(* IEC 61131-3 sources: ml2plc/benchmarks/st (part 19) *)

    weights_2 : ARRAY[0..287] OF REAL := [-0.086540468, 0.172771111, -0.220383257, -0.552691996, 0.0318835452, 0.612700164, -0.0329583585, -0.0454194695, 0.227657318, -0.476521522, 0.193516552, 0.416927308, 0.360883504, 0.35479334, -0.725205362, 0.0127351284, 0.00659608841, -0.077765286, 0.0985900313, 0.120690353, 0.105450228, 0.508144796, 0.130406424, -1.01746202, 0.904253662, -1.11978483, -0.232323259, 0.181972265, 0.00731435418, -0.0696650892, 1.03260088, -1.09293258, -0.287332207, 0.370921373, 0.321434826, -0.712032735, -0.0679141358, 0.179906562, -0.124551736, 0.192289323, -0.140516713, 0.0810432881, 0.856259704, -1.07160294, -0.223457828, 0.807030499, -0.976367593, -0.307652324, -0.786935031, -0.107092589, 0.150858521, -0.624960959, 0.36329934, 0.532729268, 0.384019405, 0.46479398, -0.802043259, 0.187860116, -0.136551112, 0.0211512949, 0.720803916, -0.827788591, -0.298880219, -0.202536553, 0.173984587, 0.185747623, -0.184981599, 0.0150071271, 0.00353488303, 0.0683722198, 0.187118113, 0.237856477, 1.01755667, -1.10523689, -0.268671334, 0.240274504, 0.30826062, -0.654990911, 0.872478366, -1.05786157, -0.229688749, -0.66336894, 0.0199285392, 0.532636046, -0.0841914713, 0.0642075539, 0.0174617469, -0.0364442356, 0.188555226, -0.242369831, 0.00474316673, -0.759811342, 0.954901636, 0.593428373, 0.096972242, -1.04332292, -0.205035418, 0.18625772, 0.209811807, 0.172150373, 0.0444886386, -0.186326519, 0.902395904, -1.12277734, -0.0967059359, -0.0028087846, 0.141072839, 0.130949974, 0.330060393, 0.323049426, -0.685176551, 0.492645383, 0.322297305, -0.804180861, -0.752909601, -0.107810475, 0.338000387, 0.220442653, 0.451399148, -0.57051903, -0.757164657, -0.126809373, 0.439987898, 0.0298772864, 0.00199659704, 0.166657642, 0.229579955, 0.268833876, -0.694251597, -0.0976240188, 0.0951045454, 0.2128084, -0.488305151, 0.345968217, 0.402587503, 0.0220696926, 0.122957081, 0.138620675, -0.146714658, 0.128199548, 0.0768355131, 0.988235116, -0.820175171, -0.0243866928, -0.564573824, 0.0925929025, 0.436609149, 0.605118215, 0.151139334, -1.10266984, 0.227359504, 0.0128947198, 0.0949031711, 0.120222516, 0.206790701, -0.00842625648, 0.120845072, 0.212780789, 0.12719503, -0.755692124, -0.150177613, 0.340954095, -0.853432715, -0.333076835, 0.391219765, 0.48939836, -0.116058439, -1.27640653, 0.0483904779, 0.217980474, -0.00876715779, -0.644433141, 0.0299610049, 0.399048507, 0.929591358, -0.906723499, -0.0457304083, 0.0974808037, -0.178352863, -0.0875617117, -0.169119462, -0.014128576, 0.133027628, 0.469002575, 0.474750727, -0.581674278, 0.372726113, 0.190089732, -0.973690569, -0.53365171, 0.140256211, 0.40247342, -0.113590144, -1.07570827, 0.916958451, -0.124050736, 0.0386698842, 0.104596823, 0.0975920856, -0.122577384, -0.230316952, 0.0917100608, -0.204680085, -0.157175794, 0.0664396286, 0.443755388, -0.550633371, 0.524068952, 0.155129775, -1.07333207, -0.0423594192, 0.0332752727, 0.193382502, -0.147190854, 0.123858854, -0.18527922, -0.251415074, -1.22913897, 0.845771313, -0.110015817, 0.065641731, 0.0683446452, 0.979607761, -0.910373867, -0.153985277, -0.0826165602, 0.125199199, 0.105670959, 0.127799779, -0.173133329, -0.0312328637, 0.147351772, 0.183071434, -0.226357937, -0.664937735, 0.321295112, 0.338666469, 1.03204453, -0.964660764, -0.207029104, 0.53012073, 0.460012823, -0.891147494, -0.551259696, 0.262762219, 0.241604507, 0.96495378, -0.912866771, -0.143412411, -0.645358205, 0.383842945, 0.425131768, -0.0753789395, -0.00826120377, 0.0299984515, -0.784333527, -0.1359182, 0.4243536, 0.178426176, -0.175408095, -0.077928111, -0.240787193, -0.203756183, 0.0390834771, -0.0964978486, -0.143233955, -0.104287267, 0.22191146, -0.0092907697, 0.138567775, -0.176785797, -0.841094136, 0.893011391, -0.736852944, 0.00464549148, 0.51239562, -0.529248655, 0.0516002066, 0.706514895, -0.518120229, 0.0655920431, 0.586107075, -0.604757965, 0.123719975, 0.379719675, 0.365877658, 0.503408611, -0.481252313];
    bias_2 : ARRAY[0..2] OF REAL := [0.0345217623, 0.145207137, -0.191580176];

END_VAR

VAR
    (* Merged variables from all regions *)
    buffer_0 : ARRAY[0..95] OF REAL;
    buffer_1 : ARRAY[0..127] OF REAL;

    (* Temporary computation variables *)
    i : DINT;
    j : DINT;
    t : DINT;
    sum : REAL;
    (* Computation helpers *)
    max_val : REAL;
    exp_val : REAL;
    exp_sum : REAL;
    (* Spatial loop variables *)
    oc : DINT;
    oh : DINT;
    ow : DINT;
    ic : DINT;
    kh : DINT;
    kw : DINT;
    ih : DINT;
    iw : DINT;
END_VAR

(* Forward pass execution *)

(* Region: r0 [ACYCLIC] *)
(* Acyclic Region r0 *)
(* Layer 0: Fused Linear + RELU *)
FOR j := 0 TO 127 DO
    sum := 0.0;
    FOR i := 0 TO 0 DO
        sum := sum + input_data * weights_0[i * 128 + j];
    END_FOR;
buffer_1[j] := MAX(sum + bias_0[j], 0.0);
END_FOR;

(* Layer 1: Fused Linear + RELU *)
FOR j := 0 TO 95 DO
    sum := 0.0;
    FOR i := 0 TO 127 DO
        sum := sum + buffer_1[i] * weights_1[i * 96 + j];
    END_FOR;
buffer_0[j] := MAX(sum + bias_1[j], 0.0);
END_FOR;

(* Layer 2: Fused Linear + SOFTMAX *)
FOR j := 0 TO 2 DO
    sum := 0.0;
    FOR i := 0 TO 95 DO
        sum := sum + buffer_0[i] * weights_2[i * 3 + j];
    END_FOR;
output_data[j] := sum + bias_2[j];
END_FOR;

(* Softmax: find max *)
max_val := output_data[0];
FOR i := 1 TO 2 DO
    IF output_data[i] > max_val THEN
        max_val := output_data[i];
    END_IF;
END_FOR;

(* Softmax: compute exponentials and sum *)
exp_sum := 0.0;
FOR i := 0 TO 2 DO
    output_data[i] := EXP(output_data[i] - max_val);
    exp_sum := exp_sum + output_data[i];
END_FOR;

(* Softmax: normalize *)
FOR i := 0 TO 2 DO
    output_data[i] := output_data[i] / exp_sum;
END_FOR;

END_FUNCTION_BLOCK

(* ---- MLP9_straton.st ---- *)
FUNCTION_BLOCK MLP9_FB

    (* Model Inputs/Outputs *)
VAR_INPUT
    input_data : REAL;
END_VAR

VAR_OUTPUT
    output_data : ARRAY[0..2] OF REAL;
END_VAR

VAR
    CONSTANT weights_0 : ARRAY[0..127] OF REAL := [-0.113805361, -0.131169349, -0.192945287, -0.0925860032, -0.117703564, 0.450317353, 0.395232439, -0.209253326, 0.52670908, -0.171847999, -0.00362640619, 0.448799431, 0.363001645, -0.0271579623, -0.0230307281, 0.528843641, 0.369391292, -0.0890475214, 0.398711413, -0.20652917, 0.420479208, -0.214330047, 0.343801081, -0.0572591722, 0.444781989, -0.109508358, 0.5149073, -0.195882052, 0.412400335, -0.190297425, 0.35653007, -0.00126373046, 0.476183206, -0.066968143, 0.488184482, -0.0159611255, -0.243453369, -0.186278701, 0.203586325, -0.212845653, -0.0807042271, -0.0202539116, 0.412385583, -0.144617856, -0.00571534038, -0.186419487, -0.193811327, -0.001996696, -0.204087764, 0.549255133, -0.182997674, 0.38119334, -0.182645351, -0.00299030519, 0.343619019, 0.518327653, 0.384723365, -0.20934774, 0.277335167, -0.172167048, 0.429218441, 0.469536155, 0.357460141, 0.234816477, -0.0928637683, 0.354974061, 0.0667782798, -0.128826559, 0.518400848, -0.0675187409, -0.198612809, -0.104182921, 0.397103459, 0.022735877, 0.368016571, 0.432546705, 0.49498266, -0.116236903, -0.0355618298, 0.522722244, -0.0902619362, -0.11224959, 0.353289217, -0.0632346869, 0.010258981, 0.431895882, 0.373197109, -0.130651206, -0.0309539437, 0.506278932, 0.413056433, 0.509223938, -0.0960097685, 0.367133349, 0.381490082, 0.457251966, 0.363914102, 0.42035231, 0.423214704, -0.188088998, -0.0470287502, -0.190154284, -0.162458539, -0.0485363007, -0.0830073208, -0.00753187714, 0.465610594, -0.205922633, 0.482488304, 0.448213607, 0.434718043, 0.34753862, 0.337949961, -0.031719774, -0.170038462, 0.495187283, -0.193692401, -0.172916174, -0.160878286, -0.200849622, 0.00499609578, -0.0520170256, -0.0275448263, 0.382134169, 0.507775307, 0.157361835, -0.0204105377, -0.147839844];
    CONSTANT bias_0 : ARRAY[0..127] OF REAL := [0, 0, 0, 0, 0, -0.100798227, -0.0795678124, 0, -0.108572058, 0, 0, -0.098264277, -0.0816824809, 0, 0, -0.0868740082, -0.0826022923, 0, -0.0856195465, 0, -0.0920739621, 0, -0.0772925317, 0, -0.0993444994, 0, -0.096356459, 0, -0.0921639502, 0, -0.080231972, -0.0145110283, -0.104885586, 0, -0.104719087, 0, 0.304739058, 0, 0.357667863, 0, 0, 0, -0.09254013, 0, 0, 0, 0, 0, 0, -0.119700968, 0, -0.0841121674, 0, -0.00373320258, -0.0695361495, -0.109383397, -0.0865293592, 0, 0.387899101, 0, -0.0930410847, -0.102059513, -0.0704434365, 0.379512459, 0, -0.0799476653, 0.354511678, 0, -0.0894547775, 0, 0, 0, -0.0889909193, 0.346559584, -0.0794480294, -0.0957549438, -0.101200089, 0, 0, -0.108003356, 0, 0, -0.07939253, 0, 0.350568563, -0.0959382132, -0.0757256672, 0, 0, -0.100857422, -0.0881503075, -0.105426408, 0, -0.0800946504, 0.326970756, -0.0932597071, -0.081825532, -0.0898775011, -0.0926302895, 0, 0, 0, 0, 0, 0, -0.00774373114, -0.0858005881, 0, -0.103054315, -0.0990050733, -0.0953028128, -0.0783599094, -0.0757565275, 0, 0, -0.100662939, 0, 0, 0, 0, -0.0165398363, 0.298638582, 0, -0.0855023414, -0.0985088944, 0.363575578, 0, 0];
    CONSTANT weights_1 : ARRAY[0..12287] OF REAL := [0.0951577127, 0.157444745, -0.116936132, -0.0790329278, -0.0228748918, 0.0134683251, 0.110163182, 0.0660780072, -0.0495770946, -0.0592429936, 0.134160757, -0.160569534, -0.0958634838, 0.142136246, 0.0809055567, -0.0727666095, -0.161114678, -0.133757368, 0.0792375952, 0.0649654567, 0.0525315702, -0.0809695944, -0.0614370704, -0.135633662, -0.00297276676, -0.0548477396, 0.128665984, -0.160567224, 0.00753733516, 0.0283032507, 0.12481007, 0.0217095912, -0.0424018651, 0.105811566, -0.0234863013, -0.0909486711, 0.050266549, -0.0875409767, -0.0314820856, 0.0861708969, -0.104749173, 0.0864515305, -0.0256673396, -0.078911148, 0.105528295, -0.106350139, 0.00202976167, 0.11709699, -0.0761083886, -0.15657708, 0.137355566, 0.0239440948, 0.131604254, -0.0955468714, -0.14261815, -0.0404164344, -0.05397138, -0.0310050994, -0.0330105126, 0.0184245408, -0.111915424, 0.0973271728, 0.103177726, 0.149213344, -0.0549873933, 0.0881988704, -0.0177367181, 0.124477774, -0.0285055786, -0.109965578, 0.0402032584, 0.0121235251, -0.0266363323, 0.125837356, -0.0728950202, -0.0705690533, 0.0583580136, 0.0598951429, 0.0236688703, 0.0522443801, 0.00132079422, 0.125945359, -0.00138136744, 0.0651458055, -0.120777965, -0.104297861, 0.0417176485, -0.161106139, -0.0645132065, 0.0710417032, 0.0645282269, -0.0479533747, 0.13674435, 0.106236696, -0.0604583621, 0.0287175775, -0.00439415872, -0.00736361742, -0.134950846, -0.135192379, 0.10444808, 0.0236009806, -0.103126153, 0.0975316465, 0.139209658, 0.0520739704, 0.125309825, -0.0581694618, -0.162468061, -0.0841054246, 0.0483714789, -0.0566895753, -0.0466354638, -0.104527183, -0.007353127, -0.0725882053, 0.0929109752, 0.113443941, 0.0509717613, 0.0587531328, -0.117151141, 0.0126229078, 0.0203929991, 0.047550723, 0.0517018735, -0.101339415, -0.138496399, 0.00150629878, 0.0771658868, -0.00845770538, 0.0908749104, 0.0518915504, 0.0117899328, -0.145934269, 0.0225093067, -0.0222804546, -0.00221456587, 0.0128537863, -0.0276821703, -0.120568201, -0.0423685834, 0.116727293, -0.0766037181, -0.0683219507, 0.138370246, 0.146753311, 0.0569230765, -0.0658973753, 0.0545879006, 0.105433077, -0.0373315513, 0.161194414, 0.0101915747, -0.0552281886, -0.103356332, 0.0682205409, 0.0157359093, -0.0698226318, -0.0442622453, -0.0125101805, -0.033475399, 0.0732399672, -0.149365753, -0.123059414, -0.124025911, 0.0979141891, -0.0852181315, -0.123718902, -0.137371242, 0.0357241184, 0.132824361, -0.160526261, 0.00875844061, 0.14891094, 0.020388782, 0.127746224, -0.0733599514, 0.12927103, 0.156546056, 0.144431114, -0.058117643, -0.0785800591, -0.0507855564, -0.160170823, -0.0641571879, -0.027300939, 0.108366787, -0.0391465947, 0.0696284622, 0.0237422287, -0.11445865, -0.11570774, 0.0200967491, -0.131474406, 0.120322555, 0.106915504, 0.106001765, 0.15025726, 0.148201168, 0.0288652182, 0.0153841078, 0.147035837, -0.0442098752, 0.0455059856, 0.08771047, -0.0411697626, 0.0291817933, 0.118134856, 0.101055682, -0.000335618854, -0.0269186497, 0.015304774, 0.0589915514, -0.02176328, -0.14560017, -0.0776190683, 0.0365733057, -0.0838752836, 0.153584182, 0.134814322, 0.148770154, -0.0831061155, 0.0914156139, 0.077782169, 0.0720475763, -0.0280352235, 0.0480267406, 0.0686243623, 0.0797413886, 0.0645133257, -0.0962903649, 0.0324638784, -0.0570613667, -0.0719860792, 0.111080825, 0.119137555, -0.055265218, 0.0108719021, -0.0382692516, 0.146787912, -0.100032538, -0.0835579708, 0.00157497823, -0.162271053, 0.119353175, -0.0655590296, 0.0131833553, 0.069874689, -0.0753858536, -0.0472645536, -0.0861709341, 0.0184095502, 0.142682731, 0.0667904317, 0.000965476036, -0.115095079, -0.0968379378, -0.121067345, -0.0672623515, -0.112838328, -0.0351838768, -0.137819111, -0.112566784, -0.155080765, 0.138557822, -0.162448362, -0.12402942, 0.0698025823, 0.118413299, 0.139092475, -0.0617644563, -0.125346243, 0.0916123688, 0.076207146, -0.0628192499, -0.128253579, 0.120955229, 0.148212641, -0.0932002217, 0.117295235, 0.161221325, -0.106977157, 0.0483250469, -0.150214329, 0.0903045833, 0.0870901346, 0.149560899, -0.0276673287, -0.151596636, 0.0847090334, 0.127780765, -0.15172115, -0.118571639, 0.0389828235, 0.0767906606, -0.0856763497, 0.0160828382, -0.121637389, 0.0912489295, -0.14491263, 0.131868184, 0.0672539175, 0.0127351731, -0.00589309633, -0.0622787848, -0.141520515, -0.0427362323, -0.0998942479, 0.149263471, -0.152347118, 0.0028988719, -0.00683000684, 0.146410555, -0.0533801764, 0.0977630019, -0.00881588459, -0.160895512, -0.0131007433, 0.0372889936, 0.126067817, 0.11309135, 0.0728558898, -0.0335129797, -0.0818832964, -0.0330946892, -0.0781284794, -0.155981824, 0.0711639673, -0.0405116826, 0.0357084721, 0.142399669, 0.138510466, -0.114842109, 0.0368577391, -0.0718035027, -0.0764543861, -0.107536398, -0.139627516, 0.00174733996, 0.094630897, 0.0877837241, -0.0499476343, 0.0859448165, -0.0901338086, -0.121612534, 0.0269791335, 0.0815927088, 0.0611288548, -0.0593353137, -0.153852284, -0.0354756266, -0.0991432667, 0.141438067, -0.00173516572, -0.0234908611, 0.0649795383, -0.114180557, -0.142907768, 0.0548550785, 0.0757389814, 0.0898238719, 0.0306845456, -0.0634233654, 0.149431825, -0.0129109174, -0.0298580527, 0.0128320903, -0.119393483, -0.0556279495, -0.048238501, -0.110748321, 0.160280555, -0.107997969, -0.129245013, -0.0782359764, 0.0218218118, 0.0503502041, 0.101736844, 0.0445458442, -0.0318994522, -0.048770234, 0.0895831585, -0.138157532, 0.0388857722, 0.111648083, 0.145862103, 0.0815838128, 0.054871738, -0.0941967666, -0.126886413, -0.0578072369, 0.0876997113, -0.108099304, -0.0487953201, -0.131870151, 0.0197252482, -0.0851159021, 0.0999375284, 0.157903999, -0.0588724166, 0.152515322, -0.0926127732, 0.109808058, 0.161163688, 0.153266072, 0.108911484, 0.0491682738, -0.157219395, 0.0929915309, 0.0676452518, -0.0539523736, 0.0412925184, 0.0595459938, -0.115160167, -0.0217127502, 0.0798177123, -0.00466352701, 0.0912430882, 0.0433716774, -0.145626664, 0.148768365, 0.0322260559, 0.131735057, -0.131727949, 0.0504067838, 0.00729522109, -0.039368853, 0.121461481, 0.132999808, -0.0395063236, 0.00795516372, 0.145861775, 0.105656266, -0.156878084, 0.00268745422, 0.117816895, -0.124721214, -0.0546680093, 0.0303108841, 0.0794312507, -0.0877228901, -0.0310570002, -0.135552973, -0.121911898, -0.120446339, 0.0388385206, 0.108996451, 0.0305833668, -0.0586595982, -0.140537083, 0.160965115, -0.125315413, -0.0336649269, 0.144092739, 0.0993903279, 0.116826385, 0.0198810548, 0.130669534, -0.007835567, 0.0403493196, 0.149000049, 0.0241642743, 0.16068995, -0.0206242353, 0.0651469827, -0.0246725529, 0.067141965, -0.0331727564, -0.144538388, -0.0538310185, -0.0991705433, -0.0017388314, 0.16014412, -0.106752947, 0.101663619, -0.142054304, -0.107962027, 0.019818306, -0.0550122112, -0.0132327527, -0.0847105384, 0.509194136, 0.0538960695, 0.604936779, -0.265589058, -0.140676975, -0.00574114919, -0.43431446, -0.453494668, 0.0540918261, -0.406886041, -0.21926257, 0.163309574, -0.143326595, -0.642100513, -0.723519862, 0.570846677, 0.244765401, -0.379419535, 0.00814934261, -0.540151834, 0.154496402, -0.0546880662, 0.161006272, -0.4712421, -0.312546521, -0.449770659, 0.659415066, -0.13482137, 0.0830492079, 0.52391237, -0.565974474, 0.158174455, -0.0621462315, -0.70691061, -0.154083952, -0.360878319, -0.407535791, 0.656996191, -0.369862318, 0.627200603, 0.069169119, -0.546665549, 0.0077586174, 0.4769786, 0.140734434, -0.0507009253, -0.760944128, 0.602752507, -0.571398199, 0.0918866098, 0.00788346305, 0.0322130509, 0.288204491, 0.329203099, -0.392646372, 0.0749019235, 0.320154548, -0.691001058, 0.112304956, -0.125678852, -0.333393902, -0.394726753, 0.752456069, 0.394099623, -0.124766201, 0.0376506299, -0.0682738349, -0.246535376, -0.51199317, -0.137057155, 0.122536659, 0.519263268, 0.0833194107, -0.686214447, 0.123675488, 0.141091406, 0.155417144, 0.331035525, -0.519244015, -0.223143131, 0.621623278, -0.614489675, 0.437765509, 0.0805219561, 0.413208932, -0.0631952509, -0.0913754106, 0.0515855551, -0.160588577, 0.397252113, 0.431347072, 0.408398241, 0.408925176, 0.597231805, -0.336975992, 0.0440444462, 0.270032376, -0.121744737, 0.549877822, -0.422593564, -0.0661128834, -0.17437312, -0.417972744, -0.310103178, -0.0716258809, -0.33077088, -0.205869734, -0.153525308, -0.139355108, -0.438011259, -0.584835529, 0.465125173, 0.344738692, -0.14478299, 0.156904221, -0.624013662, -0.153481901, 0.0398430228, -0.0846624002, -0.516546309, -0.242195129, -0.376353711, 0.532166958, -0.144245222, 0.0689140931, 0.36220032, -0.267864943, 0.057710737, 0.0646699518, -0.586554945, -0.0401847661, -0.248956472, -0.272385627, 0.415772557, -0.0767131969, 0.310505778, -0.0379597098, -0.274617344, 0.126220137, 0.480036318, -0.0241271257, 0.0331539959, -0.324106157, 0.501049876, -0.291424572, -0.0870115086, 0.0509127118, 0.0394147225, 0.584093153, 0.503804743, -0.218451321, 0.00519318879, 0.607654095, -0.3049227, 0.145615906, 0.05105225, -0.202767462, -0.423024982, 0.729864001, 0.276849747, 0.0496818721, 0.0660526454, 0.0130212307, -0.0571260527, -0.439201325, 0.0459277742, -0.0404780358, 0.408804804, 0.0655715987, -0.476458848, -0.0844522044, 0.124375969, 0.114283532, 0.39356488, -0.548989713, -0.34556523, 0.631348431, -0.40491116, 0.518371046, 0.135800749, 0.560781419, -0.00710113347, 0.0723592117, 0.0476910472, -0.124959633, 0.328189194, 0.532768965, 0.587405443, 0.499420702, 0.671146929, -0.352552384, 0.0768999159, -0.0319315642, -0.100787431, -0.0804701298, -0.146786034, 0.141987205, 0.0561998785, 0.0398712754, 0.0927682817, 0.109196901, -0.0432840809, 0.0716784894, 0.0145284683, -0.095403865, 0.0917330086, -0.15252769, -0.110293895, -0.0509034023, 0.0978683233, 0.0202671587, 0.00549578667, -0.135518357, -0.146398097, 0.124808073, -0.13327761, -0.13578631, -0.0443552658, -0.123986423, 0.163084328, -0.0966529474, -0.134083807, 0.0854204893, -0.0765637606, -0.0741811767, -0.00683036447, -0.118621819, -0.039869912, -0.162193045, -0.104409263, -0.056582585, -0.001865834, 0.154557496, 0.0310758501, 0.0742693543, -0.0389179736, 0.112253129, -0.0996025354, 0.038610369, -0.0614454597, 0.0836289823, 0.107963115, 0.140558034, 0.0794830322, 0.163360059, -0.163278833, -0.0120799392, -0.0656130388, 0.00880923867, -0.0657925308, -0.0760729611, -0.075019531, 0.114507735, 0.0841428488, 0.0406958908, 0.11450699, -0.151554912, -0.122948989, 0.0699587762, -0.110302597, 0.00226099789, 0.0974447727, 0.0653391182, 0.108267993, -0.0920944661, 0.15465036, 0.112603068, 0.0013948977, 0.14819929, -0.144036621, -0.016038239, -0.139199302, -0.0771588236, -0.0928127542, -0.0338050127, -0.0522177219, -0.157671407, -0.00344249606, -0.0332395732, -0.113233492, -0.158796951, -0.13916111, 0.0589568615, 0.0945762098, 0.14930898, 0.0418180823, -0.0978229716, 0.0602630973, 0.322021961, -0.0053896904, 0.467693686, -0.249736562, 0.126417518, -0.138710305, -0.363732606, -0.456968129, -0.0944563299, -0.472876072, -0.21804218, -0.143095255, 0.0928375497, -0.57138437, -0.472568661, 0.646057606, 0.351664901, -0.415040404, -0.111070551, -0.65686512, -0.10573642, -0.0150539875, -0.144721866, -0.56100738, -0.30737561, -0.586903989, 0.616061807, -0.043527022, -0.0646082535, 0.434298456, -0.282648176, -0.0882620364, -0.12533547, -0.59989053, 0.125016868, -0.46765244, -0.364355326, 0.523267984, -0.340620995, 0.308997214, -0.018915683, -0.40029791, 0.0643675029, 0.254231155, -0.00991281867, 0.117880344, -0.428295225, 0.443931401, -0.469592839, -0.0985035226, 0.0645282492, 0.0728940368, 0.45560959, 0.487523675, -0.384809881, 0.0336826444, 0.39610061, -0.386167377, -0.0381661206, -0.136605546, -0.445077538, -0.44675684, 0.475525707, 0.245289952, -0.161932707, -0.115931481, 0.0207827687, -0.0385752581, -0.230016008, -0.143260673, -0.0719312429, 0.350897193, -0.112227477, -0.549400151, 0.0996975377, -0.158407763, -0.00293686986, 0.503760517, -0.545467556, -0.259034455, 0.453600407, -0.456205547, 0.487957925, -0.122733943, 0.287507385, 0.0341648608, -0.0692357272, 0.137745768, -0.02918984, 0.201632515, 0.316503704, 0.563527167, 0.428642005, 0.695099711, -0.341352791, 0.14451462, 0.00366416574, -0.0520999208, 0.0875412226, -0.116182968, -0.157112911, 0.114217222, -0.0688723326, -0.121052325, 0.0575330406, 0.0796439499, 0.0595702976, 0.0227632523, -0.0794479102, 0.126714766, -0.0488853008, 0.0934711695, 0.122365475, -0.0437675789, 0.0868758857, -0.0134203285, 0.0346060544, -0.0367608815, 0.0463865548, -0.0707047656, 0.150832742, -0.128055975, -0.0556442216, 0.00231200457, -0.111579061, -0.0886108428, -0.129191309, -0.161951363, 0.0831619501, -0.0794863105, 0.103473008, 0.159343034, -0.0559051931, 0.062377587, -0.121212967, 0.0833023041, -0.162734151, 0.0321030617, -0.10398519, -0.138421714, 0.045194909, 0.142874509, -0.0367347449, -0.155020788, -0.152351826, 0.0173095316, -0.0145311207, 0.0364078283, 0.0694433898, 0.031635046, 0.0519284606, 0.1198695, -0.0134465098, -0.142700329, 0.0394844264, -0.158252656, -0.0392903835, -0.0576177537, -0.0491104871, 0.0735302418, 0.0511014611, 0.109477192, 0.0833617002, 0.101866454, 0.0914892256, 0.00224284828, 0.126525789, 0.137383074, 0.0791972429, -0.0692049414, -0.125604168, 0.128060102, -0.0253694654, 0.0628164113, 0.03625682, 0.159057289, 0.0904439092, -0.0538290292, -0.162247017, 0.00659917295, -0.0887682065, -0.0221569985, -0.0965008438, 0.104463339, -0.0614345372, 0.0150002241, 0.0888507366, 0.115881771, -0.111798167, 0.0199936181, -0.154604435, 0.0775321275, -0.02869986, 0.0626578331, -0.0132484436, -0.0378343761, 0.0255666375, -0.137642473, 0.0340280831, 0.0923664272, -0.132832348, -0.161153629, -0.0162264407, -0.138787255, -0.0474235192, -0.10354051, -0.0473156273, 0.0843745917, -0.151293129, 0.124063998, 0.113260567, -0.137583464, 0.0871079266, 0.0880226791, 0.123843074, 0.1298002, 0.0235676616, -0.118507646, -0.130145669, -0.0655051842, 0.0768328458, -0.0903019831, 0.120177537, -0.109550744, -0.12586607, 0.119989842, -0.06112881, 0.150598377, -0.0707290024, 0.0344911516, 0.103849113, -0.135946766, -0.0548578054, 0.0875094533, 0.113336772, 0.096303165, -0.068084158, 0.114509881, 0.1175614, -0.0225681514, 0.146655113, -0.00232343376, -0.0178669691, 0.054963395, -0.140081167, -0.0873917267, -0.101093426, -0.0865101367, -0.0871431231, -0.109610252, -0.147202581, -0.0557942912, -0.0006223768, -0.134950295, 0.162944168, -0.0371381789, 0.129121751, 0.157590866, 0.122555614, -0.00439842045, 0.156742811, -0.105628684, 0.0453346372, -0.0737311915, -0.0812637657, 0.127866268, 0.059443593, -0.0491509959, -0.0971391797, -0.143130645, 0.0233585835, -0.0147621185, -0.159102827, 0.149393588, 0.0969157219, -0.102926373, 0.154051632, 0.112800837, 0.0364580452, -0.0520509854, 0.0394695997, 0.0302900523, 0.1545147, 0.0542997718, 0.0890843868, 0.0546405762, 0.0287235081, -0.173261896, 0.490024894, 0.0681065172, 0.361833811, -0.328347623, -0.0356032252, -0.133056432, -0.494118333, -0.601521552, -0.121832028, -0.589727759, -0.277259827, 0.111315638, 0.0659579858, -0.741538644, -0.492740691, 0.550138712, 0.320899546, -0.288761914, -0.00195023709, -0.537688792, 0.099278003, 0.00579982996, -0.0347415805, -0.72761929, -0.377573043, -0.555244505, 0.456523657, 0.0320400745, 0.036451485, 0.486669511, -0.378461182, -0.152018994, -0.136228755, -0.720117569, 0.0192903578, -0.531963825, -0.469921142, 0.589513958, -0.366701841, 0.412990361, -0.158252299, -0.364246905, -0.160873383, 0.37125057, -0.00136806071, 0.0729077011, -0.559927881, 0.583796501, -0.387921512, 0.00662960112, 0.00455707638, -0.0358150043, 0.490136683, 0.529693484, -0.326329947, 0.022318691, 0.567211449, -0.707156956, -0.149156183, -0.132085413, -0.527429581, -0.507927239, 0.653061748, 0.349608958, 0.152013838, 0.0440299511, -0.0555629432, -0.101837404, -0.348313838, 0.0049868077, -0.0747583583, 0.262050003, -0.159494683, -0.424277574, -0.149270624, -0.160396859, 0.0718324929, 0.430129915, -0.734822154, -0.220166579, 0.418183774, -0.722909093, 0.251368821, 0.00369682908, 0.448462456, 0.131171644, -0.0492361449, -0.00822554529, -0.146481872, 0.301343501, 0.379717827, 0.573642671, 0.471275508, 0.538758397, -0.350973874, 0.12145821, 0.671127796, 0.116494, 0.640164316, -0.551232457, 0.0458213836, 0.122570068, -0.612397373, -0.660989344, -0.088481836, -0.605110645, -0.603729784, 0.0518653244, 0.139900357, -0.674467802, -0.719813704, 0.707245648, 0.596261024, -0.500923991, -0.00499203429, -0.699686885, 0.0658935606, 0.0570179373, 0.1512371, -0.636342168, -0.418134749, -0.620170534, 0.763878882, -0.002538234, -0.0417705178, 0.420946479, -0.688793957, 0.064556092, 0.157188416, -0.759609997, 0.0812719166, -0.453400403, -0.567348719, 0.724059165, -0.203651771, 0.611069858, 0.0227045268, -0.291180491, -0.157189071, 0.754448414, 0.085985437, -0.119775772, -0.712979138, 0.698715329, -0.58169204, 0.148470551, 0.0952268913, 0.0562097244, 0.633901775, 0.590043008, -0.511904299, -0.128872991, 0.575819671, -0.675768137, -0.0152154565, -0.00212833285, -0.472860008, -0.69616574, 0.622911692, 0.343438059, -0.0224477351, -0.0405841023, 0.0385661274, -0.257873476, -0.396772712, -0.152293921, -0.156207159, 0.595220387, -0.0240174532, -0.615511596, -0.13495256, -0.106912807, 0.0843406469, 0.526772499, -0.736953795, -0.275285572, 0.692019939, -0.582976937, 0.498922467, 0.0128312707, 0.633550167, -0.0273342133, 0.109861545, 0.103651047, -0.0617552027, 0.510849655, 0.394558609, 0.545751154, 0.393026024, 0.793120563, -0.497044265, 0.092567116, 0.138860226, -0.0985106304, 0.00336945057, -0.130671352, -0.111542739, 0.143976063, 0.0285258293, 0.113393039, -0.0218960196, 0.0309942961, -0.0104740858, 0.0956641138, 0.0878303051, 0.102058023, 0.00174370408, -0.117548563, -0.155215263, 0.134208828, 0.0980995595, -0.134259984, 0.0419485718, -0.0534096435, 0.0429573655, 0.0513623953, -0.14403373, 0.06175825, -0.122290827, 0.0777258277, -0.151134908, 0.0914635062, 0.140266359, -0.00751279294, 0.00970570743, -0.0983380377, 0.0919840634, -0.0801352561, 0.0911718011, 0.108400077, -0.161801755, 0.135701865, -0.131035775, -0.0860919133, 0.0889713168, -0.0941296518, -0.0192143917, 0.100918174, -0.0230973512, 0.117296249, 0.133148789, 0.156041861, -0.0570620298, -0.0986587107, -0.148947418, -0.135748416, -0.0595284253, -0.134941593, 0.117915601, 0.0543765277, -0.124985032, 0.066407606, 0.0267682225, 0.0470175147, -0.162895411, -0.149206594, 0.153207392, -0.00830924511, 0.00621114671, 0.146200955, 0.132364035, -0.154241115, 0.0508376509, 0.0611464828, 0.121670395, 0.104352921, 0.0689978153, 0.0547138155, 0.0552895218, -0.154357553, -0.0046634376, 0.118674546, -0.0442880765, -0.0731509998, 0.00893263519, -0.0351747423, 0.014497757, 0.0777242631, -0.111611374, -0.0725884363, -0.112329312, -0.0154200494, 0.146003842, -0.00320079923, -0.163586318, -0.0718479902, 0.0270866752, -0.0277421027, 0.154627293, 0.0143596977, 0.131777287, -0.116288751, -0.142893523, -0.157827795, -0.0544529706, -0.0255519301, -0.0792789161, -0.0977822319, 0.143588871, -0.124468245, 0.0958327651, -0.0322359949, 0.00266860425, -0.1135519, -0.140336871, -0.14343977, -0.113305256, -0.0109504908, 0.0786850303, 0.0330305398, -0.00475849211, 0.0163063854, -0.0716166347, -0.0528806821, 0.0159133375, -0.0289545059, -0.15040499, 0.153120875, -0.0435663164, -0.0760979354, 0.160244167, -0.0592714772, 0.132729143, -0.00471362472, -0.0540071949, -0.0376077443, 0.0736211985, 0.0239118934, 0.0179463774, 0.0792258084, -0.1428767, 0.158036083, 0.15304625, -0.0280214399, -0.0129368603, 0.0730203241, 0.00552131236, -0.102222949, -0.00217039883, 0.149807036, 0.0687736124, -0.0731835365, 0.0183587819, -0.0314919204, -0.119318336, -0.0418934301, -0.118667156, -0.141958326, -0.00374318659, -0.0770075023, -0.129735336, -0.119574621, 0.0406397432, -0.152146041, -0.0276105553, -0.0321829766, 0.0301983207, 0.0734649152, -0.0383871794, -0.158686012, 0.0197154433, 0.136941463, -0.0486620665, 0.0317238569, 0.135865867, -0.0451636165, 0.0228485912, 0.127936155, -0.0893768072, 0.0435742736, -0.0214909464, 0.0240473002, 0.103848428, -0.122813389, -0.0357450694, -0.0580369905, -0.0383514315, -0.0267788023, -0.0101375729, -0.0783320889, 0.0894583762, -0.11558798, 0.00936958194, -0.171604529, 0.37826997, -0.139284834, 0.530997694, -0.212191448, -0.00569155812, -0.13463667, -0.152116403, -0.322950393, 0.0285518467, -0.350297242, -0.0644152015, -0.0703600869, 0.0551211797, -0.260502994, -0.240122318, 0.572239399, 0.46966812, -0.211586058, -0.0670061857, -0.311251044, 0.0108838379, -0.0651359409, -0.150437683, -0.45188126, -0.119499251, -0.282272905, 0.483443588, -0.105406582, 0.00445411028, 0.432145655, -0.332937509, 0.0562750995, 0.046805948, -0.397827655, 0.00858733058, -0.166388154, -0.121550895, 0.298872322, -0.187453955, 0.401923031, -0.0599540249, -0.302921563, 0.0653752834, 0.423189819, -0.0816778094, -0.0318836868, -0.39043653, 0.558439434, -0.0932632908, -0.0381754935, 0.0619168989, -0.0710496083, 0.174890399, 0.151282564, -0.119489975, 0.0900167823, 0.294368684, -0.483624071, 0.00194258988, -0.0865473673, -0.32862553, -0.157639489, 0.403094679, 0.387990355, -0.0647413582, -0.0843798593, 0.115365654, 0.0828580633, -0.151365161, -0.0210992191, 0.113412887, 0.254138768, 0.151015371, -0.398343295, 0.108841717, -0.00285227597, -0.123278439, 0.263769329, -0.393478274, -0.168504938, 0.443632662, -0.519051313, 0.384981513, -0.123920478, 0.161044911, 0.0879419446, -0.115611427, 0.0700436532, 0.0192385763, 0.17883873, 0.29301405, 0.17283237, 0.403273553, 0.477420956, -0.0488811806, 0.0120467003, 0.375956684, 0.12920621, 0.699442625, -0.524834216, -0.121545583, -0.137277544, -0.379925132, -0.548032999, -0.137724444, -0.607119679, -0.298528701, -0.047074832, 0.124948837, -0.770748496, -0.59968704, 0.591483057, 0.494383752, -0.383634984, -0.0311492104, -0.839230597, 0.0822430253, 0.108918607, 0.0935982764, -0.704104125, -0.356704116, -0.755547345, 0.739801884, 0.0709495842, -0.0763972551, 0.586229026, -0.47056818, -0.159900367, 0.113844991, -0.622358143, 0.029721722, -0.346799523, -0.55520165, 0.644957125, -0.180072859, 0.576455891, 0.0997797251, -0.623195469, 0.0432468951, 0.458427429, -0.0401322469, 0.16339761, -0.614164293, 0.528877735, -0.538296103, 0.136346489, -0.075547725, -0.0998050198, 0.596348763, 0.419898242, -0.4143987, -0.159823969, 0.517159164, -0.650046349, 0.15730226, -0.0963807777, -0.466536582, -0.491415739, 0.719611645, 0.343206763, 0.0584654361, -0.142278448, 0.0578351021, -0.0912387967, -0.318331808, 0.0348259062, 0.0380429775, 0.49942252, 0.0159810036, -0.578052282, -0.0696077943, 0.158027083, -0.026454702, 0.356168002, -0.762355506, -0.36194548, 0.6623348, -0.802657306, 0.372459531, -0.0177604109, 0.304009169, 0.155115753, -0.0184258223, -0.163283899, -0.114621252, 0.46932736, 0.372504145, 0.596721768, 0.556582689, 0.814534783, -0.486625105, -0.0306815803, 0.025685221, -0.0854586959, -0.162569836, -0.135548756, -0.059675537, -0.0324641466, 0.0446429998, -0.0321180075, -0.122927211, -0.13147369, 0.0658006519, -0.110076934, -0.111618593, 0.00718669593, -0.00896142423, -0.0493594408, -0.00285220146, 0.0551111698, 0.0986686349, 0.055111438, 0.0596161038, 0.0573125035, 0.107870221, -0.151748225, -0.00931198895, 0.114553243, 0.045098573, 0.139641732, -0.118258893, 0.0492309481, -0.147999257, 0.0854483098, 0.0512779206, 0.0119998306, 0.122926444, -0.128550708, 0.0254909694, -0.129055202, 0.0566999912, -0.105781332, -0.152117521, -0.0161006302, 0.0674194843, 0.0572939217, 0.0674108565, 0.13852039, 0.115954906, 0.0876097679, -0.0544308051, -0.110972494, -0.120723307, 0.0269239992, -0.135097399, 0.123992145, -0.0166501552, -0.141229227, -0.159426779, 0.0976717174, 0.117086768, 0.0111603737, -0.0502780974, -0.060312897, 0.0254771262, 0.0836675465, -0.0817346647, -0.0361399204, -0.0936484933, -0.0401128158, 0.119081914, -0.00509734452, 0.00264297426, 0.128084451, -0.1033554, 0.10066396, 0.039713636, -0.0618551373, -0.159436136, -0.0763160959, 0.0509372652, 0.0389629155, 0.106907725, 0.0491593778, -0.0575763136, -0.0938487053, -0.0658800527, 0.132949799, 0.104060411, -0.108209498, 0.0415501744, -0.026478231, 0.0722434968, -0.0932231322, 0.0147849023, -0.043643266, -0.0856521204, -0.0291557759, 0.306721389, 0.109158009, 0.49179405, -0.420839518, 0.0140549093, -0.0313300639, -0.606817007, -0.659625411, 0.150411934, -0.623003006, -0.246826604, -0.0737855881, -0.0419784896, -0.615695417, -0.481226534, 0.597063065, 0.44444707, -0.134298146, 0.0320285782, -0.660773993, 0.113458276, 0.0531203002, -0.098570019, -0.45033744, -0.484261781, -0.689734042, 0.562280774, 0.0319197029, -0.0688617602, 0.32306987, -0.5978176, 0.128473967, 0.0780164897, -0.474267006, -0.0436522737, -0.478814751, -0.266604304, 0.694460571, -0.232730657, 0.662883461, 0.0570311993, -0.367856115, -0.000895634294, 0.52646184, 0.134058058, 0.120685995, -0.514581442, 0.661175847, -0.300899088, 0.0549793541, 0.14357692, 0.132087469, 0.47485584, 0.40371874, -0.450551987, -0.0643547475, 0.617871702, -0.51760745, 0.00401297212, 0.0904693902, -0.450388253, -0.561228812, 0.767486393, 0.521278679, 0.0991616845, -0.0885995254, 0.105113, -0.235097632, -0.318120718, 0.0142247677, 0.0335372984, 0.287734181, -0.111655399, -0.55720073, 0.0110705784, -0.146056443, -0.123433426, 0.447484374, -0.661124706, -0.218874723, 0.405974746, -0.544911742, 0.547021866, -0.0104877502, 0.408579797, -0.0582740754, -0.0506011918, -0.132799953, -0.0332781523, 0.229849413, 0.365624577, 0.456757605, 0.329040736, 0.700344622, -0.445164233, 0.0976964235, 0.0648446828, -0.068145223, 0.0261178315, -0.0758716539, -0.11843881, 0.0534669161, -0.0287542939, -0.0270300508, 0.116880029, -0.15281184, -0.143178761, -0.0476447642, 0.129514754, -0.04601188, 0.160012543, 0.118659914, 0.149800211, -0.13829422, 0.0939094126, 0.155368924, 0.0961622298, -0.106080502, -0.122065529, 0.119311541, -0.0381726027, -0.106803127, 0.107218027, -0.0559676215, -0.111247316, 0.121596783, -0.107714251, 0.160762399, 0.156685174, 0.0132414103, -0.0558521226, -0.141591221, 0.128323823, 0.028944701, 0.0827338994, 0.157560378, 0.115682334, 0.0123288482, -0.145623147, -0.0590403602, 0.140045971, -0.0549273789, -0.160698339, 0.0633182824, 0.0278355181, -0.119194791, -0.132618979, 0.0221527368, -0.088305898, 0.0622185767, 0.0339545757, -0.0343891829, -0.106521636, 0.00423894823, 0.148137361, -0.112975411, -0.0411045551, 0.0453726053, -0.101802856, -0.057251513, 0.0613131076, 0.109502971, -0.142033398, 0.113049865, -0.0965993702, -0.0804046541, -0.0301233977, 0.0585615784, 0.0964251161, 0.024016276, 0.0813086033, -0.139627039, 0.0790618807, -0.124294251, -0.0733692795, -0.0137121975, 0.160125464, 0.162649721, -0.0006339252, -0.0301739722, 0.114816785, -0.017870754, 0.157246739, -0.0358114392, 0.111886859, -0.0933679715, 0.00454731286, 0.00260421634, -0.0804726258, 0.0668208748, 0.0768273473, 0.125154927, 0.274506718, -0.108850718, 0.700801909, -0.369239748, 0.0876085758, -0.161883846, -0.514561892, -0.542895496, -0.107240081, -0.42260617, -0.502647698, 0.0705162585, 0.144359604, -0.694857001, -0.416060179, 0.587688744, 0.355567843, -0.281352311, -0.0684666783, -0.757600725, -0.147242934, 0.0389017314, -0.0919541046, -0.378516853, -0.251506805, -0.627697766, 0.526410222, 0.0694428086, -0.161055908, 0.480900168, -0.357618064, 0.140872747, -0.0966657028, -0.500380397, -0.0831384659, -0.474707037, -0.278030217, 0.499889076, -0.232787937, 0.37974149, -0.115171164, -0.424904823, -0.108000465, 0.337988645, -0.0508833006, -0.139382228, -0.631711364, 0.565640092, -0.327750266, 0.000222578645, 0.00204922329, -0.0240393933, 0.509130716, 0.324508965, -0.287034571, 0.162361532, 0.528735876, -0.58035022, -0.160843223, -0.144021139, -0.458830506, -0.527102709, 0.732310951, 0.509064853, -0.146347567, 0.0154169202, -0.0792815685, -0.0401333235, -0.453812152, 0.130225003, 0.110475332, 0.320518881, -0.0578591041, -0.685087562, -0.117642418, -0.0518023893, 0.0193753839, 0.43134895, -0.422985643, -0.215356767, 0.58423388, -0.718991458, 0.310932666, -0.12200442, 0.516650975, 0.0559484214, 0.0660565645, 0.00705075264, 0.0235438496, 0.346917182, 0.519647956, 0.423651427, 0.500849247, 0.526616335, -0.317088783, -0.0553651899, -0.125636369, 0.0505954176, 0.0875653625, 0.121670246, -0.13142243, -0.108666703, -0.0196895301, -0.0435220301, 0.0524786562, 0.132473052, -0.159008086, -0.147173628, -0.0993846059, 0.0238770843, 0.0251523107, -0.030727312, -0.132775143, -0.00789819658, -0.132826537, 0.160109013, -0.0251740515, -0.00414946675, -0.0882047564, -0.0729843006, 0.108053684, -0.109337732, -0.0265030414, -0.13644895, -0.0482193008, -0.0911523923, 0.1174016, 0.0776960999, 0.0588599294, 0.157708555, 0.0380899161, 0.0525003821, 0.0228294283, -0.0777316019, -0.0135964602, -0.0270562768, 0.132765859, 0.160099089, 0.103721738, -0.0351472348, -0.103914872, 0.092781961, -0.0441754609, -0.0600776374, 0.0380554199, 0.00477176905, 0.12860328, 0.144565284, -0.115085281, 0.112356871, 0.068504408, -0.107143931, -0.134599656, 0.157213449, -0.089699626, -0.0571548566, 0.0579648465, -0.0209368616, -0.0799036324, 0.108259439, 0.149805754, 0.0211984515, 0.0990114808, -0.0506354049, 0.0673717558, 0.0768712014, -0.0233896524, 0.014501974, -0.0134821385, -0.136239886, -0.0283126235, -0.145492673, 0.10757947, 0.0263343155, 0.0350339562, -0.0399172083, -0.0977675617, 0.152113855, 0.14911887, -0.0786012113, 0.126734585, 0.0955718458, 0.114830911, -0.145009786, 0.0676991791, -0.0959686413, 0.100555807, -0.0834331065, -0.0733062178, -0.107300639, 0.071643129, -0.075324364, 0.495172858, 0.0116833299, 0.664310575, -0.40660584, -0.131899521, 0.15361169, -0.670097411, -0.794834971, 0.0228863657, -0.753837466, -0.50319159, -0.144800603, -0.171272889, -0.806975782, -0.538401663, 0.815371573, 0.498376608, -0.410287172, -0.071450077, -0.5993011, -0.105997548, 0.0634727329, 0.144404054, -0.78970027, -0.537903726, -0.810344875, 0.547044933, -0.0731045231, 0.155906379, 0.559961498, -0.554831266, 0.0948560238, -0.0790507644, -0.6320889, -0.0859265476, -0.430345327, -0.382865727, 0.487086982, -0.425913572, 0.513455987, -0.110053286, -0.290440619, 0.106850773, 0.652535856, 0.0109406114, -0.137107894, -0.57162261, 0.633475184, -0.49240616, 0.0250977576, 0.0285135061, 0.0169690773, 0.653509021, 0.483197391, -0.51222676, -0.151969165, 0.565636218, -0.569306076, 0.0835313201, 0.0990638435, -0.519652009, -0.446549684, 0.55386138, 0.448214024, -0.0644896403, -0.0720341578, 0.108946741, -0.198243439, -0.515864074, 0.0362923592, -0.128786445, 0.39521724, 0.149344534, -0.701411724, -0.0392639488, 0.0790284425, 0.0872871578, 0.648983777, -0.71551162, -0.547274411, 0.47679767, -0.539834619, 0.457414448, 0.114965558, 0.607790053, 0.000513345003, -0.15862602, -0.133385301, -0.0484945923, 0.45784691, 0.538715899, 0.591025174, 0.4980115, 0.612751007, -0.330444664, 0.0633429885, 0.0478636324, -0.0816067979, 0.0906186998, -0.069659844, 0.0245619714, 0.0629294813, 0.11503616, -0.127734646, 0.0248081982, -0.0854954123, -0.0427704975, 0.153739035, -0.0753483102, 0.056936428, 0.0730580091, 0.0647097081, -0.0245947093, 0.0785699487, -0.154720873, -0.0970023721, -0.136104912, 0.0217498988, -0.00194321573, 0.0605532974, 0.0544321686, 0.0432703048, 0.0677633733, -0.158481121, 0.116616905, -0.0726224259, 0.0625041276, 0.0777515769, -0.00548809767, -0.018487826, -0.160460278, -0.054911457, 0.0180923194, -0.0210434645, 0.0419075936, -0.019303903, 0.046921134, 0.0313011557, -0.0415977761, 0.157840312, -0.0598788708, -0.0556366891, -0.110885054, 0.0175383836, 0.0952107012, -0.107919112, 0.0358991623, 0.0492685288, 0.046242103, -0.0062815398, 0.0813554227, -0.0320968479, -0.153601304, 0.161983699, 0.0796003342, -0.0262238085, 0.132196397, 0.133015186, 0.115734339, 0.0785996914, 0.0534717143, 0.0838688016, -0.0398067385, 0.0439830571, 0.0130348057, -0.0977161303, 0.118602931, 0.126940459, -0.106975943, -0.00951477885, -0.091458708, -0.0801269487, -0.0263103247, 0.0140517205, 0.113654554, -0.162440941, 0.016832158, 0.111492127, -0.0812570155, 0.0569194853, -0.0851391926, 0.0359783322, -0.0325656086, -0.10187836, 0.0287739187, -0.00210155547, -0.0120766908, 0.0916896164, -0.0260320753, 0.151476949, -0.0111931562, 0.0437888317, 0.28489542, -0.0559758916, 0.465931833, -0.463729143, 0.087120235, -0.148486435, -0.341843337, -0.490698814, 0.0225778669, -0.665469229, -0.308908492, 0.0079113543, -0.00376867643, -0.744289994, -0.636592388, 0.592644274, 0.402315497, -0.294979662, 0.147730082, -0.561049223, -0.0700448528, -0.120201796, 0.074372679, -0.566724122, -0.412927359, -0.700030982, 0.576705277, -0.047411114, -0.101848476, 0.33052963, -0.52353251, -0.0605568513, -0.0987362787, -0.598086953, -0.105469838, -0.602784157, -0.402369857, 0.456329018, -0.302669674, 0.628839195, -0.136393115, -0.525435746, -0.0802344456, 0.406169444, -0.0156131536, -0.0607768074, -0.745603919, 0.600795031, -0.621863723, -0.0576748848, -0.0739627108, -0.0343489386, 0.383514315, 0.600832939, -0.394926518, 0.0716857016, 0.317405909, -0.554795325, -0.0383089036, -0.03188622, -0.451491356, -0.567595482, 0.805678248, 0.447996467, 0.0610621572, 0.0141366571, -0.0649617091, -0.158469215, -0.453444391, -0.00282855332, -0.0891613811, 0.522305965, -0.139301226, -0.749600589, 0.106357515, 0.0332240313, 0.0198154896, 0.436969399, -0.588302195, -0.542488337, 0.580874205, -0.670159638, 0.427499175, -0.0779737607, 0.494628429, -0.0684950426, -0.0484847948, 0.0581934303, -0.0957432985, 0.341008037, 0.41196987, 0.636635542, 0.331543803, 0.637782216, -0.291789949, -0.0219285339, 0.141708553, 0.147915572, -0.0455616266, -0.116015449, 0.128730416, 0.136381954, 0.118148535, -0.0461406857, -0.0859908909, 0.0922756791, -0.046486482, -0.162138343, 0.0578264743, 0.138941288, 0.0983988643, -0.0634187236, 0.131013304, -0.144170031, -0.00460401177, -0.110742629, 0.102249146, 0.14183858, 0.0570673794, 0.0760297626, 0.144005418, -0.1019134, -0.135117501, 0.0988574922, -0.146373555, 0.0484071076, 0.129275411, -0.0648685247, 0.109079093, 0.092903465, 0.0875290334, 0.0821627527, 0.0400577933, 0.131807089, 0.0926982164, 0.0748465061, -0.102631956, 0.128583759, -0.0478909463, 0.0721225739, -0.0192542672, 0.117644817, -0.0638892725, -0.0383490473, -0.133238122, 0.0774132013, 0.15754208, -0.058579959, -0.0284232348, -0.10272003, -0.14537479, 0.0937844515, 0.0943775177, -0.0467606783, 0.0165154636, -0.0395936072, 0.0463791788, 0.0782236457, 0.10819304, -0.132041946, 0.125683188, -0.00266599655, 0.110281646, 0.131759375, 0.0128004104, -0.136597112, 0.0254746974, 0.0245522559, 0.0709870011, -0.0161857009, 0.135923654, 0.080018118, -0.119462088, 0.0183110982, -0.0249598622, -0.069484368, -0.0728697404, 0.101434618, 0.0643271506, -0.135969162, -0.0447710305, -0.161402419, 0.0465058833, -0.0512671843, 0.0459613502, 0.0268547684, 0.127304405, 0.163579553, 0.0595384985, -0.000113010406, -0.130348891, 0.0503328666, 0.375250161, -0.0564936176, 0.302692056, -0.19715254, -0.0569530427, -0.117529064, -0.136596143, -0.338833302, -0.0733796135, -0.278026968, -0.267448455, 0.104435734, 0.124707699, -0.260120779, -0.527209818, 0.494568408, 0.264729232, -0.111618727, -0.0575552285, -0.488135993, -0.0393007249, -0.146112576, -0.0535632819, -0.349757135, -0.199360996, -0.213421702, 0.305386066, -0.109520003, 0.0877522528, 0.381479502, -0.301432967, -0.0645133629, 0.0213819295, -0.420290262, 0.0836887211, -0.409564167, -0.147765741, 0.26368016, -0.182855934, 0.338299483, -0.125336722, -0.318842828, -0.0468919426, 0.510945916, 0.149190426, 0.0379741043, -0.477670908, 0.365644127, -0.393774331, -0.0996051878, 0.016202949, -0.166504771, 0.344896346, 0.42374298, -0.291637212, -0.144153535, 0.487658083, -0.429527164, -0.0753854215, 0.058832936, -0.352586538, -0.246949509, 0.640125155, 0.315155268, 0.000840380788, 0.0650290996, 0.00279921293, -0.085950166, -0.109702334, -0.115320005, -0.022042729, 0.33425051, -0.105680153, -0.35921216, -0.0682788864, -0.101727784, -0.0590116456, 0.353024542, -0.563083589, -0.0884778053, 0.391844839, -0.539848745, 0.27150932, -0.0919802934, 0.345882803, -0.111236081, 0.0926810429, 0.00275398791, 0.0237689316, 0.141124532, 0.367899001, 0.223004937, 0.342999607, 0.427729994, -0.0563706271, 0.112616539, -0.0385980457, 0.0185367614, -0.0448516086, 0.0826865286, -0.14224188, -0.159731403, -0.0195692331, 0.149634689, 0.00944805145, 0.152616501, -0.160841808, -0.122676469, 0.12757349, 0.0606708676, 0.142268062, -0.163467616, -0.0667494684, 0.0316374302, -0.043245919, -0.132333189, -0.0296333432, -0.0417868271, 0.100532204, -0.0620630011, -0.00514909625, -0.0989871025, -0.095368512, -0.0835502446, -0.0224133134, 0.108457625, 0.132040471, 0.0521520078, 0.0348580927, -0.0590357184, -0.100558415, -0.136832878, -0.101383775, 0.142769724, 0.112205118, -0.0187974125, 0.0119803548, -0.0175860971, -0.00242608786, 0.134173393, -0.0402145013, -0.118409082, 0.133866042, -0.114783771, -0.00724539161, 0.137954712, -0.0289792866, 0.0443437248, 0.0471954048, 0.0967945457, -0.0400497541, 0.0578964055, 0.115920126, -0.0748741776, 0.146988064, 0.150347441, 0.00589601696, 0.132452369, -0.014718771, -0.134253979, 0.044315502, 0.00439803302, -0.0167531669, -0.120916769, 0.132174432, 0.105356872, -0.135500997, 0.106760442, -0.0723429993, -0.12721166, 0.153713912, 0.0988725722, 0.129809558, 0.0186032057, 0.0897754729, -0.0828637555, 0.0463591963, 0.0163919181, 0.0163021386, -0.10156405, 0.0196555555, 0.0925357342, -0.0393088385, -0.0122584552, -0.00292657316, 0.0751423985, 0.0273545086, 0.0428062379, 0.0338970274, -0.00992292166, -0.053788878, 0.11162287, 0.286859989, -0.0357380062, 0.609294713, -0.411515683, 0.15647909, 0.142120957, -0.47610867, -0.54255271, -0.0284564048, -0.567184687, -0.486063093, -0.0387216583, 0.0554273166, -0.461258203, -0.592238665, 0.772567928, 0.521580756, -0.220841631, 0.0394986458, -0.55406636, 0.00442413986, 0.0589080006, 0.0139624774, -0.466613799, -0.254308671, -0.620412827, 0.563562691, -0.00233466923, 0.0419659913, 0.548646152, -0.584581614, 0.158229619, -0.056298323, -0.434417427, -0.151067242, -0.537316918, -0.555012465, 0.504357517, -0.223498568, 0.373282194, -0.0968519896, -0.469088614, -0.102262825, 0.643966615, -0.0385146886, 0.163557559, -0.682493329, 0.70912677, -0.51372081, 0.154046535, -0.0680202246, -0.174102694, 0.336427838, 0.577760816, -0.314038903, -0.0196849704, 0.583641708, -0.649650037, 0.163640857, -0.0640283749, -0.478707552, -0.61454165, 0.611967444, 0.48430568, -0.146429822, 0.000623777509, 0.0175122023, -0.198100418, -0.501747906, 0.0776187927, -0.011092335, 0.45746699, 0.0517713949, -0.486038685, -0.0853327066, 0.0845993012, 0.142949671, 0.516857445, -0.58640039, -0.304828078, 0.482333809, -0.521633863, 0.482619047, 0.135394335, 0.419143081, 0.0475963801, -0.0312981904, -0.0242736191, -0.0331758112, 0.212874725, 0.244892642, 0.497143477, 0.275314152, 0.640861928, -0.229501531, 0.095325321, 0.143483281, 0.076053679, -0.0885042325, -0.0661684126, 0.0922647417, -0.0770055503, 0.0274118632, 0.128228724, 0.153101385, -0.083956331, -0.15904367, 0.119567543, 0.125558734, 0.0556707531, 0.00787755847, 0.127062649, 0.0554860681, -0.111388646, 0.0222603977, -0.0902488381, -0.114971891, 0.0774939656, 0.00238199532, -0.0153052807, -0.00812704861, 0.0620803684, 0.00618925691, 0.137832642, 0.0504140854, 0.0324838609, -0.084137544, -0.0370414406, -0.112767704, 0.158515662, 0.155168414, 0.102624387, 0.0161525309, -0.0468471125, 0.140682071, -0.0403754637, 0.0272016227, -0.149111301, -0.0241065323, 0.0569703728, 0.098033756, 0.131118894, -0.108851224, 0.0753597468, 0.151129752, 0.0428200066, 0.0737956911, 0.00973987579, -0.0393396616, 0.0456132144, 0.125754625, -0.0443908572, 0.0740742534, -0.132125407, -0.139346763, 0.0322488844, -0.077892676, -0.113379627, -0.160263687, 0.086107403, 0.123270541, -0.10032215, -0.0493220985, -0.00889088213, 0.124768049, 0.142044038, 0.0846117586, 0.134811938, -0.155033514, -0.0329990089, -0.0894454494, 0.067272529, -0.0690529197, -0.106234834, 0.161034405, 0.149611831, 0.095339179, 0.160713285, -0.0152688026, -0.115550876, 0.159216642, -0.106235459, 0.144958436, -0.0491170436, 0.0154130906, 0.0386286676, 0.0117719024, 0.0838084817, 0.064068377, -0.161019206, 0.160186738, -0.172268942, 0.533779323, 0.0207956135, 0.667862177, -0.327755451, -0.0113181472, 0.032315135, -0.424538404, -0.684215784, -0.142610312, -0.473788679, -0.397987634, -0.109086797, -0.117940031, -0.586033762, -0.589366198, 0.809207976, 0.526101708, -0.452961713, 0.0863121748, -0.846322536, -0.0562290624, -0.133094609, 0.0637094975, -0.749593079, -0.532095969, -0.577949524, 0.608543158, -0.0566149279, 0.0425800085, 0.427210391, -0.47769469, -0.00117467344, -0.14372474, -0.667633295, -0.10076905, -0.482318223, -0.573654592, 0.623889565, -0.353755951, 0.634499669, 0.0118949413, -0.497158498, -0.0608907863, 0.640300989, -0.162745893, 0.03825517, -0.659903705, 0.567361116, -0.5714854, -0.111586049, -0.0321406946, -0.0118061677, 0.503429532, 0.327712625, -0.443685025, 0.0724555701, 0.723296642, -0.56720376, -0.131573901, 0.111232847, -0.468566656, -0.687999964, 0.607026279, 0.414428055, 0.113355339, 0.124037802, 0.0684210658, -0.20253171, -0.643614113, -0.104998745, -0.0992261469, 0.337527364, -0.10812588, -0.755333364, 0.0732733011, -0.00914275646, 0.024262771, 0.643807828, -0.503936231, -0.48651278, 0.717816532, -0.544827521, 0.512758076, -0.0277692527, 0.582044303, 0.0586120337, -0.0218767021, -0.0681503341, -0.0587955117, 0.454771549, 0.514890373, 0.375687778, 0.543844044, 0.768497825, -0.343580186, 0.143430442, 0.119612262, -0.0208224952, 0.0229425132, -0.0589544587, -0.0669005513, -0.00874778628, -0.0578448772, -0.1257613, 0.0660459697, -0.105283193, -0.0548858978, 0.0649599582, -0.107908644, -0.107327923, 0.0753218979, 0.0329284705, 0.0823225901, -0.103100866, -0.0954225808, -0.134608477, -0.0424488857, 0.15616706, -0.125207216, 0.0365718529, -0.114411235, 0.0753771439, 0.102282077, 0.030843094, 0.029556036, -0.0293676201, -0.13666901, -0.0664778054, -0.106843904, 0.0202000439, -0.139663532, 0.137247473, 0.0616394803, 0.0687653795, 0.136460513, -0.00583777623, -0.0348427594, -0.150973514, -0.117349327, 0.110115826, -0.0271724761, 0.0359578431, -0.116807058, -0.0719165578, -0.00469906628, 0.136935502, 0.0530858263, -0.148500398, -0.070095107, -0.0806360915, 0.142110422, 0.00256738067, -0.120746508, 0.143997222, -0.0649938211, 0.0369416624, 0.0838904232, -0.0202637706, -0.0361969844, -0.142330468, -0.154804647, 0.0754343867, 0.157088041, 0.0986117348, 0.00526530202, -0.120730713, 0.035393998, 0.143105209, -0.129418492, -0.0947114825, -0.109653153, -0.0258620232, -0.0408343822, 0.0078516379, 0.0411707312, 0.0689083934, -0.0703557432, -0.140870243, -0.109314702, 0.118847132, -0.0758976266, -0.125829116, 0.127197295, 0.137463987, -0.114384554, 0.139589235, 0.150440067, 0.180206478, -0.127316907, -0.145665854, -0.06194482, 0.0596955344, 0.429596394, -0.040304482, 0.461228102, -0.224525094, -0.0463400781, -0.0963862389, -0.498867273, -0.396922916, 0.12892586, -0.373993456, -0.352641553, -0.00451430678, 0.102671325, -0.490256935, -0.45638153, 0.629544735, 0.53008157, -0.277163655, 0.145139813, -0.74016118, -0.0342291296, 0.0925118923, 0.0170095414, -0.636625171, -0.18469578, -0.649915874, 0.642586768, -0.0191352069, 0.078931503, 0.525222063, -0.435780257, -0.0115135908, -0.0928486884, -0.780524194, 0.112244129, -0.5725528, -0.464159459, 0.439511329, -0.189455599, 0.540933132, -0.0249120295, -0.296746433, -0.110864177, 0.342180222, -0.102790624, 0.0731332451, -0.79270643, 0.461214572, -0.42133826, 0.162384808, 0.114454783, 0.116161741, 0.290338576, 0.308036834, -0.314717025, 0.105206728, 0.409908891, -0.592649281, -0.0964998677, 0.0581368059, -0.496952087, -0.42098394, 0.449741066, 0.484095663, 0.0679054856, -0.0864579678, -0.14294897, -0.176799446, -0.368165582, 0.117009133, -0.064208068, 0.410696387, -0.156865478, -0.507613182, -0.118181139, 0.000782132149, 0.00910587609, 0.36084646, -0.736773312, -0.439464629, 0.656639457, -0.822452188, 0.282432616, -0.0936930925, 0.482744098, -0.0161796957, -0.155828819, -0.12223433, 0.13154608, 0.391385108, 0.182680577, 0.561095774, 0.39329499, 0.540092587, -0.488901258, -0.1403597, -0.0587246493, -0.0753704756, -0.0801390037, -0.131909817, 0.0475846678, 0.0111608058, -0.12557514, 0.130687833, 0.147357345, 0.0895265639, -0.0310648829, -0.143525109, 0.143476456, 0.00316150486, -0.0652911961, 0.146549463, -0.00135888159, -0.000782638788, 0.0992844701, -0.0547906086, -0.0262224078, -0.160285696, 0.0748166591, 0.0398910195, -0.112211466, 0.0729758292, -0.041509904, 0.0760549009, -0.0819133371, -0.107092738, 0.0195774734, 0.000116586685, 0.0790748745, -0.0693661347, 0.0518049598, -0.0713005289, 0.108286411, 0.154044688, 0.0751872361, -0.0181486607, -0.0103325248, -0.073743172, -0.110061362, 0.0582866371, 0.162033409, -0.133738756, 0.0494103581, -0.0254963636, 0.133866727, -0.142346919, 0.119989604, -0.0809465274, -0.0745492503, 0.0713825077, -0.131087944, 0.128722876, 0.118853122, 0.0659968853, -0.14994061, 0.157307178, 0.0591157824, -0.0941369087, 0.139789015, -0.074152492, -0.048956044, -0.153951243, -0.0587975383, 0.127273291, -0.150281802, -0.0789495036, -0.0668480322, -0.0778852254, -0.0108916909, -0.111826375, 0.101335615, 0.000341191888, -0.0744965374, 0.100597054, -0.0969975367, -0.0443735272, -0.133351743, -0.0812312216, -0.132171765, -0.0269654691, -0.0769562274, 0.122293204, 0.0759865344, 0.029773891, -0.0684559047, 0.126707733, -0.0144809783, -0.0417289585, -0.039344579, 0.0700835586, 0.0316174477, -0.130985767, 0.443270981, -0.0539823025, 0.361890972, -0.363300443, -0.163329676, 0.1204454, -0.469485015, -0.479613245, 0.0138033479, -0.498726815, -0.411633074, -0.00491516292, 0.0560840555, -0.461526364, -0.562141538, 0.579076707, 0.288368225, -0.453016341, -0.0500700548, -0.650161982, 0.0749059767, -0.00136087835, -0.132494196, -0.380091727, -0.200003967, -0.526683807, 0.477090091, -0.0922354832, -0.0950897709, 0.555062234, -0.233314842, 0.0753492862, 0.0217465013, -0.616467893, -0.0504830703, -0.248475283, -0.43391335, 0.49960053, -0.0825850815, 0.591431379, 0.0702786297, -0.439005375, -0.0224506259, 0.541580975, -0.126283556, -0.0278686434, -0.588835895, 0.3644467, -0.392906636, -0.010158807, -0.0639783144, -0.153947413, 0.234401166, 0.525299191, -0.382777631, 0.0551414788, 0.340716243, -0.709058344, 0.132799923, 0.0478774905, -0.275504261, -0.555791557, 0.675438404, 0.290268511, 0.157366931, 0.0900330842, -0.0531345457, -0.316160589, -0.418503553, -0.134245202, 0.106508106, 0.308096081, 0.156949833, -0.379094869, 0.134452462, 0.161377728, -0.0571513847, 0.493007928, -0.576906443, -0.247688457, 0.629550755, -0.748694897, 0.229307622, -0.0219348073, 0.502853155, -0.138585091, -0.158090845, -0.0644304082, 0.113238245, 0.404934347, 0.267524868, 0.34378013, 0.453479499, 0.677596152, -0.155852243, 0.0682766885, 0.0651495159, 0.0671535581, 0.0310572684, -0.0764942616, 0.00573396683, -0.129765928, 0.0821889341, 0.0600581318, 0.0225273371, 0.134855956, -0.134547293, 0.117048204, -0.0339456052, -0.137868702, -0.119512543, -0.0883095264, -0.0782756209, 0.157427222, -0.00296777487, -0.111893997, 0.0621184111, -0.137421608, -0.00874532759, -0.15745239, -0.0671554729, -0.037850067, 0.139058918, 0.0984688997, -0.0954215005, -0.0571428388, 0.045945853, -0.110590212, 0.0175374895, -0.14030464, 0.02324754, -0.0421241224, -0.159510091, 0.145609766, 0.104720712, 0.0327236354, -0.0848023295, 0.15117386, 0.112850457, 0.0635820627, 0.121060938, 0.0202223957, 0.0440441519, -0.116166338, -0.0624290854, -0.161891535, 0.136476934, -0.0927184373, -0.0442456231, 0.157305986, 0.0721562952, 0.00208224356, 0.0666362643, 0.119968712, 0.15061757, 0.00976192951, -0.107399397, -0.00308823586, -0.0651116595, -0.0724300146, 0.0870065689, -0.137364924, -0.0823942274, -0.133502096, 0.155025661, 0.0615383685, 0.0644683391, 0.0479668826, 0.0233534425, 0.0347766131, -0.103369758, -0.11687164, 0.071431011, -0.0658613592, -0.121844277, -0.137742862, 0.13508901, -0.158615977, 0.100335091, -0.127653748, 0.121180356, -0.00451360643, -4.7981739e-06, -0.1393511, 0.0787953287, -0.0618465915, -0.0763548464, -0.0871187001, -0.0918320492, 0.142125458, 0.0136672407, -0.109021977, -0.198058099, -0.131038189, -0.195490673, 0.297558874, -0.0523217916, 0.121066831, 0.497835547, 0.337065011, -0.140253395, 0.326755643, 0.261396229, -0.12922436, -0.158674836, 0.276964813, 0.310892016, -0.288321227, -0.234429002, 0.49902004, -0.0019971421, 0.364040345, -0.00859841704, 0.0765295625, 0.108894452, 0.135448024, 0.568538368, 0.324725598, -0.304421276, 0.0320975184, 0.0213848408, -0.462374985, 0.291738778, -0.00347207487, -0.0637619868, 0.124400146, 0.109356925, 0.582001626, 0.544644654, -0.413018614, 0.492009342, -0.416079402, 0.0841503069, 0.564010024, -0.0810130611, -0.149000078, -0.0450075716, -0.0930458978, 0.197242275, -0.30742532, 0.321026444, -0.089274697, 0.0494512878, 0.097775355, -0.419094712, -0.111523539, 0.349818021, -0.0834798887, -0.292802364, 0.331537873, -0.0858734399, 0.11993666, 0.457367063, 0.412163585, -0.363937169, -0.365025401, -0.116449513, -0.022363171, -0.134212032, 0.238970891, 0.253569782, 0.0807862729, 0.0746707693, -0.403924108, -0.0802614763, 0.164183721, 0.0455143265, 0.1136823, 0.0464541763, 0.00322439731, 0.224464953, 0.457054436, -0.0127919922, 0.216530234, -0.0556155667, -0.101662852, -0.225912377, -0.161279619, -0.101869285, -0.143954292, -0.146414414, -0.510854721, -0.286709309, -0.279252827, -0.157098114, -0.152029797, 0.548834085, -0.155345172, 0.0439191014, -0.042681329, 0.0134783834, 0.0543549806, -0.00572164357, -0.0833741426, 0.0383355469, 0.0183691233, 0.0405271649, 0.147274524, -0.129355818, -0.147480011, -0.13689363, -0.111604936, -0.147378415, 0.0365482271, 0.110202789, -0.117573455, -0.0779136717, 0.0926531553, 0.0223676264, -0.0367053598, 0.0823863894, 0.103221804, 0.127338469, -0.162603036, 0.132409751, 0.00949241221, -0.138571501, -0.0106359422, -0.0275547206, 0.121317029, -0.0802596584, -0.0320254415, 0.114836752, -0.00500901043, 0.134781927, 0.000212699175, 0.0430897921, -0.121422589, 0.141032398, 0.00327046216, 0.108806223, -0.0605520532, -0.0578859076, 0.111974448, 0.0040999949, 0.0295784026, 0.152474821, 0.00350083411, -0.0258826166, -0.039329052, 0.00933359563, 0.0837092102, 0.133108884, -0.105187252, 0.121390551, -0.0943282619, -0.104005396, -0.132854119, 0.0770351589, 0.10846293, -0.0587827861, -0.0215115994, -0.137577578, -0.161529943, -0.112005517, 0.052903235, -0.0329349786, 0.148083866, -0.0371851921, 0.154467374, -0.0183540583, -0.0982050225, -0.00175713003, 0.0203277171, -0.027044028, 0.0521603674, -0.111326873, -0.114216179, -0.128956139, -0.0165171027, -0.0231119394, -0.103463367, 0.119867474, -0.121384464, 0.151464075, 0.0497992039, -0.00840507448, -0.0974707305, 0.158106059, -0.0540469959, 0.0990505219, 0.0175169557, 0.124720305, -0.0267386883, 0.0359646939, 0.0721528083, 0.0266801156, 0.345639259, -0.000464260578, -0.0303840321, 0.300714403, -0.0816367418, -0.12997742, -0.0109285135, 0.373247713, -0.11001116, -0.172555879, 0.179113746, 0.0333056599, 0.225725591, 0.192783251, 0.306283414, -0.10961698, 0.120423622, 0.00992624462, -0.152191728, -0.106580168, 0.0748748034, 0.088953577, -0.0101088481, 0.029878905, -0.159133807, -0.161174282, -0.0770875141, 0.323459804, -0.0147467405, 0.0259445906, -0.0284927543, 0.135673895, 0.359665662, 0.331357986, -0.0823882148, 0.347884804, -0.0235628802, 0.022381695, 0.410131484, -0.0982122794, 0.129379362, -0.0953466222, 0.109578341, 0.0372427665, 0.0755271763, 0.247905314, -0.1556786, -0.107570864, 0.10056641, -0.121430479, 0.0378915854, 0.332279056, -0.00254507363, 0.239575192, -0.0823266804, -0.151332229, 0.0450440198, 0.273305923, 0.326799393, 0.0589323379, -0.136635676, -0.139624432, -0.130868137, 0.0832932591, 0.179266497, 0.115092449, -0.140426815, -0.139837027, -0.182230502, 0.118175067, 0.0586825646, -0.0614913218, -0.126737207, -0.0639282092, 0.160274655, 0.0860009566, 0.236531273, 0.233578801, 0.167818636, 0.27385354, 0.0395541191, 0.178455696, -0.0326292068, -0.0539216362, 0.0986862183, -0.00362370908, -0.0719124451, 0.208243817, 0.114058159, 0.138222709, 0.168737933, 0.138840169, 0.102649122, 0.059117198, -0.157170817, -0.0358595103, -0.11643219, 0.0333441794, 0.161783367, -0.000422552228, 0.125288963, -0.072627306, -0.0231248885, 0.0250298232, 0.105993927, -0.149125472, 0.0557491034, -0.0802814662, -0.0596189573, -0.0894960165, 0.0757104605, 0.133332223, 0.0583767742, -0.0314468145, -0.0230498165, 0.059897244, 0.116782397, 0.118875325, 0.105525047, 0.152943105, 0.0806157142, -0.018586427, 0.0807473361, -0.140097439, 0.0605539978, -0.160223261, 0.00815546513, -0.0224062949, 0.0183072388, -0.140713453, 0.12905854, -0.119064115, -0.110908225, 0.153741747, -0.125838295, 0.0165252537, 0.0573668182, -0.137209073, 0.0130067468, 0.0156047642, 0.0777211487, 0.135009408, -0.0239736289, -0.143850535, 0.0834618956, 0.162123919, -0.0995615274, 0.0951184332, -0.0829925239, -0.0470131785, -0.155363664, -0.110882476, 0.0433360934, 0.150553942, 0.0585212708, -0.0261256397, -0.121727377, 0.0107326359, 0.0840308219, 0.0395815969, 0.0550657511, 0.132816076, 0.0255072117, 0.147922367, -0.000366672873, 0.102769434, -0.127750054, -0.154732198, -0.0529250875, 0.0141885132, 0.0808088332, -0.146736488, -0.0621336251, 0.132529557, -0.0418293998, 0.102083176, 0.0669139028, 0.075059399, 0.122381359, 0.0218984038, 0.108590662, 0.0654821247, 0.0483045578, 0.126004249, 0.148006916, 0.119236141, 0.156065315, 0.0639064759, -0.128038526, -0.119234249, -0.159682393, 0.0830700547, 0.15530315, -0.0311823338, 0.0374294668, -0.148635417, 0.0441427231, 0.0593574345, -0.0673493296, -0.160656735, -0.138513595, 0.0767943263, -0.0385484099, -0.0373497456, -0.15639326, -0.137173593, -0.0586581975, 0.139909446, 0.150342077, -0.0341482013, 0.0519726425, -0.0881596431, -0.0631534234, 0.0577089489, 0.162802517, -0.0488040596, -0.142477766, 0.100804627, -0.118299976, 0.0784850419, 0.155373812, 0.0361293852, -0.0566727221, 0.124344587, -0.132140547, 0.0554906428, 0.00426918268, 0.0962924659, 0.0754590929, 0.0675136447, -0.00398799777, -0.0646605492, 0.124678493, 0.000232174993, 0.157871544, -0.132603765, 0.160627306, 0.070615992, -0.0797000229, -0.147520751, -0.117849961, -0.0335112214, 0.146458656, 0.123430878, 0.102703094, 0.131458551, -0.006874457, 0.100774109, 0.0912412703, 0.017995581, -0.0206750035, 0.0975280106, -0.0100311339, -0.10461884, 0.0157497972, 0.110805631, -0.0451100767, -0.147696033, 0.150593311, 0.145387322, -0.00109639764, 0.103600562, 0.0723435879, 0.0549032241, 0.0939267874, 0.111613899, 0.0295619369, 0.0971619189, -0.0261805803, 0.124614835, -0.134735286, 0.042969346, 0.0557344705, -0.110359684, -0.0114464462, -0.05037947, -0.0943442211, 0.0287796557, -0.0259566009, 0.135300666, 0.063625887, -0.133952856, 0.157382846, -0.0383099169, 0.0372920632, -0.014648959, 0.10090968, 0.032406956, 0.0138688982, -0.109510168, 0.101833522, 0.0126260966, -0.0110776126, -0.104517624, -0.15947552, 0.061394304, -0.16039452, 0.0409538597, 0.0259913653, 0.121440232, -0.107146859, 0.0763221085, 0.096506238, 0.152134687, 0.095012337, -0.0685589984, 0.0935745835, 0.0708169192, -0.12570563, 0.141299695, 0.0227600485, -0.0713248029, -0.095150426, -0.148627341, -0.151661798, 0.060960561, -0.106167793, -0.0271804333, -0.0603089556, 0.112869173, -0.0444020927, 0.0647668839, -0.0181653649, 0.150014848, -0.112447977, 0.0347279608, -0.0887000039, 0.082597062, 0.130681038, -0.137554437, 0.0423372537, 0.0598919392, 0.092202127, -0.112948522, 0.0451487899, -0.0680088475, -0.0662727952, -0.071218431, -0.107761428, 0.078756243, 0.140598953, 0.151240736, -0.119028255, -0.0216255337, 0.0923928618, 0.144822955, -0.0766503438, -0.125935018, -0.0555256009, -0.111566931, -0.147606373, 0.0588800609, -0.0264238715, 0.104606718, -0.1535777, -0.0681323856, -0.0185834318, 0.0536869615, -0.0908887759, -0.0857664868, 0.0897387564, 0.0567321926, -0.1583637, 0.0420223624, 0.0341514349, 0.143909603, -0.137840346, -0.127124161, -0.086690411, -0.0560578778, 0.082620278, -0.137349889, 0.0890271366, 0.0576932281, -0.111131459, -0.145361289, 0.0567848235, -0.118651822, 0.136636406, 0.105677903, 0.0965199322, 0.366979212, -0.159805, 0.591868162, -0.309316784, 0.10565716, -0.0828318372, -0.552903056, -0.670090854, -0.0958844349, -0.684641302, -0.451589614, 0.0989465714, -0.129313618, -0.668335915, -0.612732649, 0.674037099, 0.585167885, -0.465203255, 0.0956034213, -0.677537382, 0.064490065, 0.126039743, -0.154063389, -0.718903661, -0.491585314, -0.584867001, 0.643716812, -0.129321724, 0.0853395909, 0.390318185, -0.584425926, 0.0177175701, -0.0815148205, -0.900959671, 0.0843823552, -0.476634741, -0.541543305, 0.663437843, -0.437237084, 0.45236063, 0.147178471, -0.597239614, 0.125269443, 0.478571326, 0.0924565196, -0.145116434, -0.686861575, 0.611978233, -0.548813939, -0.016938597, 0.0771096274, -0.00988470949, 0.60533762, 0.582346499, -0.40086019, 0.0313683003, 0.446622342, -0.704038143, -0.0328734368, -0.160054505, -0.571746111, -0.364253461, 0.539652169, 0.358666629, 0.116393089, -0.0886342525, 0.0805952698, -0.218607232, -0.414840728, 0.123056293, -0.0659081042, 0.374852479, 0.0479542762, -0.602365255, -0.0826311484, 0.0373556316, -0.128500029, 0.361640543, -0.825604975, -0.516779125, 0.535904944, -0.842159688, 0.352114409, 0.0608875155, 0.550810397, -0.0473180115, -0.0276286602, 0.00968845189, -0.154276043, 0.531933248, 0.299749941, 0.593912959, 0.454191059, 0.687884927, -0.414370596, -0.0839598402, 0.101980835, -0.0667863414, 0.0311347246, -0.0319339037, -0.1628066, -0.112477317, -0.00953990221, 0.103580266, -0.14286913, 0.0385582, 0.0169924796, 0.0500077307, 0.0302406102, -0.010894224, -0.0916189253, 0.0832256675, 0.0105787069, 0.0952459574, 0.002256006, -0.085468173, 0.130231231, -0.0190279037, 0.110951453, 0.050534144, -0.0470464304, 0.0555843711, -0.0201450288, 0.0427593291, 0.0803755522, -0.0746829733, 0.0374078006, -0.110040024, -0.0405577272, 0.0139813572, -0.0960411057, 0.0983247757, 0.091606617, -0.0918946415, 0.0949996412, 0.101967782, 0.0402811915, -0.13712962, -0.0568392575, 0.096350342, 0.0725376755, 0.084889695, 0.149472624, -0.162636518, -0.150049984, -0.041048564, -0.134644926, 0.104585707, 0.0282340646, -0.0112650692, -0.0100469291, -0.153979018, -0.0967262238, 0.0210875571, 0.0857957155, 0.100003898, 0.0371995121, 0.0588918477, -0.0797886029, -0.0846435577, -0.01554057, 0.112514317, -0.0554869324, 0.00155636668, -0.0210719556, -0.0221097022, -0.116172552, -0.154021904, -0.135038599, 0.120178759, -0.150358438, 0.124153703, 0.146567613, -0.0099029094, -0.0146910697, -0.122258946, 0.0341661423, 0.111105323, 0.0934411287, 0.121225029, -0.0771883577, -0.00605081022, -0.018688783, -0.110849932, 0.0479205549, 0.123921722, 0.00295157731, -0.108215317, 0.142806888, 0.0804552287, -0.148575485, 0.0787924528, 0.133483738, 0.0653546453, -0.10935697, 0.0227946192, 0.0435341597, 0.0218579024, -0.160159856, -0.106370464, -0.153127015, 0.046511963, 0.113976598, -0.0266286582, 0.00960974395, 0.144647866, -0.104476884, -0.00153023005, 0.0366762131, -0.0702421069, -0.139834166, -0.0828964189, 0.0899285078, -0.0231033117, -0.0747282431, 0.0981351733, -0.0103534013, 0.1611799, 0.0694469064, 0.108739823, -0.096300669, 0.100393444, -0.0914660767, 0.0376040041, 0.0458742976, 0.0739511847, -0.0697474033, -0.0594112873, 0.0881286561, -0.138204992, -0.163079903, -0.0398469269, -0.0939138308, -0.159009144, -0.0619145632, 0.149995327, 0.12875995, 0.0873259902, 0.0899540484, 0.0759403259, 0.00076764822, -0.0550867766, -0.060861446, -0.00131358206, 0.101475477, -0.0765179098, 0.0207495689, 0.0261558741, -0.0872231945, 0.13897568, -0.128655329, -0.14683415, -0.033559218, -0.0630501732, -0.0828337893, 0.0720491409, 0.00131416321, -0.0159976631, -0.0134833008, -0.0651347637, 0.0168139338, -0.0602552593, 0.0989223421, -0.0598443002, 0.127578259, 0.11455664, -0.0213681608, -0.144386873, -0.161703348, 0.0469059199, -0.0196954757, 0.0289658606, 0.105748832, 0.0850627869, -0.114843942, 0.10807842, -0.0862904117, -0.0998614356, 0.0421211571, 0.156542391, -0.0287993252, 0.154750615, -0.0727792084, 0.0656296164, -0.108356133, 0.03519921, 0.0316959918, 0.112392575, -0.0213551223, -0.162938103, -0.111852445, -0.0496560335, 0.155333489, -0.0170349479, 0.0830459893, -0.0475384742, -0.0792633891, 0.0374832302, -0.0528744757, 0.113499612, 0.0507027507, -0.056821309, -0.0187657624, 0.105995327, 0.15777868, -0.00681558251, -0.0946575999, 0.114332348, 0.155010462, -0.00671795011, 0.0608242154, -0.118855312, -0.128274456, 0.094727844, 0.0675797462, 0.0817165226, -0.0987315252, 0.141097188, 0.0814061165, -0.0333934575, 0.00480532646, -0.0735385492, -0.0617220774, -0.0593319237, -0.100604348, 0.106239438, 0.151611537, 0.0657162815, -0.137690306, 0.0905378759, -0.10086637, -0.0682336465, -0.106367268, 0.154383421, -0.0422126949, -0.0513846725, -0.0768632442, -0.0483663678, -0.142264128, -0.000134855509, 0.0894100666, 0.154009223, 0.109260708, 0.000231668353, -0.157152906, -0.0347710401, 0.129166782, -0.0879465565, 0.13964811, -0.0632168353, -0.159505904, 0.00968042016, -0.151761845, -0.0793759227, 0.135874689, 0.027664572, 0.062231794, 0.0226994604, -0.125483125, -0.0678517148, 0.107348591, 0.0575175881, -0.119363636, -0.137304977, 0.146208733, -0.147234306, -0.0536325648, 0.130470455, 0.116213948, -0.0176331997, -0.150563955, 0.089610815, 0.127705336, 0.143950671, 0.100148171, -0.0856718644, -0.138781786, 0.0115007907, -0.11264237, -0.0358800441, -0.0608763918, 0.00248213112, 0.0114322752, 0.11088568, 0.0416771024, 0.156816691, 0.125182092, 0.0733486414, -0.146360993, -0.161242127, 0.096958369, 0.126698017, 0.0938361287, 0.00978194177, -0.0552634969, -0.0848976225, -0.0830861777, 0.101703435, 0.048320204, 0.146235496, 0.0987181067, 0.0794364065, -0.127117574, 0.116301894, -0.121517643, 0.147007793, 0.0739795119, -0.0320990831, -0.080012776, -0.129819274, -0.143925264, -0.102363348, -0.0488330573, -0.13891317, 0.116308689, -0.151482299, -0.0373460352, 0.051464349, -0.0671437681, -0.0888069943, 0.00538754463, -0.0179329515, -0.126359135, 0.0427336991, 0.0329946727, 0.0260518491, 0.0246852785, 0.0288423896, 0.0529480278, -0.162076697, 0.0958556831, 0.0437395275, -0.161343768, 0.0660625547, -0.0781575441, 0.119420528, 0.0342773497, 0.0186617076, -0.134706333, 0.162374645, 0.115848899, 0.0783955753, -0.063016966, 0.0285542756, 0.0594349355, 0.128454596, 0.146908998, 0.0146725327, 0.109279007, 0.139724314, -0.154606119, -0.0651643798, -0.147924349, 0.141870528, 0.0566236377, -0.0723303184, -0.0688956678, -0.0953988284, -0.0892778561, -0.00998438895, 0.140004516, -0.138403133, -0.121336386, -0.14124538, -0.0392290056, -0.156311229, 0.0186066478, 0.123637974, 0.140597612, 0.137472779, 0.0987142324, 0.151931673, 0.106431276, 0.0457198918, -0.0945641845, -0.077840507, -0.143344477, 0.0360056013, -0.103137434, 0.0560354739, -0.116182849, -0.020291701, -0.0535030961, -0.0226698369, 0.125092268, -0.00848829746, 0.0610738248, -0.120339535, -0.0634002686, -0.132697731, 0.0929083228, 0.0497631431, 0.0315331221, 0.108042151, -0.124601111, -0.0852937922, -0.0859740376, -0.0591733456, -0.0360203534, -0.0201662034, 0.0327463448, -0.102120057, -0.0902734622, -0.113973707, -0.113877371, -0.0750775114, 0.15590781, -0.0966590717, 0.0641274899, -0.0477756038, 0.159189463, -0.0847013444, -0.015976429, -0.101970181, -0.0360754579, -0.0833040625, -0.128675431, 0.000967204571, 0.12452361, -0.0137724131, 0.052472949, -0.0247370154, 0.160731673, 0.147895694, -0.023585692, -0.0742103606, 0.066429466, 0.108699203, 0.115016282, 0.00913280249, 0.151615828, -0.0408849865, -0.00784166157, -0.0684461147, 0.0501029789, -0.00485752523, -0.14747265, 0.0987522304, 0.0887751877, 0.0356176198, 0.0902802348, -0.0260884911, 0.0932527483, 0.00385470688, -0.0997035578, 0.0596693307, -0.00495298207, 0.0622439682, -0.103032276, -0.0559337139, -0.141635314, 0.135635287, -0.096205458, 0.0797926933, -0.151022166, 0.134229034, 0.0540894121, -0.0130882263, -0.0465265214, 0.108011246, 0.0334777534, 0.0220413357, 0.0441906005, 0.0341357887, 0.0450375825, -0.102616899, 0.0168300867, 0.129836231, -0.0439711511, -0.1631428, -0.140327618, -0.0133825541, -0.0304959267, 0.102105021, 0.109223515, 0.157596022, 0.0424760133, 0.025866434, -0.14363046, 0.0839447826, -0.00702808797, 0.0856500566, 0.0974706113, 0.0411905199, 0.0739976615, -0.098994635, 0.125551879, -0.075891085, 0.134391576, -0.0831373706, -0.150016814, 0.153182894, 0.113226146, 0.0668544322, -0.0937932953, -0.0832801461, -0.122296721, -0.0476440266, 0.122502446, -0.0872083306, -0.0760335922, -0.147510961, -0.156250164, 0.0952301919, -0.0415546969, -0.0963032395, -0.115351088, -0.0120344311, -0.0912762433, 0.0580475628, 0.115711004, -0.0530346185, -0.0901259258, -0.153519943, 0.0317372084, -0.120866857, -0.0906759575, -0.120001927, 0.00179213285, 0.162703633, -0.00967292488, 0.0571701974, -0.0859936997, 0.0947292447, 0.100652456, -0.0490462631, -0.0410071611, 0.0876711905, 0.0642231256, 0.0434615016, -0.157467723, 0.0564225614, -0.104834937, -0.142395854, -0.0269855261, -0.0092010498, -0.0192741603, 0.145421296, 0.153734088, 0.154290944, 0.00844147801, -0.135789707, -0.1490058, 0.0132638067, 0.0775982291, -0.115593404, 0.0571661294, -0.102534726, -0.00456105173, 0.0802254379, 0.116427779, -0.0761071071, 0.0259064585, -0.0217196196, -0.0111827403, -0.0905446485, 0.131847352, -0.155291006, 0.152496338, 0.0766965002, 0.0584231317, -0.0593572482, 0.0288425535, 0.115809113, 0.0470971167, 0.0316260308, -0.123210423, 0.0893628001, -0.0261571705, 0.153539211, 0.125678301, 0.0511402413, 0.309443474, -0.0410209745, 0.445964456, -0.359625578, -0.0904764831, -0.139445871, -0.407372952, -0.499414623, -0.129436523, -0.369349003, -0.222930014, -0.0379773453, 0.027540436, -0.674120545, -0.492138475, 0.523334861, 0.237869754, -0.446797192, -0.0635370091, -0.450644523, 0.0559678227, 0.00991535187, -0.0237967819, -0.563645601, -0.147682622, -0.393336058, 0.641609669, 0.0583105683, 0.0314334109, 0.454124957, -0.388759017, 0.161477655, 0.0840028822, -0.490048409, 0.0370392203, -0.419826031, -0.356802881, 0.532599568, -0.305735588, 0.369892329, -0.0152055025, -0.497555792, -0.125483945, 0.24376823, -0.154752567, -0.15329808, -0.57041049, 0.477470905, -0.337265581, 0.0756777227, 0.102758005, 0.0290173031, 0.513453543, 0.427936137, -0.471153051, -0.060199149, 0.461946398, -0.723814905, 0.0214590728, -0.0620852411, -0.320358276, -0.243344843, 0.568753362, 0.233652547, -0.0664692223, 0.119743079, 0.0966901779, -0.146970004, -0.409434915, -0.0698849335, -0.0276391152, 0.428497791, -0.133351237, -0.618188918, -0.121357717, -0.0110222846, -0.0604976937, 0.444407314, -0.472613662, -0.306672066, 0.419025421, -0.609449208, 0.441865802, -0.0382930636, 0.367543191, 0.0110176504, -0.0977119505, -0.000515893102, -0.0948615968, 0.43166858, 0.456758261, 0.362691075, 0.199984983, 0.73247081, -0.410469204, -0.0500826463, 0.00678436458, 0.076051265, 0.00419035554, -0.075273782, 0.0135698169, 0.0476934314, 0.0130815506, 0.161955059, -0.0255148113, -0.0254456699, -0.158978, -0.160531878, -0.0877384245, -0.0536556989, -0.0989084765, 0.109233826, -0.111181527, -0.00619885325, 0.0296189785, -0.0289089978, 0.159552723, -0.0156824142, 0.161916196, 0.112175375, -0.0390156806, -0.109862953, 0.0766022652, -0.117787056, 0.139306366, 0.153947622, 0.109614968, 0.122255504, -0.0341136605, 0.121012628, -0.0626597777, -0.114562526, -0.0176611841, 0.146118104, -0.115447983, -0.148465171, 0.0994842947, 0.0570782572, 0.122706175, -0.0831273049, -0.00532698631, 0.135909051, 0.148210049, -0.103683367, 0.152936161, 0.113456458, -0.0364342779, 0.00445565581, 0.0283626467, 0.00979864597, -0.034679845, -0.0868891403, -0.118503317, -0.0332165062, -0.12679565, 0.141245067, 0.027341947, -0.118432924, 0.0276024789, -0.0614001602, -0.108914442, -0.158766434, -0.124834843, 0.160843134, 0.0514851213, -0.0766366869, 0.128185183, 0.0217501223, 0.000925049186, 0.0450871736, -0.0931365043, 0.136534452, -0.126440689, 0.0521594286, 0.0254421979, 0.0871620774, -0.156746745, 0.09702456, -0.0395499095, 0.140528142, -0.139346838, 0.0109403431, -0.151589453, -0.0431390032, -0.0110176504, -0.0573284552, -0.0414792672, -0.149166748, 0.0521813184, 0.102638483, 0.114292502, -0.175287291, 0.507310271, 0.145499885, 0.640718222, -0.431651801, -0.0270268917, 0.0974114388, -0.358768851, -0.681254327, 0.0593203008, -0.675242722, -0.294044942, -0.0413634181, 0.0357905589, -0.618607342, -0.67785114, 0.599707246, 0.644103765, -0.448615789, 0.105018906, -0.763976872, 0.0102487504, -0.0453047529, -0.112931363, -0.440053999, -0.425577015, -0.493176043, 0.684021771, -0.0921099186, 0.144310728, 0.477689624, -0.359718174, -0.0742876604, 0.0744303614, -0.516384363, 0.0872224569, -0.321946532, -0.428286523, 0.564672947, -0.366745055, 0.458216041, -0.13321124, -0.522803187, -0.124522485, 0.705768466, -0.0293953866, -0.0446631387, -0.601200938, 0.601401687, -0.620148838, -0.124550618, 0.134968013, 0.108758181, 0.638626456, 0.559719324, -0.304972917, 0.0753992349, 0.670586109, -0.759760082, 0.152544022, -0.0344163477, -0.368279606, -0.580714703, 0.684982598, 0.511205792, 0.0245447606, -0.0283989757, -0.132486314, -0.106720522, -0.533188045, -0.095429644, -0.157350898, 0.361209184, -0.134494558, -0.514968336, 0.0523039512, -0.104569636, 0.147384107, 0.483279437, -0.748663604, -0.407871455, 0.531846941, -0.509758651, 0.428317964, 0.00657755136, 0.38526994, 0.0274642408, 0.0411971174, -0.13891992, 0.115089417, 0.2890625, 0.464041501, 0.537629664, 0.386016846, 0.69347173, -0.288379073, 0.00259512663, 0.153360009, -0.104501389, -0.124651484, -0.0994781777, 0.0342565924, -0.0875080824, -0.0986559018, -0.0327717513, 0.0833479315, -0.00281594694, -0.117249236, -0.0592920855, 0.0637751371, 0.0372549593, -0.0974785015, -0.0978867263, 0.0905888677, 0.0822022408, -0.0533728451, -0.034975931, -0.0581181571, -0.103711769, 0.0761750787, 0.0914187729, 0.0272061974, 0.108920366, -0.0473434478, 0.00286011398, -0.0819454566, -0.0545869246, -0.0272968411, 0.0600103736, -0.0848217607, 0.100141436, 0.0185231417, -0.0492273942, 0.123306692, -0.0477575734, -0.0228613913, 0.0328577459, 0.149354488, -0.102355972, -0.146478444, 0.0882565975, -0.0578210503, -0.0827491581, -0.0141749382, 0.123653859, -0.0747208297, 0.0870402753, -0.0453518108, 0.044588685, -0.159154654, 0.154590636, -0.0531909689, 0.11537981, -0.0682943985, -0.0845522508, -0.0007263273, 0.13022992, -0.132736936, -0.0592299625, -0.146575481, 0.138293713, 0.027850613, 0.0206435025, -0.0495990217, -0.069524169, -0.139569417, -0.0722318739, 0.120699823, -0.136658415, 0.0416600108, 0.037176609, 0.138313621, 0.0537907183, 0.0865195096, 0.0768840015, -0.157129601, -0.0424082279, -0.0557150468, 0.140841722, -0.0492894351, 0.139309496, 0.0526455045, -0.00730262697, 0.0539788753, -0.111365937, -0.0693356618, 0.0169841349, 0.153485686, 0.0697082281, 0.00517641008, 0.0662829429, 0.0297198892, 0.0974073559, 0.0527710095, 0.0542461276, 0.0121014137, 0.0983252972, 0.03839311, -0.0752131045, -0.0583192445, 0.0256708153, -0.0617399514, -0.162323549, 0.134012789, 0.118890554, 0.00273517519, -0.0800314471, 0.0412297696, -0.0571742766, 0.0784918144, -0.0127361417, -0.0994722992, 0.143718079, -0.0675426722, -0.00598713756, 0.0846547633, -0.0600037687, -0.0354444496, 0.0256366432, -0.030177556, -0.0515845418, 0.104366556, -0.00214775815, -0.0498692654, 0.0720154196, 0.0614446104, -0.0786873251, -0.0922366157, -0.138412878, 0.136779994, 0.179302603, -0.133729726, 0.150865316, 0.102304459, -0.15150322, -0.0432793573, 0.0548448004, -0.0175472796, -0.0759298354, -0.0818395913, 0.159195855, -0.0844869763, 0.127749622, 0.0623118468, 0.138545707, -0.0734245181, 0.00545040704, -0.0781268403, 0.140223682, -0.040840786, 0.115423113, 0.00377982855, -0.108167157, 0.0234216172, -0.134580851, -0.0855451301, -0.0865153819, -0.0740812793, -0.030549109, -0.10352096, -0.0662894845, -0.0756704211, 0.0606323481, 0.092569679, 0.150832579, -0.127181888, -0.0580021441, -0.0868376493, -0.134938821, -0.046344921, -0.128015026, -0.0359454304, -0.00955039263, 0.0946386829, -0.0238915198, 0.0673492104, 0.0279185176, 0.0883836821, 0.0428816229, 0.0417820551, 0.14585498, 0.0654753298, 0.108118899, -0.0838340074, -0.135392383, -0.133392319, -0.0725811422, 0.0193491187, -0.168806329, 0.530087411, 0.0406112671, 0.643129289, -0.475254178, 0.0011806041, -0.151397467, -0.412369937, -0.592032373, -0.161963612, -0.360388964, -0.349347144, 0.0538633503, -0.0628043786, -0.479809225, -0.570897639, 0.760729313, 0.383155823, -0.262503356, 0.150528312, -0.621515214, 0.113631099, -0.00338578387, 0.143046618, -0.384876817, -0.296113551, -0.473288178, 0.477635801, -0.00615948439, -0.0573445559, 0.499427468, -0.543975592, -0.151235029, -0.0411666781, -0.519301534, 0.00746612251, -0.323862463, -0.292993277, 0.51971662, -0.0623354502, 0.654080689, 0.157254994, -0.242604136, -0.116682388, 0.5508039, 0.00576280057, -0.132955253, -0.357764959, 0.523423135, -0.391797274, 0.13513124, -0.0902149379, -0.00448856503, 0.540275395, 0.30841133, -0.457743198, -0.120846331, 0.653473258, -0.317180187, -0.110743642, -0.100062959, -0.208966568, -0.35412696, 0.697604895, 0.267000139, 0.0882976651, 0.0859353989, 0.126033753, -0.109840102, -0.349812597, -0.0934672952, 0.00340263662, 0.412219048, -0.0632713363, -0.56117022, -0.169174731, 0.0643895566, 0.151125431, 0.637183845, -0.473790526, -0.208168596, 0.54246366, -0.589235127, 0.638085127, 0.0230967551, 0.421797842, -0.0346478075, 0.0590770878, -0.0905418843, -0.0940413475, 0.332086086, 0.493487746, 0.366049528, 0.646426201, 0.766292214, -0.133262813, 0.051349625, 0.395899981, 0.00388689339, 0.494815379, -0.281581283, 0.0515768975, 0.125198662, -0.266026378, -0.383036941, 0.0100709349, -0.574913204, -0.321213245, -0.1525442, 0.0779309422, -0.598291039, -0.67618829, 0.447915524, 0.293678463, -0.435835302, -0.0936105773, -0.715294778, -0.148454636, -0.107942559, -0.159281746, -0.342858136, -0.249567077, -0.379220247, 0.624188364, 0.00389993191, 0.113193348, 0.420729011, -0.488305628, -0.125710428, -0.119276464, -0.572307408, -0.115350783, -0.536709726, -0.254787117, 0.48124963, -0.190767244, 0.589077473, 0.015547052, -0.331876308, 0.120542526, 0.505546808, 0.0755365491, 0.151749402, -0.584850311, 0.473985374, -0.46886611, 0.0277551711, 0.140559211, 0.0909491628, 0.282177687, 0.29187876, -0.31223321, -0.0719461218, 0.366725892, -0.514394939, 0.0661440194, 0.00924283266, -0.251746356, -0.543293655, 0.654523671, 0.400812119, 0.156397074, 0.140883684, -0.145640835, -0.0929114446, -0.22473228, 0.156979352, 0.0333597064, 0.526512027, -0.142326146, -0.476264447, 0.0180234667, 0.121793121, 0.130113572, 0.456732929, -0.601095021, -0.368622184, 0.32785511, -0.557375312, 0.326730669, -0.136411101, 0.19332467, 0.107854605, -0.148511142, -0.10753499, 0.127788454, 0.185422555, 0.444670141, 0.448104441, 0.261858225, 0.546359897, -0.211134925, -0.0101957982, 0.398396522, -0.0269882679, 0.486129194, -0.524054885, 0.0727696568, -0.118738256, -0.438090384, -0.469442487, -0.00278258324, -0.468992561, -0.583100319, 0.0269657075, -0.0669030473, -0.814213276, -0.504547656, 0.605623543, 0.530114889, -0.260449857, 0.15419656, -0.736406028, 0.00292864442, -0.135944843, 0.0293183625, -0.768488169, -0.495452046, -0.633008897, 0.735788822, -0.028500542, 0.0832792521, 0.630212367, -0.617331326, 0.148983002, 0.0830580741, -0.607211053, 0.00499406457, -0.523331702, -0.471750289, 0.604487598, -0.141686991, 0.471280068, -0.103268117, -0.477256984, 0.043151021, 0.486764938, -0.0526891649, 0.0831881762, -0.718536496, 0.792366803, -0.676878095, -0.113822311, -0.164372757, 0.0626577586, 0.561889887, 0.580988765, -0.573537648, -0.0261766762, 0.428409547, -0.547622681, -0.0791829675, 0.0884450674, -0.366336882, -0.525043964, 0.741204917, 0.426674157, -0.141808748, -0.146373868, -0.015917629, -0.158308223, -0.589035511, 0.0272668749, 0.133654833, 0.361192167, 0.0850632191, -0.678721011, 0.0615904741, -0.0218304694, 0.101252556, 0.651000559, -0.580663681, -0.38956967, 0.549939513, -0.731697917, 0.391068518, 0.126874208, 0.418774664, 0.00719602406, 0.0579656251, 0.00795219839, 0.159683913, 0.383722872, 0.479412884, 0.473163426, 0.529177964, 0.85292536, -0.40756166, 0.0685930699, -0.136739925, 0.0922677517, 0.129282087, 0.0102041066, 0.158997357, -0.0855297893, 0.0311845988, -0.0428866595, 0.0168897808, -0.106866732, -0.13909325, -0.0805881321, 0.0341135859, -0.150936097, 0.121639252, -0.132139146, 0.0987407267, 0.0620809942, -0.00286878645, -0.103712827, 0.0591438115, 0.0411442816, 0.0279308408, 0.122015625, 0.0595818907, -0.156353369, -0.0935732946, 0.0566514134, 0.0325902253, 0.00210338831, 0.0499197394, 0.0718968064, 0.146708459, -0.155467927, -0.0565499589, 0.0719884634, -0.125986919, 0.159107715, 0.00474877656, -0.145661786, -0.124665841, -0.156221405, 0.108644038, 0.117592335, -0.00519475341, 0.00753878057, -0.0557395443, 0.0367338806, 0.028139323, 0.0497469455, -0.162103146, -0.0264572799, -0.0240476131, 0.0175928473, 0.0990706384, -0.0561073571, 0.0856311619, 0.0213924199, -0.0227620751, 0.0389403701, 0.135115117, -0.0453911424, -0.110545494, 0.129325539, 0.0947327018, 0.159509331, 0.0771846175, -0.0242215246, 0.123737007, 0.0832939595, -0.149173588, 0.114168346, -0.157780588, 0.14469409, -0.0783481598, -0.12071573, -0.113739625, -0.162453011, 0.0244588852, 0.156361014, -0.0704952255, -0.159694925, -0.0917142853, -0.137090802, 0.14289692, 0.041899398, 0.14936924, 0.132419586, -0.0325821042, -0.114108101, -0.0276777893, -0.160233051, -0.118044585, 0.0791963488, -0.144054577, 0.0271427818, -0.0217401367, -0.0110936165, 0.202737838, 0.320353329, 0.0400065631, 0.0512734056, 0.281253934, 0.0797522292, -0.137393907, 0.0451838896, 0.345733911, 0.142001897, -0.135361344, 0.0854217261, 0.0524540097, 0.259759128, 0.216498002, 0.3923558, -0.114049412, 0.0122456271, -0.133329511, -0.0725391656, -0.00678158039, 0.126580909, 0.0954810381, 0.143829852, 0.0336655378, -0.081894882, -0.152411312, -0.146954179, 0.287810862, -0.0366004705, -0.0305089951, 0.0418138094, -0.146023124, 0.249957636, 0.259197444, -0.0751675367, 0.326609641, 0.0486662649, -0.0398752466, 0.296301484, -0.0908877179, 0.279924721, -0.105482832, 0.0375565141, 0.0506152511, 0.177911937, 0.270081609, -0.0623320043, -0.00954065379, 0.00429970492, -0.00950819999, 0.0726488009, 0.303632617, -0.0721708834, 0.0783931985, 0.216672555, -0.129633695, -0.126710668, 0.294468433, 0.15697737, 0.263451576, -0.0925969109, -0.0990182459, -0.107685491, 0.102668047, 0.337305516, 0.211583152, 0.0959029868, 0.0353240073, -0.168356106, 0.0670877621, 0.159387246, -0.0154752787, -0.00822967291, -0.0159040838, 0.25072819, -0.0283130296, 0.206127927, 0.255291402, 0.190409914, 0.158475682, -0.0939276442, 0.0387200229, -0.050979957, 0.134874895, -0.0778312981, -0.145023376, 0.0532395802, 0.00979417749, 0.136485144, 0.144414574, 0.116937362, 0.194281086, 0.108338654, -0.00313591957, -0.124966219, -0.150131568, 0.0970275402, -0.0511199236, 0.040860489, 0.0450057387, 0.112365693, 0.0998730958, -0.153620467, 0.0787642002, -0.0468129292, 0.0937750041, -0.0339456797, 0.0815242231, 0.100352347, 0.109116137, -0.151327819, 0.1362167, -0.0983692557, 0.140543491, 0.0566242933, 0.143955231, -0.143135101, 0.0831642896, 0.130589634, -0.158614844, -0.140757188, 0.0859078914, 0.0386551321, 0.158173949, 0.0597891957, 0.0753865093, -0.0432403758, 0.087349236, 0.0729618967, -0.0272989422, -0.0383048058, -0.00840806961, -0.0684592649, 0.0501502603, -0.0734564513, 0.112330407, -0.120182052, 0.144563466, -0.136457816, -0.0890362784, 0.109228492, -0.063772209, -0.0414140671, -0.0281617641, -0.0734562501, 0.156790078, 0.0490309596, -0.0089442879, -0.0754611194, 0.0683722794, 0.152359962, -0.0114639252, 0.00558507442, 0.0681650937, -0.123505808, 0.112213433, 0.0313823074, -0.0307093263, -0.136884928, -0.0653262362, 0.0441680551, 0.148320258, 0.108153164, 0.0154031068, 0.0839119703, -0.149226144, 0.0102346539, 0.110051364, 0.148182124, -0.00468592346, -0.151746541, -0.133229762, -0.0341391414, 0.0275392383, -0.102420628, 0.0219992697, 0.0557424426, -0.153013036, -0.163454145, 0.147724718, 0.122225344, 0.114112616, -0.0749990046, -0.0339612514, 0.0982846618, 0.160975575, -0.0879514739, -0.027687788, -0.040075317, 0.337122709, 0.107447267, 0.640170038, -0.329167187, -0.0782561153, -0.116001979, -0.390516013, -0.408062309, -0.0230023712, -0.344756961, -0.191970453, -0.0982619897, -0.0374863222, -0.677941144, -0.393138319, 0.463380277, 0.542116821, -0.280091047, -0.0900378451, -0.732562482, -0.0660698116, 0.00760039687, -0.0983186513, -0.36917448, -0.199815884, -0.367835581, 0.590327799, 0.0596091598, 0.0875963122, 0.492991835, -0.227184862, 0.0808094889, 0.148977399, -0.444585264, 0.0352514535, -0.356494039, -0.361255109, 0.520882905, -0.233719334, 0.403641045, -0.0699140579, -0.330485076, -0.111756064, 0.451643586, -0.0491847098, 0.0904435515, -0.713424981, 0.637271583, -0.576943457, -0.131233528, 0.050658714, 0.124697693, 0.367391616, 0.472480297, -0.404045999, 0.0101627856, 0.556181908, -0.637078285, -0.163084477, -0.0383832306, -0.300044745, -0.510922074, 0.562109292, 0.413187742, -0.128509164, -0.0564064085, 0.0175370127, -0.0172287393, -0.175369397, 0.0639542192, 0.1058902, 0.313734561, -0.162553921, -0.502674282, -0.0472101085, -0.0159854144, 0.0263384134, 0.300245047, -0.531729043, -0.442276359, 0.453635544, -0.684684515, 0.386095226, 0.116625696, 0.533678293, 0.10686177, 0.0719436184, -0.0362551063, -0.0360603482, 0.3622531, 0.382044673, 0.57828176, 0.354670405, 0.719807088, -0.388015062, -0.174508139, 0.215570286, -0.0529062375, 0.587997556, -0.274947524, 0.147426516, 0.0804440752, -0.304535478, -0.454660237, 0.0439731479, -0.498901427, -0.238230318, -0.0102666914, 0.132998526, -0.464719653, -0.668762863, 0.652952313, 0.414137334, -0.164560154, 0.0550990552, -0.553726614, -0.112812109, -0.122778744, -0.0852179676, -0.565746963, -0.258202195, -0.467502058, 0.572059691, -0.0768992975, 0.0707095638, 0.54078877, -0.448104501, -0.162558943, 0.0321276784, -0.455607891, -0.128493592, -0.456510514, -0.312486023, 0.648222923, -0.161865026, 0.53218621, -0.00764027238, -0.454849929, -0.0451953411, 0.308694005, 0.0343857855, 0.0705213398, -0.601460397, 0.485473126, -0.321680903, 0.0949182808, 0.00787513889, -0.136335582, 0.421144545, 0.385141343, -0.473435849, -0.104788467, 0.52582401, -0.427538633, 0.100839704, -0.0165983438, -0.278423756, -0.413939446, 0.710184216, 0.383353055, -0.0378847569, 0.0809023529, 0.128169835, -0.151743189, -0.289103478, 0.066611968, 0.0934093818, 0.545054197, -0.15806447, -0.497845143, -0.0229860172, -0.0444824323, -0.141557619, 0.327936679, -0.462643296, -0.475876302, 0.403761983, -0.736859441, 0.555431128, -0.00659908354, 0.33542043, 0.0818387717, -0.160694242, 0.0236755461, -0.1533968, 0.398297995, 0.384744167, 0.331441551, 0.402751356, 0.574325919, -0.432564348, -0.0759227723, 0.21706064, -0.00387589633, 0.595609605, -0.16957134, -0.100181989, -0.00945903361, -0.344490319, -0.529660106, 0.00818738341, -0.479003251, -0.129812747, -0.0479281582, -0.168775782, -0.292848498, -0.274457544, 0.49036634, 0.567371368, -0.250275254, -0.151724041, -0.354970723, -0.122710414, -0.163857132, 0.0673733875, -0.368491411, -0.177162036, -0.485425949, 0.602810919, -0.116760544, -0.0111203426, 0.377181858, -0.207599178, 0.0399638712, -0.0879004747, -0.304508209, 0.0691077411, -0.246673048, -0.260217458, 0.582288802, -0.234835148, 0.436360151, -0.0231363978, -0.264080077, -0.132058918, 0.404458582, -0.130737647, 0.0289660543, -0.304377824, 0.668018639, -0.104033113, -0.017525509, 0.0636320934, 0.0609187111, 0.538498819, 0.226304561, -0.207088634, -0.0801743567, 0.495170355, -0.377418458, 0.00442689657, 0.0791558772, -0.084760122, -0.170767263, 0.662046015, 0.317836255, -0.0690529197, 0.0191694796, -0.0940831006, -0.02795678, -0.401670635, -0.155979499, -0.121273443, 0.362218797, -0.0847134963, -0.193296194, 0.0645343363, 0.147687644, -0.154912859, 0.277315527, -0.501701415, -0.254464865, 0.33047539, -0.468411326, 0.451083332, -0.0666101649, 0.502041042, -0.0057362318, 0.0234047901, 0.0615597069, -0.0230766982, 0.178798541, 0.272201389, 0.193953156, 0.523422956, 0.58787322, -0.0762311071, 0.124301597, 0.146508142, -0.0245867968, 0.0490946323, 0.181274444, -0.0463002399, -0.0781106129, 0.254877925, 0.161187053, -0.0924234465, -0.0232587345, 0.111719772, 0.153336734, -0.100928925, -0.0635686293, 0.133363381, 0.200311378, 0.173549443, 0.110425085, -0.00163604121, 0.0115742395, 0.0842915475, -0.086629197, 0.111786924, 0.112823293, 0.234550133, 0.15787448, 0.195090517, 0.00715474784, 0.130857646, -0.100298427, 0.311769009, -0.143178761, 0.103133738, 0.0129326005, 0.0264683794, 0.301859975, 0.356458753, 0.212239712, 0.332933933, 0.00455258274, 0.0237383973, 0.281135976, -0.104026474, 0.249128297, -0.0867572501, -0.163077056, -0.023107715, -0.0466414206, 0.354050308, -0.132886782, 0.101235151, -0.153015211, 0.14476037, 0.00557650113, 0.242924795, -0.138929993, 0.0375652537, 0.125058398, -0.0741051212, 0.00141421182, 0.351935267, 0.32540375, 0.022557836, -0.101481967, -0.0460637361, 0.0761575252, -0.0773790553, 0.27669093, 0.174276769, 0.0963980481, 0.102250092, -0.250503659, 0.0271127075, -0.0766117796, 0.142860278, -0.0988712534, -0.0182005614, 0.173824608, -0.0354685336, 0.326069683, 0.0977501795, -0.00536953844, 0.189159334, -0.123455241, -0.105712011, -0.103039339, 0.138820991, 0.144249767, -0.0986062661, -0.0333374292, 0.00253537344, -0.0127978548, 0.139320791, 0.134012252, 0.378334731, 0.159006089, 0.158631384, -0.0491215289, -0.119058341, 0.151373267, 0.0978735089, -0.135633588, 0.0106204599, 0.1536493, -0.130392283, -0.036535576, -0.0961244926, 0.0741660744, -0.0625309348, -0.0770806223, 0.0163824856, -0.00639404356, 0.0915825069, 0.100205839, 0.12346223, 0.0245793015, 0.151512235, 0.124110103, 0.101939768, 0.0779728591, -0.153700769, -0.0725752115, 0.0262785256, 0.0832325369, 0.0713638961, 0.118414849, -0.0110956132, 0.0532189459, -0.0898631215, -0.0841295794, 0.132030934, 0.145936608, -0.082064271, 0.0247146189, 0.149070531, 0.0442207605, 0.121726424, 0.119324535, 0.0319827944, 0.0127410144, -0.0877777562, -0.049722366, 0.0433338284, 0.0680450201, 0.0709024072, 0.00350956619, -0.0812475756, 0.0194038749, -0.0353440195, 0.0494886041, -0.135520726, -0.135726601, -0.0388039947, 0.0957541168, 0.119312555, -0.111680865, 0.0307031274, -0.0424036235, -0.084837921, -0.129196346, 0.0787917078, -0.0558628514, 0.109969705, 0.119111836, -0.0690820292, 0.0367564708, -0.00851109624, -0.00579847395, -0.0819538459, 0.129984707, -0.118437953, 0.00957283378, -0.148309514, -0.155115411, 0.0160821825, 0.113973528, 0.0600227416, -0.156380221, 0.0118638724, -0.0939336866, 0.0164368302, -0.159813866, 0.0110994726, -0.154618025, 0.0571646541, 0.0965426266, 0.0777838081, -0.0862945095, 0.0870448351, -0.0645615533, -0.0133520067, 0.105862245, 0.630711079, -0.0482766256, 0.582876384, -0.468586981, -0.0930065662, 0.0433471054, -0.632086515, -0.623380303, 0.150847018, -0.458049506, -0.515512288, -0.130552813, 0.12842685, -0.547448397, -0.548324585, 0.651475549, 0.677594602, -0.321426928, -0.148372516, -0.857636094, 0.12027508, -0.139636055, -0.156285748, -0.660622597, -0.340143412, -0.542996168, 0.771724463, -0.117285527, -0.12961939, 0.515686512, -0.633553743, 0.0262765735, -0.0320099145, -0.612082779, -0.0577144846, -0.530255616, -0.602814734, 0.747009516, -0.281968534, 0.429226577, -0.108002335, -0.369228363, -0.0983397961, 0.563722134, -0.0548454374, 0.069581911, -0.565653741, 0.576729715, -0.682845891, -0.0798710883, -0.171374962, -0.131261602, 0.459016383, 0.492421597, -0.42575106, 0.0185760558, 0.534101665, -0.581607759, -0.108211331, -0.0990887955, -0.312394887, -0.386555672, 0.654724061, 0.492949098, -0.0820863917, 0.0125001818, -0.0965857878, -0.0550288111, -0.525408864, 0.157194942, 0.0500186533, 0.439202189, -0.149013907, -0.774572015, 0.0820892155, -0.119983904, -0.0655998066, 0.462346435, -0.553625941, -0.55579263, 0.60715872, -0.72079587, 0.552710772, 0.0245950222, 0.599570632, -0.161135942, 0.138237879, -0.047213085, -0.146563828, 0.336478353, 0.588278234, 0.591952503, 0.549817085, 0.65846318, -0.350836992, -0.121515155, -0.110477298, 0.0122210383, 0.201217785, 0.395042509, -0.104612797, -0.083784923, 0.0757881626, 0.20623751, -0.130482346, -0.0672471523, 0.37774393, 0.0587109923, -0.100154921, -0.0529181957, 0.114344984, -0.0643938631, 0.0425152443, 0.271492839, 0.00219953689, 0.133931518, -0.00557613373, 0.00475039706, -0.125167385, 0.191803291, 0.354961276, -0.023218561, -0.0377069525, -0.115602538, -0.00906254444, -0.0770430937, 0.313838035, 0.0363580436, -0.021689415, 0.0965251252, 0.135844037, 0.301656395, 0.391370624, -0.0270590279, 0.303341031, -0.056381505, -0.113421284, 0.474829495, -0.118202001, 0.107827209, 0.0186836272, -0.026815787, 0.179403469, 0.00967931189, 0.270995289, -0.026760146, -0.151628032, -0.0115571199, 0.0529516041, 0.0263677593, 0.124068633, -0.160642922, -0.112853952, -0.0200299285, 0.0159182549, -0.0208371449, 0.339251608, 0.305176735, 0.117476285, -0.134620458, 0.0015437305, 0.127077252, -0.0785016268, 0.417288393, 0.238831848, -0.0646649003, -0.13563621, -0.062621884, -0.100907519, 0.221166372, 0.000283576926, 0.108006507, -0.00899751484, 0.171452075, 0.163231164, 0.334624052, 0.269409269, 0.0745114684, 0.0378841646, -0.156279817, 0.00339309173, 0.0224851519, -0.0913040936, 0.0710502118, 0.0245534331, -0.0525172763, -0.038577199, 0.0161448307, -0.107072286, 0.136192858, 0.39509064, 0.133099765, -0.150670916, -0.049446024, 0.130605578, -0.0288623422, -0.143798009, -0.163164347, 0.00693029165, 0.126590222, 0.118523479, 0.080938369, -0.00965197384, -0.0947464108, -0.0619419217, -0.00715470314, -0.00270146132, -0.0735214204, 0.0742535591, -0.151724458, -0.0125956684, -0.104397401, -0.0435350612, -0.119662181, 0.130253017, -0.0800807476, 0.0336041003, -0.162998661, 0.151249141, 0.118235916, 0.152863652, -0.0664393678, -0.0333562046, 0.0307316929, -0.0308411717, -0.102692015, -0.0138695687, 0.0295279026, -0.142072499, -0.00501096249, -0.107449733, 0.0455400497, -0.0195156187, -0.0615311861, 0.115972221, 0.124515563, -0.0950696915, -0.126622051, 0.124619126, 0.0318044722, 0.125589073, 0.0714403093, -0.0599766597, 0.0153121948, -0.0946025029, 0.0842743814, -0.0511309654, -0.0530208051, 0.0968111455, 0.00915293396, -0.0872821137, -0.0341456234, 0.102241755, -0.01665999, 0.119171172, -0.144422844, -0.0895541161, -0.0499199256, -0.052215457, -0.0440448597, -0.0190680623, -0.0335104018, -0.0262646675, -0.0497884303, 0.0697918534, 0.142495424, -0.0332986861, 0.110444307, -0.0094948411, -0.126372278, -0.00455704331, -0.0486105233, 0.12990889, 0.0143363625, 0.0227083117, -0.0708423927, -0.152520552, -0.137440622, 0.0991905332, 0.100105286, 0.000482797623, -0.106433988, 0.0626822561, -0.0254948735, -0.0445605963, 0.143724233, -0.0775816068, 0.0380899385, 0.131213173, 0.0369970351, 0.555347502, -0.201430574, -0.0414778665, 0.141114205, -0.33520025, -0.370464921, -0.0574532077, -0.274042398, -0.131483033, -0.0907322243, 0.0974460095, -0.203305453, -0.42073375, 0.47158137, 0.366813898, -0.113600843, -0.0614014827, -0.353852451, 0.0422197282, 0.129882872, 0.124867126, -0.461125076, -0.305486768, -0.296992272, 0.273998022, -0.021624133, -0.135703504, 0.213814691, -0.22922188, -0.0694982186, -0.0723364055, -0.410044223, 0.133643985, -0.346173316, -0.377693415, 0.273995072, -0.092024982, 0.492017895, 0.155702621, -0.243523747, -0.113333344, 0.411658019, -0.128447473, -0.0385939032, -0.389254302, 0.5887869, -0.366192728, -0.154247478, -0.168141752, 0.125041366, 0.325447083, 0.195079327, -0.224076152, -0.118206054, 0.446439296, -0.486365557, -0.124470234, 0.133741826, -0.171902403, -0.177047312, 0.638065815, 0.274646997, 0.051066041, -0.139466986, -0.107618734, 0.0297544282, -0.220091492, -0.0604409091, -0.151147515, 0.330189705, 0.0256975237, -0.350477636, -0.0640393198, 0.00320906937, 0.0241069943, 0.464509428, -0.417699486, -0.246973693, 0.444603145, -0.266747594, 0.376226664, -0.150105625, 0.152337834, 0.0612906218, -0.0664541274, 0.114929914, 0.0786673874, 0.268577397, 0.15605171, 0.417720705, 0.199413553, 0.470382959, -0.0577348359, -0.0548698977, -0.0935151204, 0.127545625, 0.0078035742, 0.0265699625, -0.0717224181, -0.0504340976, 0.141311139, -0.0696884468, 0.16323486, 0.161642551, -0.122329846, 0.000614061952, -0.11422047, 0.050358355, -0.00613173842, 0.147310913, -0.094123058, 0.0851150006, -0.0109216571, 0.162879407, -0.0766158551, -0.0408613831, -0.138835713, 0.0914271474, 0.0538008511, 0.00182381272, 0.0737814903, -0.145339787, 0.0960951149, 0.00186766684, 0.074337095, 0.0707745701, -0.121303573, 0.0869064927, -0.143426806, -0.0767021254, -0.145929232, 0.0590681434, -0.0940708891, -0.0895382762, 0.0371032953, 0.0883596539, -0.0582239404, -0.113797262, 0.0268214941, -0.131399393, 0.0876528025, -0.0169712156, 0.1179443, 0.123716325, -0.10347344, 0.0290490538, 0.131688386, 0.117466539, -0.0690310672, 0.078287527, -0.0800115243, 0.0246971101, 0.163132936, 0.0679558963, -0.162407547, 0.0510225743, 0.0700337291, 0.0353672355, -0.0471597016, 0.124563307, -0.0549175069, 0.0960765481, 0.0576039851, 0.0939226151, -0.138071612, -0.16272974, 0.14180693, 0.127052635, 0.0691979527, 0.0186066478, -0.0436210185, 0.112668008, 0.151836753, -0.130478293, -0.0800932348, 0.0843013078, -0.0159841925, -0.0699108988, -0.0854893997, 0.101829261, -0.131741494, 0.110427737, -0.0373147428, 0.0468182415, 0.120769411, 0.157920867, 0.131401509, -0.116937503, -0.0149295926, 0.0747306943, 0.0690521449, 0.157443345, 0.0361470133, -0.000928029418, -0.085797511, -0.099450469, 0.0439981967, 0.0752660632, 0.0999066532, -0.0695023164, 0.127101213, 0.138731539, 0.0538168997, -0.126113072, 0.0579102933, 0.0603288114, -0.11367555, -0.0932602361, -0.0947551876, 0.161928266, 0.0670054406, -0.152517274, -0.119443081, -0.0530025437, 0.0707716495, -0.0716721267, -0.0182028264, 0.0914666355, 0.0158282369, -0.107406847, 0.148881912, -0.0748758167, 0.135902673, 0.0107438415, -0.0505460501, -0.035291031, 0.0490114987, -0.116351187, -0.0820245892, 0.125596762, 0.055951938, 0.0660329014, -0.141267851, 0.159412682, 0.10837099, -0.105503708, -0.0242334604, 0.0999364257, 0.0926392674, 0.0424462706, 0.131631523, 0.149942487, 0.103099883, 0.0117439628, 0.00787490606, 0.120170981, -0.0066229254, -0.0698821396, -0.142651588, -0.069035396, 0.101812184, -0.0520091951, 0.128917664, -0.152586937, -0.068852745, -0.150097668, 0.0555632114, -0.104257867, -0.0154575855, -0.113112211, 0.028790772, 0.0293522775, -0.0490736142, 0.0488602519, 0.0887404382, 0.0914811492, 0.017524913, -0.0747600794, -0.122864351, -0.00964725018, -0.0602798834, -0.0753273591, 0.0550567359, -0.0577910841, -0.0398901626, 0.0426249057, -0.00190958381, -0.0837952122, -0.0396775827, 0.0311595798, 0.142115742, 0.0540243685, -0.102474824, 0.111106873, -0.0722910613, -0.14458482, -0.0315432698, 0.00662769377, -0.0315567404, -0.0343233198, -0.138836607, -0.1084117, -0.120071545, 0.0678287297, -0.0514928028, 0.042799294, 0.0842432827, -0.151789159, -0.0310573131, -0.145213485, 0.0543832779, -0.105361283, -0.147677034, 0.121757835, 0.0353050381, -0.109623164, 0.0578208119, 0.0270651281, 0.0954961479, 0.0455076545, 0.122286648, -0.0423400179, 0.123219997, -0.0148939341, -0.0822361931, 0.00892750919, -0.0868784487, 0.151639044, -0.142283082, 0.047772795, -0.12218824, 0.106648445, -0.0525964126, -0.0187165588, 0.0657648593, 0.15673545, 0.119693875, 0.0478522331, 0.0524375588, 0.152596295, 0.0568727404, -0.0369117409, 0.0815172493, -0.0637242943, -0.0175206214, -0.0627865121, 0.0228999853, 0.0277960598, -0.0258706808, -0.148519099, 0.0107162446, -0.0336691737, -0.0282700807, 0.135024667, -0.0349259824, 0.118313044, 0.0499210954, 0.0843484104, 0.134076774, 0.069212392, 0.0448146164, 0.0758006424, 0.0656589568, 0.0590565503, -0.111669049, -0.0728071108, -0.0931207761, 0.0381206721, 0.14083901, 0.156331807, -0.132252619, 0.0311704725, -0.00140348077, -0.122498423, -0.0275599957, -0.00414100289, 0.160844088, -0.0431024805, -0.0646839961, -0.10675396, 0.0082680285, 0.0919086933, -0.145149052, 0.0982291996, 0.117589533, 0.0733727515, 0.0108935535, -0.0992472172, -0.048558116, -0.150409788, -0.0792096928, 0.030762082, 0.49022162, 0.0182307661, 0.480714977, -0.378586292, -0.0368776768, 0.049268052, -0.425883979, -0.725615144, -0.0373228937, -0.675218999, -0.574738979, -0.0518868715, -0.0013038636, -0.583526909, -0.730223477, 0.609810591, 0.441707015, -0.363520652, -0.0241881199, -0.752693892, 0.00165833533, -0.115487777, -0.15008311, -0.567783654, -0.232549682, -0.633635938, 0.500672102, -0.161515221, -0.0721822381, 0.620773315, -0.522351861, -0.00097887218, -0.156921908, -0.580892146, 0.129641712, -0.298512191, -0.566257, 0.536092401, -0.287257999, 0.484759092, 0.0449498594, -0.490486383, 0.110678136, 0.689217448, -0.0428475589, 0.15737474, -0.545062065, 0.76489383, -0.47298798, -0.0273196995, 0.0972206593, -0.00384633429, 0.630496681, 0.32831189, -0.538388073, 0.145757467, 0.399862111, -0.691184819, 0.0017003864, -0.0220513642, -0.447445124, -0.644410372, 0.668422043, 0.392070234, -0.0468451977, 0.0855437219, -0.0803282112, -0.300294876, -0.3404468, -0.0529031977, -0.156171352, 0.604205549, -0.142909676, -0.69650954, 0.116179541, -0.141062409, -0.0140885115, 0.641033947, -0.651350856, -0.476627052, 0.736315191, -0.705283701, 0.370219767, -0.0481508225, 0.295990199, -0.130537242, -0.120599881, -0.155902058, 0.0943113565, 0.534347773, 0.314219654, 0.659861743, 0.298346281, 0.774193525, -0.401816577, -0.0551900975, 0.0420240201, -0.154031619, 0.0370177217, 0.362220645, -0.00129672885, -0.202740803, 0.356362015, 0.0258443691, 0.0255437344, 0.149662539, 0.369858652, -0.0747841522, -0.0535692647, 0.27031967, 0.104696937, 0.146699116, 0.0754570588, 0.379355639, -0.0937281996, 0.249930471, 0.11574167, 0.146808445, 0.131498873, 0.0208481476, 0.372382045, -0.0393468291, -0.0316809863, 0.130481809, -0.149029747, -0.232095107, 0.361285716, -0.114618637, -0.0316845179, 0.205974355, -0.137053832, 0.490240693, 0.297377646, -0.120189525, 0.330296159, 0.115219384, -0.0331172645, 0.387578487, 0.146963894, 0.0641053915, 0.0907479823, -0.0902338177, 0.200826332, -0.111598574, 0.187561527, -0.0348756909, -0.0835927054, -0.0900550336, 0.0753460377, -0.0871660635, 0.194430575, 0.12928158, 0.0506621487, 0.144959927, -0.112752371, 0.0526520722, 0.403419793, 0.198506206, 0.11006856, -0.195946127, -0.0933659822, -0.0305248052, -0.0438925624, 0.316075265, 0.350200236, -0.0871866569, 0.124133334, -0.275475562, -0.0483866632, 0.236736432, -0.120782956, 0.00392837822, -0.0532640964, 0.13787958, 0.243518308, 0.261905015, -0.0372108705, 0.19408752, 0.0487671271, 0.0377072096, -0.173241466, -0.108089164, -0.0878314525, -0.145793796, 0.0463362187, -0.0969878435, -0.0221837349, -0.110339925, -0.0465959013, -0.0996397138, 0.441467464, -0.100139305, 0.500793517, -0.12553893, 0.650648475, -0.448481858, 0.055727765, -0.0804335698, -0.37545985, -0.382088363, 0.142399877, -0.592610776, -0.387133062, 0.146225095, -0.0953281298, -0.679993451, -0.575969636, 0.7376948, 0.568961322, -0.269446194, -0.0607884936, -0.531687319, 0.16166997, -0.0567344129, 0.110301703, -0.541509688, -0.340792179, -0.647219956, 0.608231425, 0.00234161317, -0.0024798885, 0.374973297, -0.498539656, 0.0463496745, -0.0568172559, -0.461672008, 0.0596202761, -0.358760566, -0.512394845, 0.474952221, -0.329839826, 0.477880478, 0.155993015, -0.474174678, -0.0169381648, 0.624229074, -0.131074041, 0.123580843, -0.728925049, 0.722532332, -0.598751128, -0.0936767384, 0.120279208, 0.0826101005, 0.52550292, 0.48629564, -0.296032012, 0.00989131629, 0.573383629, -0.63683629, -0.0097566992, 0.134450316, -0.251293987, -0.574646294, 0.570992053, 0.358471274, -0.0954062417, 0.0190446526, 0.0947686136, -0.133238733, -0.394725561, -0.0839549676, -0.0391273946, 0.4193497, 0.0271346197, -0.680548251, 0.113933273, -0.108122133, 0.0418651849, 0.493965507, -0.621778667, -0.364649504, 0.532188177, -0.408471376, 0.493265361, 0.15193212, 0.421377808, 0.118740946, 0.0574604534, -0.144471034, 0.0241376609, 0.281591117, 0.470254034, 0.427933753, 0.525194347, 0.510937274, -0.209113285, 0.0440744981, 0.537911177, 0.0631909966, 0.700703204, -0.296489149, -0.121498212, -0.0651518553, -0.438825577, -0.428939164, -0.0273933411, -0.542364836, -0.447933465, 0.11440134, -0.0916150808, -0.582198918, -0.472121894, 0.568189561, 0.316690892, -0.31232211, 0.113893203, -0.816570938, 0.141042948, -0.00329105556, -0.133219779, -0.681307614, -0.51381892, -0.520639539, 0.719965994, 0.130457491, -0.00253837183, 0.415222347, -0.554577887, 0.155463308, -0.107652009, -0.576649547, 0.118378758, -0.421216518, -0.505962789, 0.566176474, -0.237000242, 0.645743132, -0.0933980942, -0.510626853, -0.145580977, 0.65582639, 0.154009104, -0.0868722498, -0.549431741, 0.636650503, -0.354063123, -0.105135903, -0.161880419, -0.0204298478, 0.549638927, 0.508406162, -0.436023414, -0.0584783927, 0.446715385, -0.566174209, -0.0571391732, -0.0420459658, -0.416007429, -0.470021367, 0.775681853, 0.412166148, -0.0932256281, 0.11301896, -0.0802996904, -0.353574634, -0.246986672, -0.156189337, -0.140446439, 0.303787619, 0.125294387, -0.617018402, -0.0880270675, 0.0654413402, 0.0156612247, 0.542069077, -0.662613392, -0.46349588, 0.560698509, -0.608466208, 0.469120681, 0.00691606104, 0.328685313, 0.114083976, -0.109526314, 0.0544763058, -0.107762322, 0.234286532, 0.386639029, 0.324281037, 0.246348247, 0.687322855, -0.41911912, -0.116650671, 0.477443218, 0.0278963149, 0.444910675, -0.386232644, 0.103998303, 0.15486148, -0.320408076, -0.393775672, -0.131230876, -0.414794326, -0.359006017, 0.0249598324, -0.127389133, -0.569236636, -0.629272878, 0.539147139, 0.278620213, -0.257499665, 0.0520966873, -0.63428694, -0.125744715, 0.0248388648, -0.104800373, -0.566212237, -0.208551422, -0.363361478, 0.533870697, -0.0685384348, 0.0626019239, 0.439630836, -0.319578081, -0.14858824, -0.0550490022, -0.403415829, 0.108038008, -0.34575063, -0.429843307, 0.447198749, -0.141990691, 0.59693414, 0.110544086, -0.234951258, 0.0155857205, 0.357939929, -0.114321262, -0.152918845, -0.557902098, 0.37512207, -0.369553179, 0.0144886672, -0.160623297, 0.0732184798, 0.441052884, 0.317533225, -0.447550356, 0.0472142547, 0.284377068, -0.414046228, 0.120714337, -0.0163616836, -0.277786702, -0.32725051, 0.601789117, 0.402672023, -0.16362685, 0.141238362, -0.153014898, -0.16286689, -0.216121882, -0.013390556, -0.162145436, 0.47623083, -0.0257440992, -0.439182729, 0.103489846, -0.122017995, -0.0420396402, 0.461774796, -0.625268221, -0.309446841, 0.555086374, -0.609337032, 0.431747079, -0.043488197, 0.234840974, 0.0455984175, -0.0035201048, -0.133364901, -0.056265153, 0.370648772, 0.209268123, 0.390237391, 0.307164699, 0.614932656, -0.189340666, -0.0842343122, -0.0473672897, -0.0557996035, 0.027109459, -0.0249961168, 0.0939038396, 0.103752702, 0.045732066, -0.147157088, -0.0992687121, -0.00786061585, -0.0154058039, 0.00219622254, -0.0564748123, -0.130933926, -0.042567119, -0.0871178806, 0.0647472441, -0.00422275066, 0.0225516111, 0.102591366, 0.00966468453, -0.114079177, -0.120590433, -0.0356951207, 0.0790043622, -0.0486133695, 0.107794017, -0.0546786189, -0.129563645, 0.096283108, -0.13277939, -0.0293904841, -0.0927322134, 0.102269202, 0.0439638942, -0.138153598, -0.11100094, 0.0922213197, -0.0625466928, 0.106727898, 0.0414349884, -0.00586426258, -0.0285898596, 0.137372851, -0.0835694075, -0.0667934418, -0.0879341066, 0.0573251098, -0.0845206007, 0.0711719245, -0.0733544454, 0.0576870143, 0.157588571, 0.0551721156, -0.0499989837, 0.0523094982, -0.101175874, 0.108446538, -0.0881896168, -0.00455497205, 0.148655325, -0.134757295, 0.0246354938, 0.130518228, 0.092833668, 0.062664032, 0.00789417326, -0.152462259, -0.152179718, 0.0317082852, -0.0225716233, 0.0739560723, 0.159877151, -0.0290782303, -0.0287330598, 0.0506217927, 0.0666262805, 0.0566642135, -0.102736846, 0.00603431463, -0.00853055716, 0.07415694, 0.100707084, 0.121025503, -0.07195241, -0.0150468051, 0.121577859, -0.0408267304, -0.120197229, -0.0681589618, 0.115850985, 0.0236096829, 0.0548617393, -0.0622332469, 0.0821170658, -0.110110804, -0.0769889653, 0.0318334252, -0.0336323529, 0.123325884, 0.13359347, -0.133499131, 0.12924853, -0.00541119277, -0.111132674, -0.0541024879, 0.0614909977, -0.0928525105, -0.0908371881, 0.0132574886, -0.0147155672, -0.0558533296, -0.134932235, -0.106114566, 0.0129137635, 0.0888277292, 0.162185282, 0.0526746511, 0.124589205, 0.0483893156, 0.133044064, -0.0779883564, 0.134553224, -0.0794128329, -0.110639259, -0.00511342287, -0.157095894, 0.0743829459, 0.0151098669, -0.12768501, 0.0795354396, 0.157717228, -0.0775416121, 0.12226823, 0.00716878474, 0.0430308729, 0.0567948222, 0.017297551, 0.00478850305, -0.150256559, 0.0542277843, 0.154354751, -0.152704701, 0.129501969, -0.058455877, 0.116351455, -0.159054905, 0.0939283967, -0.0433823317, -0.0626717582, -0.0263082236, -0.0351381749, -0.100268766, -0.0709652305, 0.0514042675, -0.0680380762, -0.056085974, 0.046707347, -0.131497651, -0.116149254, 0.00604832172, 0.145483106, -0.0444852039, -0.111925371, -0.116210908, 0.054586336, 0.106943041, 0.0966070294, -0.0428996906, -0.0645875037, -0.00403787196, 0.115516216, -0.126738533, -0.0812134668, 0.131926775, -0.0382048339, -0.153560132, -0.133586928, 0.0575451404, 0.114768088, -0.0789349154, -0.114086047, 0.151159137, -0.0538072959, 0.0923282206, 0.134355068, -0.0795231089, -0.0624867603, 0.134258896, -0.101627342, -0.0795248598, 0.0107967677, 0.441993952, -0.139066011, 0.509807169, -0.338727742, 0.121571869, 0.0526470989, -0.253651619, -0.293420553, 0.163493395, -0.335473537, -0.320666045, -0.0325923488, 0.0726035386, -0.529781938, -0.504741907, 0.534747183, 0.21533148, -0.306457669, -0.113015719, -0.687392771, -0.0583471283, 0.0610998571, -0.146588206, -0.57851243, -0.201835886, -0.62127316, 0.405878484, 0.0238256156, -0.0037840358, 0.309542894, -0.505534053, 0.074793756, -0.051894553, -0.532541692, -0.114649743, -0.370541394, -0.485619992, 0.394204617, -0.0929058194, 0.527324915, 0.0534673929, -0.30447951, 0.056747213, 0.503786325, -0.143919289, -0.0526537746, -0.686152935, 0.651907206, -0.509824336, -0.0910361111, -0.103456348, 0.0490102917, 0.348727286, 0.343414128, -0.23864533, 0.0663249195, 0.400783867, -0.502852857, -0.155497, -0.0931663513, -0.420302957, -0.367817551, 0.547714174, 0.164440691, -0.0813766941, -0.124500081, 0.100800812, -0.180826217, -0.29651469, -0.144222438, 0.0243655443, 0.4347004, -0.161698669, -0.501220822, -0.146695539, -0.117981143, -0.147671416, 0.244278744, -0.503401697, -0.427816302, 0.311740518, -0.563367724, 0.47603637, 0.0146994144, 0.37532112, -0.075766921, 0.058101818, 0.0307064801, 0.0104036629, 0.215222538, 0.438887119, 0.312867224, 0.434892386, 0.678836644, -0.230070308, -0.0346788764, 0.135539651, 0.0684356987, -0.0969461799, 0.0690549463, 0.019808352, -0.0010163188, -0.158974886, -0.109342575, -0.130033523, 0.0430771559, -0.0633718967, 0.158747047, -0.0806969181, 0.0806020647, -0.0229079723, 0.0113418251, -0.0197244287, 0.0359276384, 0.140138358, 0.16205129, 0.14720434, -0.158206537, -0.126719534, -0.113589481, -0.0429993868, -0.11510475, -0.061171107, 0.160494298, -0.0569947138, -0.064365752, 0.0895652771, -0.160383955, 0.094832927, -0.102129027, 0.1289213, -0.10924194, 0.0664292276, 0.077781707, 0.00805166364, -0.156181887, -0.0123315454, -0.162259966, 0.0842120349, -0.153292581, 0.0169813335, 0.048204869, -0.0271361917, -0.0257713348, -0.120521367, -0.0996543169, 0.070569098, -0.142044365, -0.0572488979, -0.123574056, 0.105383098, 0.0740566254, 0.0334204286, -0.0226937234, 0.0601163059, -0.0554802567, -0.122368634, -0.129194438, 0.00694075227, -0.00992651284, -0.117194608, -0.0737629905, 0.0412670374, -0.120901704, -0.0318135619, 0.142036945, -0.122761771, -0.0417991206, 0.0187350959, 0.151388019, -0.083446525, 0.0418585837, 0.12548551, -0.12980698, 0.129596412, 0.0319731534, -0.113043115, -0.0834885538, -0.0419114605, 0.0409790277, -0.144570425, 0.153580338, 0.14070195, -0.0528837591, 0.126832068, -0.0166703314, 0.157051057, 0.0121169239, 0.0262094587, 0.139373958, 0.105287313, 0.0971889794, 0.0245707184, 0.104733497, -0.0554573163, 0.118129134, -0.00633625686, -0.104179233, 0.132831305, -0.154248729, 0.0872364938, 0.120168746, 0.0602686852, -0.110118181, -0.00822480023, 0.0902855694, 0.0575203598, -0.00816880167, 0.111358821, 0.0666944534, 0.0063624382, -0.116616175, -0.00947968662, -0.143011168, 0.0111370087, 0.0329586565, -0.0655932948, -0.0110010654, -0.052273795, -0.15626055, -0.0279808193, 0.160158396, -0.0524790436, -0.0802717507, 0.120310575, -0.126747116, 0.151772678, 0.120188922, 0.120360225, -0.112718269, 0.0354563892, -0.145706937, -0.0829948261, 0.0753687918, 0.0902329087, -0.0786656737, -0.0319633633, 0.124139667, 0.152555436, 0.000954940915, 0.148836911, -0.127420843, 0.144207329, -0.0666759089, -0.0436390489, -0.00409628451, -0.0378840864, 0.10916838, -0.112517662, -0.155451417, -0.00303453207, -0.104178339, 0.0397262722, -0.145308688, 0.0642977804, -0.0240566581, -0.0208615959, -0.0868684202, 0.0205352604, 0.0880286694, -0.00967116654, 0.100672543, -0.112298802, 0.065178901, 0.0787963867, -0.158477649, -0.102013916, 0.0337083638, -0.153997511, -0.0629012734, -0.0121338218, -0.158902302, -0.1543331, -0.0726605877, 0.111928463, -0.0777457282, -0.113058992, 0.116038084, -0.0927543789, 0.162210882, -0.0585885867, 0.0893027484, 0.123223305, 0.0966741741, 0.143311441, 0.145341635, -0.103996426, -0.164190054, 0.557450056, 0.0884151161, 0.639291942, -0.492361397, 0.0588587224, 0.117629766, -0.697069645, -0.742527306, -0.135094091, -0.642018616, -0.533658803, -0.116707787, -0.0142391846, -0.619176805, -0.611424685, 0.830365181, 0.491555691, -0.38637495, -0.132741034, -0.826098859, -0.0299241245, 0.0403840393, 0.0436050296, -0.602282345, -0.396619678, -0.785297215, 0.772719622, 0.0429444015, 0.0994133949, 0.507937968, -0.576737106, 0.146941662, -0.0635526776, -0.813409805, -0.0771416128, -0.536961317, -0.499054492, 0.644790232, -0.367845625, 0.685696363, 0.0110028088, -0.571688116, -0.0189255625, 0.70587188, -0.0163114965, -0.0300222635, -0.819171786, 0.597843289, -0.730313182, 0.0847572237, -0.126224041, -0.179086804, 0.620737255, 0.658990204, -0.428564608, -0.00946056843, 0.70666337, -0.720004976, 0.159122914, -0.0150391608, -0.399178833, -0.536109865, 0.639187992, 0.33377105, -0.0819991454, -0.00196225941, -0.0973744318, -0.245614499, -0.655343592, 0.0418089926, 0.136663407, 0.450652063, -0.0654002577, -0.811347425, -0.154498622, 0.0102185905, -0.160562858, 0.585477829, -0.578837037, -0.483005613, 0.605349004, -0.719573796, 0.47880441, 0.0901592076, 0.576717079, -0.131314769, -0.123574443, -0.111098178, -0.0128426254, 0.49125734, 0.603938222, 0.694636881, 0.723750353, 0.868569374, -0.484859616, -0.0460911319, -0.0282955319, 0.0105078816, -0.141571507, 0.0507009178, -0.00449171662, 0.160088629, 0.00964927673, -0.01668033, -0.0717027932, 0.0996360481, 0.107839793, -0.0042155236, -0.144733965, 0.145816535, 0.145177275, -0.13588506, 0.0657990873, -0.0969760343, -0.112076342, -0.056308195, 0.0260210633, -0.110306494, -0.137235254, 0.10531497, 0.026987642, -0.0318824798, 0.115143389, -0.0018171072, -0.0149492621, 0.041564256, -0.131003618, 0.143586278, -0.152686045, 0.140414089, -0.0679210946, 0.0356287062, 0.121698976, 0.0570731461, -0.0440827906, 0.148509175, 0.0366041809, 0.140334755, 0.0871664286, -0.0929299295, 0.0331635177, -0.145010069, 0.048058033, -0.150053769, 0.105083108, -0.116331905, 0.0805566013, 0.0667756051, 0.0069886297, -0.0406157449, 0.135706544, 0.156641632, 0.0750845373, -0.108838312, 0.103431165, 0.00327451527, 0.0382039696, 0.0843829811, 0.14751029, 0.0988347232, -0.135932952, 0.011143133, 0.13726452, 0.133011132, -0.155044481, -0.163575575, -0.0662450865, -0.12452057, -0.0628954619, 0.0880795717, -0.0777861103, -0.147109449, -0.0931565985, -0.028097108, 0.127007425, -0.0165983438, 0.0371452719, 0.0371015668, 0.130644977, 0.136970609, -0.0527876541, -0.0943405926, -0.0974269137, -0.132315829, -0.148498803, 0.103043675, 0.0140194893, -0.0725216344, 0.00304752588, 0.0776591748, 0.137675077, 0.0794013739, 0.0382805914, -0.162488669, -0.0958845466, 0.45020178, -0.101660199, 0.0576596111, 0.172514543, 0.167942315, -0.0752003118, 0.14174071, 0.312186599, 0.0337000154, -0.112241484, -0.0183200799, 0.173688367, -0.106258214, 0.139832288, 0.397794992, -0.0765157267, 0.161394566, -0.110299118, 0.0283825845, -0.134118006, 0.151293561, 0.389932126, -0.0337686837, -0.0862103403, -0.140315637, -0.129797518, -0.309679002, 0.294054031, -0.0485343561, 0.0548333377, 0.217076972, 0.140377596, 0.252240419, 0.269010067, 0.0323706903, 0.427743554, -0.155928552, 0.0966330469, 0.498500675, -0.0237093419, 0.0201865807, -0.013591826, -0.0770387575, -0.0273821075, -0.00800037198, 0.30545491, 0.0933884084, 0.0674042925, 0.0630279109, -0.00901216641, -0.240343884, 0.343841553, 0.00339852273, 0.106477417, 0.23892124, 0.0218574703, -0.0225892235, 0.497582793, 0.315465987, 0.151702091, -0.102816641, 0.00822237134, 0.114549458, -0.115673319, 0.25545013, 0.294650525, -0.0473477505, -0.108388156, -0.13317962, 0.102105878, 0.122800909, -0.11320357, 0.0174437165, -0.102633208, 0.103764646, 0.0253255628, 0.382327557, 0.0639541373, 0.21675925, -0.0397479422, 0.160911381, -0.1017536, -0.10928978, -0.160529092, -0.158405811, 0.117346019, -0.302847862, 0.00291978917, -0.0958752409, 0.0248619895, 0.105108425, 0.341887057, -0.00308091217, 0.287705183, -0.0105575472, 0.688412488, -0.26570183, -0.0863649845, -0.110546738, -0.392989814, -0.500748336, -0.0560525283, -0.448686957, -0.473035693, 0.0970930457, 0.0248499755, -0.574537039, -0.59329325, 0.490238756, 0.364462078, -0.346703529, 0.00366949174, -0.729998648, 0.0676431507, -0.163104802, 0.134877235, -0.460834265, -0.215701088, -0.559190631, 0.474410236, -0.158409089, -0.156517759, 0.458755732, -0.487597734, -0.0281765163, 0.129767358, -0.688476324, -0.105123416, -0.378440678, -0.435511798, 0.539446592, -0.290164888, 0.33827883, 0.0429170877, -0.333833486, 0.109210134, 0.416009873, 0.0366159976, -0.0821951479, -0.741815627, 0.458495885, -0.488926262, 0.127418876, -0.103338398, -0.0534072742, 0.528965116, 0.301861882, -0.424823552, 0.0128292888, 0.620722651, -0.615962863, -0.122730121, -0.0244416296, -0.415584892, -0.391243011, 0.689538658, 0.35691601, -0.039811112, 0.146358579, 0.0182403624, -0.288917094, -0.234162822, 0.0675176233, 0.0780176967, 0.515063047, -0.0749909282, -0.466391742, -0.0223069396, -0.104797281, 0.107833564, 0.382557809, -0.769132912, -0.557063818, 0.639055431, -0.553016961, 0.532853186, 0.0337761343, 0.457398891, 0.00832043588, 0.144739807, 0.129954278, 0.0430634618, 0.229402944, 0.399002939, 0.492834717, 0.217971221, 0.626553833, -0.355263889, -0.0705634356, 0.365773976, -0.102968745, 0.581715167, -0.292746723, -0.158097163, 0.000816971064, -0.524812043, -0.540849507, 0.0835072398, -0.554740667, -0.203891128, 0.112377599, 0.0999121964, -0.577461302, -0.624885738, 0.645700157, 0.546612561, -0.16563566, -0.159115002, -0.553806603, -0.0300434828, 0.12264204, 0.142362773, -0.319244921, -0.141219452, -0.563815057, 0.524686813, 0.0863822699, -0.0676425621, 0.487702399, -0.42823261, 0.103487641, -0.0790933371, -0.579273939, -0.0181378126, -0.233051777, -0.369673759, 0.531396389, -0.216927305, 0.389629453, 0.0376024395, -0.263708085, -0.1122142, 0.600750923, -0.00697302818, 0.143476903, -0.354352534, 0.466777235, -0.513120234, 0.148634136, -0.0483818129, -0.0145727647, 0.552580833, 0.302301943, -0.514643669, 0.035983488, 0.565658629, -0.555040777, -0.0657578036, 0.043617785, -0.368212581, -0.2518332, 0.682877779, 0.210403129, -0.0530348495, 0.0242800862, -0.0479837731, -0.155546635, -0.32477513, 0.147618383, 0.0404638797, 0.331791252, -0.0305147041, -0.29054299, 0.00499023171, -0.04934863, -0.11974787, 0.335277975, -0.354659379, -0.179735973, 0.473471969, -0.453504831, 0.4686625, 0.107458383, 0.556927741, -0.152169064, 0.0492892563, -0.0520460755, -0.15253292, 0.244955033, 0.535728574, 0.448274583, 0.449199677, 0.58666712, -0.255327255, -0.00719438493, 0.113307148, -0.0490309298, 0.136712521, 0.102911264, -0.0562655032, -0.135443196, 0.0771055222, 0.00926114619, -0.15982151, -0.119227417, 0.0349941254, 0.023914516, -0.0962749496, -0.0184646845, 0.00231051445, -0.0516015515, 0.0474790484, -0.0376097709, 0.139554203, -0.00712683797, 0.0152093768, 0.0482303798, -0.0546784252, 0.000771477818, -0.115711249, -0.0532100871, 0.0822083354, -0.151371017, 0.0722572356, 0.0575166941, -0.0874566957, 0.0718728453, 0.119369715, 0.145302653, 0.126144797, 0.00938253105, 0.0255864561, -0.072615169, 0.092800498, 0.0756323785, 0.141705006, 0.138131678, 0.153961122, 0.0350870192, -0.139959693, 0.158412635, 0.0583490431, 0.124685198, -0.141283348, -0.0853454173, 0.107138813, -0.0281750262, 0.145110786, 0.120010078, -0.0907068178, 0.144778758, 0.11662972, 0.111001283, 0.0123670399, 0.00130191445, -0.060296312, -0.0778801888, 0.13452217, -0.118228219, -0.121032074, 0.160016149, -0.010779351, -0.0615965873, -0.113177419, -0.00719375908, -0.135659263, 0.151763588, -0.0326568335, -0.122038797, 0.158478349, 0.0329133123, 0.0567354709, -0.0743193477, 0.0364985466, -0.00123086572, -0.0693276227, -0.0117699951, 0.0864805281, 0.0515207797, -0.104820654, -0.139231101, 0.00988297164, 0.0226658136, 0.0392648578, -0.0405441448, 0.118405789, 0.090160042, -0.111576803, -0.00421194732, -0.048291415, 0.0914777219, 0.0717419237, 0.0794127584, 0.0746217966, 0.149923742, 0.0298696458, 0.129404753, 0.127113312, -0.154944152, -0.111794457, 0.0374573171, -0.0439781398, -0.145979106, 0.115781009, 0.138640881, 0.110454142, -0.0922910497, -0.0243179351, 0.12454167, -0.122636236, 0.146100909, 0.102338761, -0.0293168128, -0.0777365565, -0.0299185067, -0.116654679, 0.073814109, -0.0465901643, -0.0353710204, -0.0922853127, 0.110100627, 0.121983886, 0.0366243571, 0.0896642208, 0.146680325, -0.0634426847, 0.0662637353, -0.023409307, 0.0878977776, -0.105877489, -0.0825615823, 0.0578624904, 0.000741735101, 0.106188476, -0.161148012, -0.0537287071, -0.0181663334, -0.160685301, 0.0324846804, 0.058604002, -0.136509702, 0.0350973606, 0.123163432, 0.13711828, -0.121017516, 0.0100488067, -0.158680752, 0.12512064, 0.0452426672, -0.0946112797, 0.0939565301, -0.10807839, 0.112726271, -0.0899684727, 0.0789184868, -0.0634277016, -0.0892491713, 0.089758873, -0.00540518761, 0.148056298, -0.129682034, 0.160088122, -0.0990025997, 0.0283056647, -0.116143093, 0.0582511276, 0.0243424028, 0.14091894, 0.089319855, 0.106828302, -0.158878192, 0.108011752, -0.0146413445, 0.0393931568, -0.0985064879, 0.0611050129, -0.0437651649, 0.0230949968, -0.132615, 0.0725359917, -0.030034855, -0.139944196, 0.0286053121, -0.161292106, 0.115559071, 3.50028276e-05, 0.138058379, 0.44595167, -0.112750418, 0.586436749, -0.18605642, 0.0221053362, -0.121054962, -0.28348121, -0.481277496, -0.138386697, -0.443925351, -0.152053058, -0.143291309, -0.09675356, -0.331217974, -0.322780609, 0.652282, 0.389210433, -0.22817868, 0.108947843, -0.605782509, -0.0636121109, -0.103902429, -0.00235677604, -0.474621475, -0.331117302, -0.50037533, 0.576908469, 0.138083309, 0.0427852869, 0.216796279, -0.204590082, -0.139792457, 0.151014566, -0.396641999, -0.0956864879, -0.273098677, -0.340411037, 0.49002412, -0.035883449, 0.315274835, -0.153516039, -0.431934029, 0.13903892, 0.442591548, 0.147287577, 0.0348900855, -0.33573693, 0.349962384, -0.512681246, -0.0903105661, 0.137177259, -0.183730364, 0.52737993, 0.432697535, -0.188888282, -0.100112647, 0.388102978, -0.36916399, 0.0430034846, -0.109816089, -0.333949298, -0.25057292, 0.430464625, 0.256102145, 0.150464833, -0.137685239, 0.0858787149, -0.0092154704, -0.409404546, -0.135986999, 0.115654387, 0.190700099, 0.0764649734, -0.489438385, 0.013715148, 0.0423517674, -0.0132389218, 0.34220162, -0.504123628, -0.417430013, 0.443611652, -0.381673127, 0.372079343, -0.0413543284, 0.48459959, -0.0061288625, -0.0898546651, -0.139980927, -0.122052342, 0.397376984, 0.287683517, 0.389755011, 0.168228, 0.440504611, -0.391135067, -0.115398087, 0.368806154, 0.144292057, 0.666148245, -0.295957625, -0.128800988, -0.0523887873, -0.327424884, -0.63010931, -0.0571694896, -0.4527722, -0.327675492, -0.0638770536, 0.116620019, -0.623492956, -0.399212122, 0.687634766, 0.4854168, -0.165422186, 0.0381399803, -0.560516655, -0.111920848, -0.0713309273, -0.0218032002, -0.600302339, -0.245551959, -0.584802151, 0.602103591, -0.0248815566, 0.147765622, 0.547490478, -0.363089383, -0.135686725, -0.056656763, -0.709209502, -0.0244266093, -0.33522138, -0.376700163, 0.454973698, -0.164785072, 0.417199075, -0.118631303, -0.4710522, -0.149125859, 0.396622092, 0.0551476926, -0.159949645, -0.672562361, 0.391216636, -0.572889864, -0.134335175, -0.00379136065, 0.0866543278, 0.562384129, 0.562679172, -0.291454941, 0.123171002, 0.543776989, -0.617436826, -0.0384951085, 0.0378085077, -0.315583587, -0.596083164, 0.667865932, 0.369450241, -0.0663186833, 0.0879521668, 0.0813223422, -0.278673381, -0.239515796, 0.0235563815, -0.0272717029, 0.418066204, 0.0371295176, -0.395289093, -0.169852585, 0.0153496116, -0.106603414, 0.563040793, -0.391532809, -0.39579609, 0.614383042, -0.733934581, 0.34122771, -0.127683178, 0.256479502, 0.139217913, 0.0250917338, -0.00917327404, -0.138782993, 0.398879826, 0.503764868, 0.572306454, 0.417858213, 0.709144771, -0.423139185, -0.00984169636, 0.249974772, -0.138091862, 0.364506155, -0.349626631, 0.0302381963, -0.127652079, -0.490085542, -0.506152272, 0.0902526975, -0.544142902, -0.401436567, 0.147049859, -0.100977749, -0.443593055, -0.640596688, 0.513544142, 0.272330821, -0.308311224, -0.0190547593, -0.42115292, 0.088840723, -0.0523722842, 0.0393958986, -0.431444377, -0.221192867, -0.630877137, 0.392028749, 0.0817826539, 0.0805819854, 0.283990055, -0.347432345, -0.11417982, -0.147417858, -0.606067061, 0.0422533602, -0.539653599, -0.40425384, 0.618931174, -0.138789877, 0.509309411, -0.0261738747, -0.469365388, -0.135597095, 0.442085475, 0.0206466317, -0.102746956, -0.70041877, 0.625671446, -0.367646456, -0.0632964373, -0.0993643552, -0.0348705277, 0.377774149, 0.278579116, -0.48243764, 0.126838237, 0.529198825, -0.669488847, 0.0812171698, 0.054817766, -0.187311932, -0.349997312, 0.542369664, 0.303090066, 0.0404316038, -0.00761955976, 0.0447394699, -0.142743871, -0.155341089, 0.097596854, -0.114327192, 0.489023179, 0.0430193879, -0.622503221, 0.042683389, -0.0441782326, -0.0414686576, 0.300205052, -0.373713821, -0.276699483, 0.400933266, -0.616034627, 0.307890356, 0.162023872, 0.400575429, 0.0726469308, -0.0236400664, -0.0107193291, -0.156185508, 0.2785483, 0.457425833, 0.410774738, 0.193416193, 0.432937652, -0.17723386, -0.146579936, -0.00756184757, -0.119481906, 0.102186471, -0.00778718293, 0.00475034118, -0.13913402, -0.0542624295, -0.110377587, 0.140395194, -0.127389356, -0.0256051123, 0.125957698, -0.00957213342, -0.138897985, 0.119996846, -0.00475716591, -0.0739550516, -0.147220612, -0.0860958546, -0.108710796, 0.00204724073, 0.0643659383, -0.016369611, 0.0479123294, -0.0116454363, -0.0187886357, 0.033736527, -0.0737894103, -0.103630066, 0.037814945, 0.0955679715, 0.00987255573, 0.130285144, 0.023203209, -0.0693595409, -0.0193948895, 0.0844631642, 0.0923372805, 0.00386692584, 0.00629664958, 0.0247004628, -0.133215606, -0.0103455931, 0.139389604, 0.117557853, -0.154562965, -0.121263929, 0.128890812, 0.112620324, -0.134338409, 0.00920456648, 0.0256420672, -0.143788069, 0.0683580041, -0.12773031, 0.0784700215, 0.155654162, 0.0480764508, -0.0747131407, -0.0710990727, -0.13354747, 0.131954491, -0.149661109, -0.107521765, -0.139731497, -0.0106424689, 0.0728490204, 0.01741831, -0.158807725, 0.0159702748, -0.0415058434, -0.119286455, 0.0227292627, 0.0414880812, -0.126885593, 0.0374771059, -0.0701874718, -0.0629096627, 0.122658938, -0.0442790613, 0.114217967, -0.0829791799, -0.100799873, 0.12931779, 0.0433369577, -0.0923474357, -0.104685172, 0.120629996, 0.0667749494, 0.0171021372, 0.118342817, -0.0239938796, 0.0588032752, 0.00731675327, -0.056843549, -0.1150617, 0.519775033, 0.147494406, 0.614444494, -0.258088827, -0.0822837204, 0.088101238, -0.353880972, -0.424828082, 0.017291069, -0.401889592, -0.342932194, 0.0998233259, 0.128418967, -0.499779075, -0.417371124, 0.635582507, 0.595416248, -0.266298324, 0.0291384086, -0.597675443, 0.124464393, 0.0385677665, -0.155177101, -0.66621244, -0.398452222, -0.627606809, 0.533958614, 0.153116792, -0.1258737, 0.556227088, -0.589947164, -0.146078765, 0.016105786, -0.423407733, 0.0321676433, -0.243269831, -0.442018747, 0.616438389, -0.31291604, 0.520751715, 0.126311183, -0.262663662, -0.1560155, 0.653536022, -0.00504483283, 0.157828242, -0.466344327, 0.651329696, -0.353001237, -0.097630173, -0.0325627476, 0.0778525472, 0.485905498, 0.427210808, -0.413364828, -0.0744382367, 0.614035904, -0.565784395, -0.161923185, -0.146218568, -0.31388855, -0.458032191, 0.757910967, 0.230990171, -0.0592873618, -0.0806296095, -0.122000054, -0.0845654085, -0.359386235, 0.0791448355, 0.0826618373, 0.468694746, 0.0463402309, -0.494799078, -0.00298376475, -0.0321459472, 0.020420149, 0.397592872, -0.614408612, -0.293756515, 0.49530074, -0.555849254, 0.524762213, -0.089752771, 0.544954598, -0.152584046, 0.0429189093, -0.113132432, -0.140150577, 0.478245139, 0.497568518, 0.327347666, 0.51620239, 0.679007888, -0.395210326, -0.0649744272, 0.148974866, 0.145406544, 0.326290607, 0.310199171, -0.126020357, 0.0601469167, 0.201868996, 0.0761633217, -0.0479025319, 0.0397451632, 0.05259436, -0.147881895, 0.0754169673, 0.111209087, -0.00514646061, 0.0437962823, 0.12779972, 0.0701746419, 0.0762056783, 0.122506157, -0.103380799, 0.0606693588, -0.02817134, 0.0684814155, 0.104962528, 0.0349797159, 0.0805134177, 0.113111347, -0.0596714243, -0.0685503334, -0.0513786189, -0.0752981305, 0.0539475381, 0.117789574, -0.0718425959, 0.221287593, 0.15251343, 0.286976069, 0.294763237, 0.21767965, -0.154597819, 0.355161935, 0.0312419534, 0.340162426, 0.136729896, 0.020221144, 0.0934556276, 0.0655074269, 0.294748843, -0.122991249, -0.117743813, 0.123258702, 0.131560728, 0.0630405247, 0.0318238959, -0.101435632, 0.0697783306, -0.139293939, 0.112363696, 0.0877092034, 0.236433983, 0.313382506, 0.0940187052, -0.0633466691, 0.0664201677, -0.161030874, -0.151650518, 0.256947249, 0.160200164, 0.0945609882, 0.112756416, -0.0365187563, -0.109610677, -0.127906963, -0.0406174064, -0.101556361, 0.0777039379, 0.268369436, 0.191169307, 0.226924211, 0.196128279, -0.0254770555, 0.185996354, -0.141340315, 0.202250749, 0.0238962919, 0.108804502, 0.0545238703, 0.0531742275, -0.0210179687, 0.0817717761, 0.184890166, 0.0318714604, 0.139185533, 0.364861608, 0.106378496, 0.405968398, 0.11867854, 0.621314943, -0.150368065, -0.0711757839, -0.090414755, -0.367947131, -0.555050194, -0.0816438645, -0.595071852, -0.199055448, -0.061466828, -0.101530716, -0.53283298, -0.636598051, 0.539453864, 0.389318317, -0.349864304, -0.0257032141, -0.560641646, 0.0508092493, 0.0861191601, 0.121918261, -0.381255478, -0.18316631, -0.466059476, 0.572981119, -0.155610383, -0.154670388, 0.554691136, -0.469072819, -0.159416512, 0.013751179, -0.594866157, -0.101650283, -0.219495296, -0.358794928, 0.31815964, -0.0620448031, 0.328524083, 0.144110203, -0.366164953, 0.0451763719, 0.556052566, 0.0099939853, -0.0961542651, -0.637229979, 0.659403741, -0.32282716, -0.10913717, -0.130307913, 0.0232311822, 0.518359661, 0.33809033, -0.401391, -0.0845281705, 0.417067647, -0.55512315, -0.0236482769, -0.0824360922, -0.495364964, -0.522868514, 0.51517874, 0.270456582, -0.0449266434, 0.0202498734, 0.0107681155, 0.0149108153, -0.424757004, 0.0333399437, -0.16085735, 0.500839889, -0.00494448934, -0.305134892, -0.0757917464, 0.0154404491, 0.112606734, 0.215725273, -0.502727866, -0.440516531, 0.582694948, -0.509508312, 0.394873142, -0.116406709, 0.29935807, 0.138118565, 0.139017195, -0.012118876, 0.142583609, 0.381821364, 0.385827512, 0.338229328, 0.349675417, 0.525165737, -0.162506357, 0.0806630775, 0.397840798, 0.158269227, 0.565423429, -0.482560396, 0.076637432, -0.0361478329, -0.551676989, -0.518240035, -0.00471878052, -0.750547767, -0.533950269, -0.130543947, 0.117984653, -0.577980936, -0.542497277, 0.709943354, 0.608192801, -0.290380239, 0.0145241646, -0.641399682, 0.0205915272, 0.0721015781, -0.0806564167, -0.769179463, -0.391189367, -0.66115123, 0.61085844, -0.0707913935, 0.0495737791, 0.607234836, -0.670937061, -0.0285124332, 0.0933458805, -0.649779618, 0.00695577264, -0.447989613, -0.478503346, 0.547068417, -0.263118178, 0.570910633, -0.0855446532, -0.299159408, 0.131563038, 0.457598746, 0.0860937089, -0.131892502, -0.728270054, 0.665035605, -0.676929832, -0.103465825, -0.0917274803, 0.0441536009, 0.526314795, 0.551245034, -0.508450031, 0.162079453, 0.723964572, -0.626730025, -0.138353184, -0.0878784657, -0.316647023, -0.614921331, 0.689072728, 0.560254633, 0.0810371786, 0.158037364, 0.108243942, -0.269830137, -0.588239431, 0.0591605008, -0.108321875, 0.518104255, -0.0168613438, -0.536693215, 0.134729356, 0.0346420407, -0.0584235266, 0.417535305, -0.612774253, -0.359917134, 0.665088236, -0.740427077, 0.684177279, -0.158214375, 0.417424828, 0.0969944596, -0.0641079023, 0.0246922672, 0.0800217092, 0.324285537, 0.382858187, 0.64445585, 0.564454079, 0.622563481, -0.264034808, -0.182002351, 0.50633955, 0.148214698, 0.667985201, -0.275125474, -0.112389594, 0.149507165, -0.29702732, -0.530860662, 0.160199463, -0.519571424, -0.395419925, 0.115671486, -0.0081042964, -0.582681179, -0.541328728, 0.66664952, 0.521088779, -0.333488792, 0.150842801, -0.585325658, -0.106383383, -0.0460309237, 0.0532179326, -0.351838708, -0.155277163, -0.474652886, 0.624399066, 0.0299001634, -0.060808327, 0.312970072, -0.500387847, 0.101518661, -0.0265271217, -0.619048536, 0.0174390376, -0.432781994, -0.449227065, 0.63662535, -0.188352078, 0.570470452, -0.151203692, -0.349397272, -0.0856873915, 0.297691554, 0.0859886706, 0.139911354, -0.552419126, 0.610449553, -0.408825487, -0.0327040106, 0.0340986922, -0.110104032, 0.258700788, 0.343072563, -0.238430113, -0.067981258, 0.584845066, -0.56816262, 0.0731910765, 0.0714245439, -0.467525035, -0.295898318, 0.669248044, 0.426592946, 0.0510256141, 0.010111779, 0.131234467, -0.244817048, -0.432687908, -0.152725846, -0.0786553249, 0.42936331, -0.0623702295, -0.565815985, -0.156089813, 0.043109268, -0.0849284455, 0.551438272, -0.694053113, -0.329528183, 0.478031367, -0.491907597, 0.449810416, 0.0867519975, 0.296629578, -0.112815231, -0.148438647, -0.125211895, 0.0728497952, 0.407273591, 0.355800509, 0.382842451, 0.296325058, 0.616428375, -0.308542997, -0.0751222149, 0.453615427, 0.0577753931, 0.3828803, -0.416544408, 0.0849298537, 0.116603225, -0.532384634, -0.44641757, 0.0267062634, -0.617753983, -0.492963284, -0.0179675668, 0.133806497, -0.707872331, -0.581415296, 0.59788996, 0.413527071, -0.434634835, 0.131985739, -0.481587589, -0.0678793788, -0.0812599808, 0.060745094, -0.561051071, -0.198959947, -0.418468595, 0.648442626, -0.0445676595, 0.126099154, 0.290102661, -0.3357023, 0.0497563183, -0.0737208128, -0.678454101, -0.0649868399, -0.540649831, -0.280909985, 0.666397512, -0.115215681, 0.356908649, -0.0561072379, -0.393194079, 0.0271456391, 0.360621095, -0.00482104719, -0.101055421, -0.755787194, 0.69054687, -0.2751652, 0.0243001133, 0.0668939501, 0.0816490576, 0.561572075, 0.485886395, -0.526705921, 0.0488811284, 0.555535436, -0.609173179, 0.0269331634, -0.0549761951, -0.356687486, -0.396110177, 0.648423851, 0.438526928, 0.117753237, 0.0433321595, 0.0664716065, -0.191660315, -0.51265794, 0.0635962412, -0.109660096, 0.495803326, -0.160259277, -0.678943098, -0.0486204214, 0.118565559, -0.0302938819, 0.439080924, -0.74465692, -0.408146977, 0.567203701, -0.628664851, 0.392708182, 0.0364463031, 0.539461076, -0.0431091934, -0.122114636, -0.141344175, -0.102616817, 0.405467778, 0.283423007, 0.514123976, 0.326692671, 0.670492947, -0.263855696, 0.08216241, -0.0388310328, -0.107183188, 0.0785647631, 0.0351204276, 0.0376709551, -0.101815298, 0.102445573, -0.0482023656, 0.108227611, 0.0152095705, 0.0615635365, 0.152454495, -0.131727323, 0.133497417, 0.0382147878, 0.0124592185, -0.0766612291, 0.137142777, -0.15651609, -0.119501613, 0.133707017, 0.0176309049, 0.0328589976, -0.136286035, 0.100911617, -0.129882902, -0.140613794, 0.0409542918, -0.145751953, 0.155828208, 0.122812688, -0.115925863, 0.0327185988, -0.0719003528, -0.157261074, -0.00874872506, 0.103502899, 0.163358271, 0.0562630892, 0.0865329504, 0.0371291935, -0.0100828707, 0.158189207, -0.130781978, 0.130930871, -0.0712066889, -0.0204116553, 0.0157199502, -0.0266768038, 0.0437467098, 0.135944456, -0.0985283405, 0.0103695542, -0.0244678557, -0.0596612915, -0.0967206433, -0.136298299, -0.128198087, 0.150954813, -0.032151714, 0.0824177563, 0.0438205749, -0.152101055, -0.0721465349, -0.101961359, -0.096888043, -0.111593693, 0.0891235769, -0.114137359, 0.0211732537, 0.110271603, 0.13884452, 0.132000655, 0.0578103662, 0.162905514, 0.0782548636, -0.0433111191, 0.0684325695, 0.0323264152, 0.0631094873, -0.0388659537, -0.133827165, 0.00686399639, -0.139517948, 0.0431393087, -0.0887382776, 0.0840364397, 0.109793961, -0.0809742361, 0.00205282867, -0.0816948265, -0.111829728, -0.0600410402, -0.13300544, 0.105756789, 5.89638948e-05, -0.0927059501, 0.0117419064, 0.0474243462, 0.0968144536, -0.010594666, -0.00223568082, 0.129005492, -0.0224349797, 0.132145345, -0.161708385, 0.129850835, -0.0260870159, 0.0257228762, 0.0645697862, -0.00966651738, -0.000548943877, 0.136621416, -0.124691792, 0.138217419, 0.0693324655, 0.142067879, 0.0935439467, -0.10715989, -0.0409200713, 0.111809373, -0.0730942637, 0.06886971, 0.152408063, -0.0060108155, -0.056498535, -0.0998365805, -0.0427559018, -0.13804391, -0.133692622, -0.127558351, 0.139859378, 0.115055382, -0.116937697, 0.0134195834, 0.0283520222, -0.130246654, -0.106850773, 0.0778239965, 0.0786512792, -0.0456171855, -0.111089401, 0.0569805205, 0.101532519, 0.15635708, 0.125812292, -0.0781410784, 0.151676387, 0.0361477882, 0.0478829145, -0.0769888088, 0.0199892968, 0.156485587, -0.0215195566, -0.0441067442, -0.138089329, -0.0403212979, 0.0625969172, -0.00178217888, -0.0309625715, -0.0956418067, 0.127897501, -0.14210403, 0.0665718466, -0.00214217603, -0.135596901, -0.091559805, 0.0842342377, -0.0223634839, -0.132945821, 0.0846386403, -0.0635155365, 0.0578899235, -0.06170737, -0.08923392, 0.0979696512, -0.108609766, -0.111130059, -0.0533079952, -0.00795345008, -0.144035608, 0.0530887395, -0.0260584503, 0.0362722725, 0.0582222939, -0.0592440516, 0.0344848633, 0.142323405, -0.148073673, -0.0477864891, -0.0852552056, 0.0638860762, -0.00849227607, 0.117513061, -0.108621396, -0.0595070049, -0.0546364412, -0.0856257826, -0.0665752366, -0.0167004615, 0.047051847, 0.0724532306, 0.122164041, 0.15057227, -0.148559004, -0.129538625, -0.114822984, 0.138359904, -0.101009145, 0.0342938155, -0.0540949553, -0.155863166, 0.107158601, 0.000746846199, -0.106591828, -0.0920575112, -0.103666857, -0.0837997049, -0.128735825, -0.144584239, 0.109977722, 0.0365142822, -0.089817822, 0.0686632544, -0.118353978, 0.0208329856, -0.0169291198, 0.121135801, -0.0383384079, -0.0704740435, 0.00662916899, -0.00616030395, 0.141269028, 0.0238397866, 0.00578574836, 0.148270756, -0.0914776698, 0.0931250751, 0.0479803383, 0.114563704, -0.152636841, -0.0359028578, 0.0379691571, 0.0383860022, 0.0368668288, 0.0355007648, -0.0565695912, 0.00555181503, 0.0846559703, 0.0924804211, 0.124581605, -0.024696365, 0.161692291, -0.157570302, 0.144645333, 0.00591908395, -0.0799500644, -0.0864313543, -0.151238739, 0.00941304862, -0.0696537122, -0.117625237, -0.0772694796, -0.0992655903, 0.0247317553, 0.0445473194, 0.0941916406, 0.126629204, -0.160147369, -0.0240224749, -0.027992174, 0.118278056, -0.0174906552, -0.0447164029, 0.0152300149, -0.157149076, 0.0326353014, -0.0297223479, -0.0806426033, 0.0219101459, -0.100199431, -0.0197615325, 0.093583405, 0.0927602351, -0.0203849971, 0.131421179, 0.0165056735, 0.133956343, -0.124049872, 0.00708770752, 0.00541654229, -0.0545195788, -0.0799320787, -0.129711732, -0.0440752581, -0.11498972, -0.162459165, -0.11959666, 0.0107180029, 0.157032371, 0.0371583402, -0.149518833, -0.121065006, 0.0785758793, 0.00238473713, 0.16225329, 0.0344697684, 0.15203613, 0.162339389, -0.126531214, 0.0897512436, 0.00254370272, -0.150429532, 0.12278074, -0.127163619, 0.0806029588, 0.0555133075, -0.0710638762, -0.13952738, 0.128767073, -0.0739056095, 0.0709145069, 0.0982347131, -0.156076491, -0.0326104462, -0.0898958966, 0.0621866137, -0.115847431, 0.0908744037, -0.127097487, -0.147080988, 0.00496701896, 0.0847074687, 0.112060159, 0.115001231, 0.0699253678, 0.0887205005, -0.103006169, 0.152153879, 0.0276395977, -0.0173458904, -0.0970288664, 0.151672065, -0.104945913, 0.0993124843, -0.082130529, 0.0472138971, 0.0591498464, 0.0025165081, 0.0561734587, 0.116410345, 0.00971533358, -0.158004716, 0.000844746828, 0.0539794117, -0.0303224027, -0.0172255486, 0.106499046, -0.0482207835, 0.124287426, 0.0913334787, 0.0589807332, -0.0470732749, -0.145849556, -0.146196827, 0.0152328163, -0.0500512347, 0.0185734779, -0.134608001, -0.106996626, 0.0323509872, -0.055607155, 0.090772301, -0.128017664, 0.0789488107, 0.0435970277, 0.102189124, 0.11229828, -0.105882987, 0.00146690011, -0.0865171999, 0.0608022064, -0.0245680958, 0.114218801, -0.0611610785, 0.156162828, -0.148456082, -0.00524675846, 0.132782161, 0.132859021, -0.00129774213, -0.0549030676, -0.00461381674, -0.161984563, -0.0757002756, -0.00927983224, 0.0743108839, -0.0866766796, -0.0463303998, -0.0886987522, 0.150229394, 0.0311086178, 0.147141278, -0.090859428, 0.137998849, 0.0968773365, -0.0606210008, 0.153783172, -0.147051454, -0.0981692001, -0.0569776669, -0.152216166, 0.0464507043, 0.0545966029, 0.0901091397, 0.0207318962, -0.0152929574, 0.0532311201, -0.0832163095, 0.0727336407, 0.0413533151, 0.125680208, -0.0663604289, -0.0458159596, 0.0937085152, -0.0754143, -0.0280897766, 0.133869439, -0.037905857, -0.150748685, 0.0257207602, -0.0458133072, 0.125277996, -0.0266110152, 0.101955652, -0.0578948036, -0.00356604159, 0.0977877676, 0.0490948409, 0.10258919, 0.127317637, -0.0701702684, 0.0549246073, -0.13032259, 0.0402686596, 0.160877556, 0.000131621957, -0.150902569, 0.0951546729, -0.0236901045, -0.131989583, 0.0745921433, -0.0583700314, 0.0736912787, 0.15345943, -0.102284759, -0.0570667088, -0.16215001, 0.0929598212, -0.0282217413, 0.149925649, -0.104648814, 0.0151261389, 0.0776869208, -0.158167154, -0.162315384, -0.0982486084, 0.0347411931, -0.126369506, 0.0033583343, 0.0136035681, -0.0348615199, 0.047157988, -0.119330235, -0.112234063, 0.105329335, -0.136223733, 0.00558198988, 0.0519717038, 0.145612687, -0.121952757, 0.0238354504, -0.0617154837, -0.149181783, 0.0423938632, -0.133591801, -0.125239909, 0.0524818152, 0.0818570256, 0.0321598649, -0.139162153, 0.0761044174, -0.0540762618, 0.0459468365, 0.0898633301, 0.0114016831, -0.0874212608, 0.020981431, -0.127568886, 0.0844451338, 0.00714354217, -0.0613120124, -0.0566081777, -0.162151843, 0.0672827512, -0.077286616, -0.0474304631, -0.0929063633, -0.0875704363, 0.095430702, -0.0288354903, -0.0626533777, -0.00968232751, -0.00746659935, -0.158143908, 0.15200451, -0.0720696226, -0.0889598802, 0.079224363, 0.154342413, -0.0559937656, -0.0257438272, 0.0452196151, -0.0841155723, -0.068070814, -0.106328249, 0.0819824487, -0.128205806, -0.0245463252, -0.127599627, -0.0368299186, -0.162989303, 0.0764556378, 0.0239453018, 0.0943070054, -0.139077216, -0.0284653753, 0.148467928, 0.0383403152, 0.123082995, 0.0394094288, -0.0376930088, -0.130046725, -0.0765794441, -0.0595789626, -0.124194048, -0.0745625198, -0.0703442991, -0.0767715424, 0.0141807944, -0.151448116, 0.107176125, 0.152304411, 0.105451822, 0.0219457, -0.0640773103, -0.010845989, 0.108332992, -0.158579022, -0.0581467152, 0.101733625, 0.137660652, 0.0030760169, 0.0287179202, 0.133891582, -0.0398783386, -0.000854074955, 0.133014053, 0.137655258, 0.0579888821, 0.0522723049, 0.141502321, -0.0937897861, 0.00193537772, 0.0307513177, 0.0973593071, -0.0541716442, -0.0721254647, -0.0137725277, -0.0211353004, 0.154372394, -0.0886581317, 0.0983873382, 0.0898563042, -0.0761090145, -0.0455986895, -0.151796505, -0.0100342929, 0.143575042, -0.0641278028, 0.0476813614, -0.00897518732, 0.111726798, 0.0868349075, 0.0369581915, 0.0565167964, -0.117083244, -0.113838308, -0.0178825855, 0.0457149558, -0.00411985256, -0.10190326, -0.0801126882, 0.0446258038, 0.14128074, -0.0120808082, 0.0469621383, -0.00652398169, 0.0689584464, -0.0892492533, 0.0704481304, -0.131360695, 0.00791610871, 0.124002606, 0.0285931509, -0.133395582, -0.0275967121, 0.0657383651, -0.0628945231, -0.0796126053, 0.122940838, -0.0386064649, -0.0232444853, 0.140711948, -0.103686646, -0.00885927677, 0.118877523, -0.101937078, 0.160151228, -0.118134968, 0.0796763748, 0.138080776, -0.125875741, -0.0750917122, -0.0390297621, 0.0366276652, 0.163267136, -0.125967905, 0.0895617306, 0.0669770166, 0.145614386, -0.07808505, 0.05569987, -0.17504026, -0.0798169822, -0.0166844577, 0.0716707259, 0.011714654, 0.100986004, -0.0804149583, 0.0227044281, 0.159397155, -0.0321065634, -0.145676777, -0.0417278707, -0.146821395, -0.0551559478, -0.098714821, -0.00708699739, -0.078324087, 0.0873268619, 0.0700409859, -0.0579633191, 0.00693501532, 0.0628858954, -0.0673067048, -0.101266347, 0.00345513457, -0.0832723603, -0.166402042, -0.0803929865, 0.0198201444, 0.347372204, 0.0305967182, 0.412540674, -0.267104596, -0.00209473073, -0.0973251536, -0.192331493, -0.331010222, -0.0856090412, -0.304830521, -0.207485348, 0.141899422, -0.0334983803, -0.258603722, -0.536549151, 0.497887373, 0.418978423, -0.0626062378, -0.071420446, -0.400168687, 0.153853953, 0.0806448609, -0.166687846, -0.319215536, -0.0586516373, -0.212138534, 0.418498695, 0.036223188, 0.0417298451, 0.359410495, -0.380353272, -0.0642690137, -0.0847125053, -0.199162707, -0.128748477, -0.257194072, -0.265956461, 0.520730853, 0.0135677662, 0.46175909, -0.0989187434, -0.355642796, -0.0122152567, 0.438414723, 0.0280621052, -0.00993509591, -0.323545098, 0.414043814, -0.170853257, 0.15252775, 0.131180853, -0.0361544527, 0.353281707, 0.394390166, -0.398201078, -0.147230759, 0.44170922, -0.501864433, -0.13107498, -0.11892356, -0.217570409, -0.239248216, 0.425702542, 0.356086582, -0.0333236903, 0.143705428, -0.144949347, -0.0225226469, -0.311825037, -0.137032896, -0.0673775375, 0.277637184, -0.143999711, -0.412071317, -0.0232741944, 0.0338007957, 0.0173711777, 0.222030818, -0.457059532, -0.203986719, 0.41679585, -0.28484422, 0.518876314, 0.096483469, 0.356640786, 0.0531070381, -0.110804401, -0.109069236, 0.154181778, 0.21716471, 0.310356677, 0.43239224, 0.202034548, 0.620221794, -0.199884713, 0.0464695096, 0.12707141, 0.126740992, -0.0551695004, -0.0627429262, -0.133385226, -0.0879672766, 0.0976508856, 0.0430643111, -0.0311950594, -0.0251043141, 0.119974852, -0.127670139, -0.160888717, -0.0260237902, -0.0665860847, -0.0620029047, -0.0181810409, -0.0774263442, -0.162334114, 0.125682861, -0.0142752975, 0.054279089, -0.0176326931, -0.00877432525, -0.0643327385, 0.00476509333, -0.0449662507, -0.10598506, -0.0870684832, 0.126794785, -0.0860924274, -0.150241956, -0.131484509, 0.0600378364, 0.0202653557, 0.14740026, 0.116257191, -0.0322854072, -0.0585436299, -0.0956767723, -0.135802269, -0.044010289, -0.0221577734, 0.0177947134, -0.152910247, -0.101975754, -0.101217084, 0.0672132969, 0.150510609, -0.127762541, 0.16081199, 0.0981208384, -0.0670810193, -0.0528443903, -0.109811008, 0.0691851228, -0.0645181984, -0.162850976, -0.0379654765, -0.0623779297, 0.0587584376, 0.00559653342, 0.136839777, 0.0544781387, -0.144981384, 0.0847612768, 0.0283272862, 0.161950737, 0.0888574123, 0.144622713, 0.0429650098, 0.127184033, -0.0217859894, -0.0324133039, -0.150943786, -0.0317936689, 0.10203284, 0.0256467015, -0.0713156685, -0.156210557, 0.129269034, 0.007338956, -0.102121651, -0.0477264747, 0.0442777276, 0.0722139627, 0.101030886, -0.147381067, -0.142820626, 0.14448607, -0.138357788, -0.0785528272, 0.00679275393, -0.0126515776, 0.114257544, 0.0808940232, 0.41525802, -0.0470375717, 0.54068327, -0.24931632, -0.100485526, -0.0711906329, -0.190743431, -0.499752074, 0.0221821219, -0.432241619, -0.220779747, -0.00414595474, -0.148462296, -0.533766806, -0.517019451, 0.489838123, 0.320862293, -0.346463829, 0.135957927, -0.585019767, 0.0534664541, 0.0742014199, -0.16031085, -0.58774811, -0.191212773, -0.319360077, 0.429542243, -0.115652405, -0.107481323, 0.506136537, -0.258292496, 0.055115059, -0.022811681, -0.453629017, -0.112617515, -0.484506428, -0.440099955, 0.384203047, -0.038478829, 0.301786602, -0.0276364386, -0.296875954, -0.0370980948, 0.331825495, -0.10799434, -0.153116316, -0.401817709, 0.537028134, -0.535211504, -0.0156095624, 0.0163132641, 0.113064177, 0.500517607, 0.353334934, -0.224180207, -0.00614270568, 0.376861304, -0.444317281, 0.0732095987, -0.0399487317, -0.353808552, -0.280396104, 0.47777608, 0.376695752, -0.145461768, 0.123662502, 0.117217332, -0.136304766, -0.322687417, -0.0732764155, -0.0769338012, 0.320448786, -0.0291238688, -0.61821878, 0.0398676209, -0.108344354, -0.132738814, 0.30245924, -0.543233573, -0.498420089, 0.540336728, -0.754650891, 0.368320286, -0.000724732876, 0.28601414, -0.126356438, 0.137574002, -0.0683457926, -0.129003555, 0.218589857, 0.379687577, 0.314757347, 0.393100947, 0.640961766, -0.397934556, -0.0766773671, 0.267823637, -0.133264452, 0.668701172, -0.433248341, 0.101451606, 0.11710114, -0.537119746, -0.624923348, 0.10571602, -0.646909952, -0.45817557, -0.0412172452, -0.163217977, -0.630589783, -0.528855085, 0.490371138, 0.339602619, -0.196056575, -0.1115546, -0.726505637, 0.129455209, -0.15798521, -0.1603003, -0.418429017, -0.472715676, -0.506358325, 0.668755531, -0.115362599, -0.0895886868, 0.444033027, -0.354223549, -0.0517369509, 0.102366388, -0.527836204, 0.134996563, -0.403559595, -0.303828865, 0.663216233, -0.37628144, 0.591505468, -0.112084262, -0.489739925, -0.126792371, 0.521321654, -0.000668928027, -0.06336952, -0.743025482, 0.675772071, -0.351291776, -0.0242804438, 0.0475857556, -0.0739587173, 0.35162878, 0.480359286, -0.438748777, 0.091450125, 0.43106702, -0.763750434, -0.0540910885, 0.0284001827, -0.494619161, -0.496299535, 0.572596788, 0.409462839, 0.0841749609, -0.0476697758, -0.161480531, -0.0439777784, -0.263649672, 0.0257336814, -0.0144569101, 0.446306318, -0.0288852025, -0.432113081, 0.0087942956, 0.119196385, 0.0362982899, 0.41826278, -0.672761798, -0.398551553, 0.680422843, -0.594136596, 0.337536871, 0.142527401, 0.23631458, 0.11564514, 0.0946296081, 0.129702181, 0.000390827656, 0.446580708, 0.33545512, 0.550885737, 0.470069498, 0.623328447, -0.383132935, 0.138308018, 0.444388002, 0.028099522, 0.577534676, -0.42575258, 0.100100875, -0.132449746, -0.493283689, -0.388921916, 0.0513092428, -0.507928967, -0.31721133, -0.0679259673, -0.0863463804, -0.462516606, -0.623660803, 0.673458636, 0.502588868, -0.373455644, 0.00349247362, -0.697658658, 0.0437643081, 0.104052216, 0.160691947, -0.545008361, -0.402570963, -0.495602012, 0.630491197, 0.0313064605, 0.13320069, 0.524216652, -0.51990819, -0.111845151, 0.0225383788, -0.623089731, -0.0325553417, -0.293082386, -0.371053845, 0.528266668, -0.121174268, 0.644679904, 0.0882796645, -0.495728731, -0.108858526, 0.331112891, -0.133785814, 0.0913422704, -0.627573609, 0.537632287, -0.529607296, -0.125232965, -0.143395051, -0.0801532343, 0.286299229, 0.444152385, -0.502187073, -0.123857424, 0.401568681, -0.685675144, 0.0542019159, -0.00974772871, -0.504119217, -0.425121635, 0.579836071, 0.215468377, 0.13298586, -0.0903162658, 0.0165199488, -0.323535264, -0.234561488, -0.15145807, -0.124103874, 0.433957547, -0.0337882787, -0.601083159, 0.0218432266, -0.0260008872, -0.146205455, 0.441564649, -0.688122869, -0.223995849, 0.401472479, -0.596491992, 0.562832713, 0.0841847956, 0.49470067, -0.145028755, -0.0903297812, 0.013372764, 0.0394408107, 0.424351037, 0.343531489, 0.501020372, 0.418810219, 0.776348591, -0.273792207, -0.0818665102, 0.597009242, 0.04290995, 0.655070364, -0.538043678, 0.0370013267, -0.140541762, -0.685210943, -0.673634291, 0.0380292833, -0.472703099, -0.551744819, 0.0526464432, 0.0552807041, -0.707426965, -0.616695285, 0.724300444, 0.72779119, -0.207957208, 0.0112277921, -0.696847796, 0.158597738, -0.136686981, 0.0754225254, -0.593944609, -0.425629169, -0.763673723, 0.677075148, 0.0270163268, 0.119123586, 0.646436155, -0.610333562, 0.0353329331, 0.0828341842, -0.698317885, 0.000371947885, -0.463281274, -0.627031505, 0.526281416, -0.428260773, 0.423360348, -0.0180162638, -0.425837368, -0.126180887, 0.666808903, -0.0243054181, 0.0692905486, -0.678057969, 0.76500088, -0.4943524, -0.150353953, 0.109155007, 0.0488821827, 0.650208354, 0.501309156, -0.673963428, 0.0594189316, 0.499033362, -0.649286687, 0.122007728, 0.0483755767, -0.434515417, -0.658635199, 0.845367193, 0.572630584, 0.0664959103, 0.0177727044, 0.146929204, -0.0970276222, -0.376407534, 0.0163521618, -0.14672704, 0.374620467, 0.0465037674, -0.672666788, -0.0656483099, -0.0496134236, -0.0929352343, 0.401180208, -0.666605473, -0.476131976, 0.521337926, -0.794493794, 0.69625777, 0.151797771, 0.663843989, -0.122508794, 0.0165390465, 0.0905514061, -0.138756037, 0.319661826, 0.406682968, 0.490576744, 0.636822879, 0.61840719, -0.525159121, -0.0513994619, 0.503029764, -0.13656047, 0.815601945, -0.417270958, 0.104085445, 0.0526553765, -0.528447747, -0.7300331, 0.0137076378, -0.497281045, -0.544685602, -0.0433716886, -0.146049827, -0.638704002, -0.684384406, 0.649452984, 0.702250063, -0.438050747, 0.0139068058, -0.604019046, 0.100179672, 0.119058639, -0.0703429729, -0.680922389, -0.472380579, -0.649161637, 0.643359065, -0.0150906742, 0.0603066161, 0.43197611, -0.690997601, 0.0438588113, 0.0523733795, -0.521576762, -0.102957591, -0.41933915, -0.677487731, 0.593353391, -0.334632933, 0.511640549, 0.163541764, -0.466967374, 0.132696331, 0.54848963, -0.11855603, 0.0558734238, -0.645681262, 0.580150843, -0.428349078, -0.110145852, 0.143840998, -0.141338065, 0.518344045, 0.498623282, -0.628185153, 0.105362535, 0.515334249, -0.655823886, 0.0752197355, 0.145433754, -0.561434507, -0.572901249, 0.863208711, 0.357862741, -0.163092196, 0.138181031, 0.0153587759, -0.251604259, -0.487531364, 0.127054393, -0.0147024989, 0.515282214, 0.0958273113, -0.767876863, -0.0950485691, 0.0865165889, 0.141456872, 0.741376758, -0.744033873, -0.319546044, 0.648385465, -0.774301827, 0.673389792, -0.16039823, 0.471927881, -0.0583370999, 0.115023293, 0.0565826595, -0.0981604606, 0.523279786, 0.4614259, 0.542733967, 0.573020935, 0.763521791, -0.242885187, -0.0293573439, 0.069412291, 0.0730496198, -0.151006728, -0.145702794, 0.0900216103, -0.0994054452, 0.11095506, -0.101037003, -0.060667865, 0.0190453529, 0.0267233104, 0.0214355439, -0.0437630937, 0.0508560985, -0.136317253, 0.140143514, -0.08868853, -0.0774196312, -0.0449667946, -0.106950149, -0.147827655, 0.119437337, 0.0837459713, -0.00834037364, -0.0190687627, 0.0781720579, 0.129248857, 0.162696689, -0.138791069, -0.10027349, 0.00313524902, -0.0249195248, -0.0684585199, 0.131610036, -0.0957273766, -0.013932392, 0.144721597, 0.0370782018, 0.028160274, -0.0205518454, 0.0750066936, 0.104853898, 0.145021021, 0.0334349871, 0.135550469, 0.115787953, 0.0275911242, 0.0689579844, 0.112334222, 0.119560719, -0.144694433, -0.0604742467, -0.0382232964, -0.0974074826, 0.158459842, 0.159139752, -0.00982959569, -0.152535379, 0.0419855565, -0.129570946, 0.104130387, -0.157032207, 0.0459318161, -0.131371111, -0.126610234, 0.0640060604, -0.0769069046, -0.0855389163, -0.0414569527, -0.129209608, 0.00853239, 0.0531715006, 0.150542468, -0.13171187, -0.0431230813, 0.157875448, 0.0193243772, 0.0270704031, -0.153836682, 0.0295955241, 0.0157054812, 0.068245858, 0.000253170729, -0.115474865, -0.0709753782, 0.140475363, -0.111023337, -0.0244388282, -0.0692336634, 0.140080661, 0.110994577, 0.0787107795, 0.157543451, -0.0132067651, -0.0484567061, 0.155867875, -0.0193053037, -0.0161635727, 0.119335622, -0.0949590653, 0.0908037722, -0.108221561, -0.0622468218, 0.134051025, -0.0920001492, -0.0880780146, -0.121789694, 0.0584148616, 0.0480424613, -0.0165174901, 0.1272614, 0.105705976, 0.0111332238, -0.134370565, 0.0514526516, 0.0918411314, -0.0124515295, 0.0159996897, 0.141326576, 0.000145852566, -0.100328237, -0.0171524286, -0.148517296, -0.112245455, 0.14284423, -0.0440397859, 0.0482228994, -0.160654202, -0.0420692563, -0.0476969779, -0.0844033062, 0.0381466895, -0.0295516253, -0.120712176, 0.103265882, 0.0656362176, 0.113504618, -0.110794246, -0.0688497424, -0.106944188, -0.0667484105, 0.114784658, 0.0467143208, 0.0718533397, -0.104621768, 0.0242572725, -0.148502737, 0.0229506642, -0.124020137, -0.0880889446, 0.0819785744, -0.0242780596, 0.0188888013, -0.0801361129, -0.1584014, -0.162905246, 0.0192248076, -0.123885788, -0.036697045, 0.026028946, 0.0231203735, -0.120717764, 0.156676769, 0.0333094895, -0.142389998, 0.0376690775, 0.0765116215, -0.124334246, -0.0463511199, -0.0292654186, 0.0842002034, 0.106793165, 0.0637783706, 0.128580958, -0.116304636, -0.142138898, 0.0289230496, 0.0905574858, -0.15331392, -0.00102615356, 0.0834569037, -0.0417026207, -0.0329467207, -0.120827913, 0.0981094241, 0.00165192783, -0.141740307, 0.160194188, 0.00855514407, -0.0194704384, 0.0139152557, -0.0171852056, 0.435134917, 0.0533352345, 0.466278404, -0.30961141, 0.0102815628, 0.0293299556, -0.449819505, -0.481088132, -0.0896748453, -0.535767794, -0.389113933, -0.059349414, 0.0160006266, -0.5851686, -0.507782638, 0.422795147, 0.480564117, -0.290110648, 0.157965988, -0.6829772, -0.0210507214, 0.0563232899, 0.096057266, -0.423185289, -0.221076608, -0.583534896, 0.586024582, -0.0907108039, 0.138302475, 0.267823845, -0.322174847, -0.0115953088, 0.114385247, -0.580904901, -0.0221508294, -0.406589925, -0.283831, 0.520663798, -0.107653625, 0.339897811, -0.0166603774, -0.271357179, -0.0393348634, 0.359255582, 0.0572659522, 0.142239213, -0.635874271, 0.410241753, -0.43037048, 0.0587957799, -0.0729601085, -0.181916714, 0.425718218, 0.248500898, -0.387961894, -0.162950009, 0.277428448, -0.493088335, -0.0605593473, -0.0232945085, -0.479390204, -0.362918288, 0.498416305, 0.420660168, -0.109202415, -0.126010373, -0.117713347, -0.048794765, -0.241373956, -0.133012265, 0.0203766767, 0.351603448, -0.0330382809, -0.458165169, 0.0231650993, -0.109691262, 0.0796325207, 0.328488261, -0.612487912, -0.412912846, 0.463281184, -0.506850541, 0.408033788, -0.0622303188, 0.477035373, -8.11219215e-05, 0.0330588855, 0.140223742, 0.0604051054, 0.419340104, 0.271430701, 0.475094557, 0.404987395, 0.450934798, -0.143382207, -0.119593501, -0.0262070298, -0.0954136923, 0.0671947598, 0.0996865332, 0.020083949, -0.128543302, -0.118744731, 0.161292642, 0.0527010709, -0.0321330279, 0.0225084424, -0.0529962182, 0.106788605, -0.0269529969, -0.0499997661, 0.143568546, -0.0708172619, 0.125422418, -0.0541658551, 0.163316131, -0.0292220265, -0.0793786496, -0.125133738, 0.0109965801, -0.0055270046, -0.085991241, -0.118159272, 0.00876827538, 0.0744910687, 0.154188246, 0.00962387025, 0.0348311663, 0.109077573, 0.0620035678, 0.123497576, 0.142127812, -0.10050527, -0.0404578745, -0.0421698913, -0.0164550245, -0.0649667382, -0.0577578768, -0.160013646, 0.0386661738, 0.107988238, 0.0138740093, -0.135323167, -0.15442425, 0.0327413082, -0.0781763941, -0.0247027278, -0.00660693645, -0.15065226, 0.0256781131, -0.120672576, 0.0600239038, -0.133241981, -0.105128214, -0.145407572, 0.121236652, -0.114004299, 0.109494746, -0.00628599524, -0.103798516, -0.0417579114, 0.129987627, -0.089652881, -0.040289931, -0.125343397, 0.090357244, -0.0215902925, 0.0465506017, 0.0614771843, 0.120478421, 0.124835074, -0.110027343, 0.16117385, -0.0467158481, 0.0142052174, 0.0818445086, -0.0344318748, -0.0426447317, 0.160519302, -0.110517047, 0.00232745707, 0.048954919, -0.0981580764, -0.127706662, -0.0688704997, -0.133296415, -0.123790815, 0.0962895453, 0.150461793, 0.0300154686, 0.0295400023, -0.0175164938, -0.0737835541, -0.0637548044, -0.0610377789, -0.125476733, -0.163549796, -0.0998020098, -0.0539408252, 0.131315321, 0.0591077954, 0.0347940624, -0.114081636, -0.14958021, -0.0998097733, -0.0901194438, 0.0293716639, -0.157770172, -0.00564011931, -0.1546451, -0.0538466275, 0.0423156321, -0.0119268149, -0.115133904, -0.150866672, 0.162878394, 0.10041061, 0.141930223, 0.127972007, 0.121370971, 0.157082707, 0.0850015283, 0.0349835902, 0.123525709, -0.012712881, 0.00236654282, 0.131688774, 0.160950452, 0.123911619, 0.0888023376, -0.0555470958, 0.0705881417, 0.0336866677, 0.0400004387, -0.0906125084, -0.162759081, -0.00304476917, -0.154094875, -0.0224884748, -0.126035973, -0.0758281872, 0.142537475, 0.0748237222, -0.0121932924, 0.0262228847, -0.0996327773, 0.0805983543, -0.0137577355, 0.0500964224, -0.107271209, 0.0253515542, 0.0681271553, -0.0722264871, 0.0698977858, -0.104521722, -0.0034134239, -0.108044676, -0.0682371557, 0.0822340101, 0.108027935, 0.0442011803, -0.0698211491, 0.103643924, -0.152514398, -0.0841721892, 0.0655691773, 0.0676607043, 0.095651567, -0.0163287073, -0.0834635049, 0.159953088, -0.0276508629, 0.00471869111, 0.159102291, 0.0360194892, 0.066743657, 0.096793443, -0.0947196037, -0.0220860988, -0.0392077789, 0.0707284212, 0.158304006, -0.0932359248, -0.0517626703, 0.00560446084, -0.154681981, 0.0878305733, 0.162604749, -0.00177273154, -0.136650607, 0.00359109044, 0.00132665038, 0.0647623539, -0.0696758404, -0.161142543, 0.0701793581, -0.00121626258, 0.0116966814, -0.110020787, -0.0803181455, -0.124480926, -0.00105284154, 0.0978569984, 0.0786918551, -0.0612047464, 0.00649240613, 0.0497363806, -0.161141142, 0.0499025583, 0.0997779071, 0.033796072, -0.0494628027, -0.13143757, 0.0947518647, -0.0708334595, -0.140762463, 0.0681798309, -0.132274985, -0.115443841, -0.0256372243, -0.0475513488, -0.163624436, 0.0692263246, 0.0436404496, 0.0790618509, 0.0225345939, -0.046496354, -0.060157828, -0.139818832, 0.00770695508, 0.138914615, -0.0480370373, -0.163309768, 0.010941714, 0.0888002515, 0.01956819, -0.0516789705, 0.00118626654, -0.156167254, 0.0625212193, -0.0396163613, -0.0349113941, 0.0725515187, -0.120996602, -0.0737750083, 0.143910825, 0.0964934528, -0.133498266, -0.146321967, 0.0891873538, 0.1069282, -0.105225176, 0.142148226, 0.0290645808, -0.0745165572, -0.014673695, -0.131524116, -0.111877143, -0.0715093315, 0.123099774, -0.118344344, -0.152529642, -0.0799285695, 0.0937563479, -0.14088811, 0.0661247075, -0.019340232, 0.0506648719, -0.0676545799, -0.0187790394, 0.0012434274, -0.0999870449, -0.0336635262, 0.0313615203, -0.0311756581, 0.161171496, -0.0978405699, 0.0726053715, -0.0470858365, -0.131985292, -0.0252578259, 0.114766121, -0.0769705847, 0.0112785399, 0.0544565916, 0.0886667669, -0.00644554198, -0.0195663869, 0.15279147, 0.0430598259, -0.0460788757, 0.0370145589, 0.0732228309, -0.0897551551, -0.13718316, -0.0133368969, 0.10276401, -0.0558564141, 0.140054137, -0.106407106, -0.108627558, -0.0944892243, 0.0843421966, -0.150660455, -0.123637229, 0.16204676, -0.064826034, 0.106584102, -0.100369558, -0.0982201174, -0.132144302, -0.0457998812, 0.0477772057, 0.00509114563, 0.084395662, 0.0418061465, 0.018984437, 0.119122952, -0.0706580207, -0.0790217295, -0.046558708, 0.0440043211, 0.108298153, -0.0620034561, -0.0996157229, -0.0957243741, 0.102545679, 0.124085188, 0.0818397403, 0.16204235, -0.0891578645, -0.14002502, 0.0188542604, -0.155582845, -0.128179044, 0.0165965408, 0.120755643, 0.0472933948, 0.0604600757, -0.160928905, -0.12732555, -0.0997992009, -0.0310150981, -0.150829107, 0.0576651692, -0.0747323334, -0.0805957392, 0.123521775, 0.0893250406, 0.104241699, -0.0609934479, -0.0354587734, -0.112907983, 0.0816107392, -0.0680459216, 0.0333081186, 0.132987648, -0.0353368372, 0.146573931, -0.132101998, 0.150555521, -0.000697016716, 0.131190091, -0.0634880215, 0.10290885, -0.074080579, -0.0476958081, 0.0465862155, -0.0997000858, -0.108771354, -0.0696401, -0.122483671, 0.0509519726, 0.00759164989, -0.0848605484, -0.0562895387, -0.144697741, 0.0874796808, 0.0889988244, 0.0268278234, 0.0343950503, -0.141184896, 0.0220942944, -0.0393744595, 0.135214925, 0.110376537, 0.0996540934, 0.11919003, 0.0980022252, -0.0669112653, -0.155193776, 0.0452546924, -0.0703773424, 0.0583671853, -0.0346381813, 0.0513165705, -0.00258591701, 0.0447351784, -0.0900598615, 0.105706215, 0.146674991, -0.0620219484, -0.151174858, -0.0161081403, -0.100465514, -0.0336442813, -0.110900372, 0.00215126574, -0.0686746538, 0.00195884914, -0.0760199577, 0.106658101, -0.117959172, 0.0354569405, -0.00336793065, -0.0230299979, -0.0014782151, 0.0943241194, -0.0998774171, 0.0012039172, 0.113150835, 0.0110323876, -0.0261056572, -0.126829952, -0.0870876759, -0.11976859, 0.046524331, -0.071955286, 0.0405203402, 0.011234045, -0.154406205, -0.12930125, -0.023624232, 0.0756945983, 0.0907269865, -0.0393210873, -0.0752031282, -0.0358981788, -0.0751911774, -0.142585725, -0.0390843526, 5.15287029e-05, -0.075960584, 0.0311313868, -0.155949354, -0.104150869, -0.1187962, 0.0607762262, -0.0981793106, -0.113741107, 0.155204773, 0.0446541235, 0.118418485, 0.108119518, -0.133762747, 0.0919227302, -0.110248864, -0.116491996, -0.0400639623, 0.0946984887, -0.0689975768, -0.022416085, -0.11836338, -0.0799732804, -0.0902090967, -0.0792491436, 0.162841797, -0.0835223421, 0.107949615, 0.051379282, -0.136231199, 0.142566562, -0.0843271837, -0.149434701, -0.0448695868, -0.162784055, -0.153907061, -0.101484761, 0.00953845121, 0.426583201, -0.148609549, 0.115576871, 0.199490532, 0.0147352507, -0.117657743, 0.245287716, 0.135029003, 0.0666001812, 0.121388517, -0.0181217957, 0.216936842, -0.106331646, 0.0277778357, 0.153495222, -0.0800978318, 0.197749496, -0.138691336, -0.0196990892, 0.0528009906, 0.0243862551, 0.186370388, 0.175517678, -0.1221525, 0.0521855354, 0.0731666014, -0.154113561, 0.363856167, -0.0282237232, -0.158015102, 0.176865205, -0.0974879637, 0.450661808, 0.331305534, 0.0805322826, 0.0872784406, -0.100408114, -0.0638073161, 0.386017829, 0.0769390613, 0.00142675987, -0.162395611, -0.141840905, 0.198867813, 0.166513488, 0.161055252, -0.11835929, -0.0183188859, -0.156000659, -0.137438938, -0.0241766218, 0.264292717, -0.0963973999, 0.00985603686, 0.0537395552, -0.132096976, -0.0467022583, 0.206219435, 0.414941043, 0.0961033329, -0.258318126, 0.0483516604, -0.0401404426, -0.0940226987, 0.312713206, 0.0591716096, 0.0113053732, -0.0660526603, -0.00768682361, -0.034788806, 0.215964571, -0.0245724861, -0.0390488431, -0.118346334, -0.0609221458, 0.00612892304, 0.399582237, 0.203330249, 0.196806058, 0.0530752875, -0.120979592, -0.107711084, -0.0730255097, -0.107436724, -0.133462176, -0.0744402334, -0.244415417, -0.0644059032, -0.156561211, -0.197872341, -0.103289597, 0.377865851, -0.0912091658, 0.1201033, -0.160948843, 0.156024545, -0.0639129952, -0.090083316, 0.146453589, -0.133513406, 0.0668042153, -0.0696549639, -0.141248181, 0.0630055368, 0.07204777, -0.0348255932, 0.104903817, 0.112185001, 0.0530579835, 0.0353051573, 0.152558982, -0.0174464881, 0.0578029007, 0.105488569, 0.0597463995, 0.133562177, -0.0298817456, -0.00572316349, 0.140778273, -0.143284202, 0.070868969, 0.0905631185, 0.147948056, 0.00595268607, 0.111803114, 0.0150186718, -0.124211848, -0.111544259, -0.0879064053, 0.0283788741, 0.0223622769, 0.116948336, -0.134138405, -0.0613509566, -0.0249846131, -0.10112831, -0.0355166793, 0.153874338, -0.0331345946, -0.131313011, 0.108126283, -0.129989982, -0.0541868061, 0.0846642405, 0.150049508, 0.0616748184, 0.0230356902, 0.0458371788, -0.00594834983, 0.0577939004, -0.0151311308, -0.145535201, 0.049468115, 0.0481966734, -0.113490559, 0.112496555, 0.0780519545, 0.0340096354, -0.0834872648, -0.0842126906, 0.0518238842, 0.0795846432, 0.109701157, 0.00858768821, -0.113648981, -0.118920989, 0.101658702, 0.0139685273, -0.139759749, -0.143213376, 0.113406599, -0.0240487754, 0.118874878, 0.110942841, -0.124504417, -0.0329809338, 0.13233161, 0.143387914, 0.0195756704, 0.0417485088, 0.139091969, 0.0137803257, 0.0205974281, -0.110451728, -0.0441940725, -0.0737197548, 0.157211125, 0.135692805, -0.0257898979, 0.298779458, 0.0781985521, 0.73985666, -0.266648382, 0.158021152, 0.0878175497, -0.539944649, -0.468864471, 0.0780267864, -0.540843844, -0.301655084, -0.0518210381, -0.026734395, -0.5966115, -0.762952268, 0.608376324, 0.398852915, -0.428730398, 0.049971696, -0.877293885, -0.136541083, -0.0994077474, 0.105191648, -0.490723759, -0.217326015, -0.666309834, 0.778362572, -0.0650892258, -0.0835762545, 0.487896889, -0.573699355, -0.123805448, -0.14677234, -0.695474207, 0.151781172, -0.380929798, -0.430921823, 0.456907123, -0.241932958, 0.549462914, -0.128027797, -0.55221045, 0.0231493562, 0.42661494, 0.0878407359, 0.0608166158, -0.712416768, 0.63901335, -0.449384868, 0.159114778, 0.0459368229, 0.0560229085, 0.610547602, 0.439166307, -0.592269897, 0.0565300584, 0.432459027, -0.527898312, 0.103265107, 0.147524357, -0.516388357, -0.588715911, 0.584630847, 0.352748632, -0.110237658, -0.0693953186, -0.108473666, -0.346531063, -0.279783189, -0.0729684606, -0.0655859187, 0.316692352, -0.0261591226, -0.786450922, -0.0631145239, 0.139841437, -0.142838657, 0.555980444, -0.66320163, -0.440560728, 0.768226922, -0.572616398, 0.450141042, -0.0127197951, 0.578406453, -0.113352701, -0.160333842, -0.0408433527, -0.0532096624, 0.439689189, 0.509643078, 0.39703089, 0.380325615, 0.619017959, -0.466819972, -0.00208250037, 0.197571889, -0.127699718, 0.57061708, -0.0889461562, 0.125420928, -0.124083146, -0.276578277, -0.514425039, -0.146964327, -0.509113431, -0.211362898, -0.0108989729, -0.160072714, -0.547774315, -0.534742832, 0.395833552, 0.444723606, -0.232113659, 0.10457135, -0.327795565, -0.0158315152, -0.109176621, 0.0947844088, -0.381525606, -0.193215504, -0.381637394, 0.443191588, -0.0624629557, -0.0875668302, 0.421671033, -0.220988944, 0.0183748603, -0.0979562625, -0.243815437, -0.0816091374, -0.318637252, -0.332960784, 0.387937754, -0.277409554, 0.480808109, -0.153253913, -0.354886085, -0.110755458, 0.502071917, -0.000588700175, -0.0559961498, -0.504071116, 0.557788849, -0.311017245, -0.0190320462, -0.112524584, 0.135903507, 0.281695038, 0.396817982, -0.236351028, 0.0239005834, 0.300112993, -0.354014724, -0.151639357, -0.0630136654, -0.105432972, -0.339013815, 0.599060297, 0.374561906, -0.104892686, -0.0753091723, -0.0211449265, -0.134819672, -0.167134747, -0.106380664, -0.107125737, 0.190131694, 0.109646179, -0.258304358, 0.0528509617, -0.107956916, -0.162901938, 0.274834245, -0.527358353, -0.351559311, 0.255262375, -0.593395054, 0.473694742, 0.0425339937, 0.302442133, -0.0197344571, -0.0237521213, 0.0384304076, -0.0421131179, 0.29344365, 0.231285095, 0.428982615, 0.309211254, 0.506714523, -0.194418505, 0.115764767, -0.0791986361, -0.147098288, 0.185434774, 0.227256998, -0.128825843, 0.112930514, 0.311439842, -0.00934564229, 0.00648616254, 0.126490504, 0.383692741, -0.158667207, -0.0816213787, 0.219326809, -0.032250043, 0.243424058, 0.0349649936, 0.371581644, -0.0709593222, -0.0400902331, 0.0598755479, 0.0168898609, 0.0322019123, 0.0468513891, 0.266098768, 0.153939903, -0.0650820136, -0.0646832213, -0.141601965, -0.20775193, 0.294126153, 0.161030412, -0.0318337828, 0.0222735871, -0.138500065, 0.443114609, 0.300167769, 0.0713025928, 0.249774694, 0.0179388225, -0.0432932079, 0.473966599, 0.0670043826, 0.256366789, 0.0242951214, -0.12646386, 0.215348199, 0.164384544, 0.379755765, 0.0300121456, -0.0899164379, 0.0295841116, 0.141041934, 0.0596595742, 0.124051869, 0.0898015201, 0.0306205861, 0.185432822, 0.0973767042, -0.12642394, 0.243974239, 0.337619752, 0.0185867902, -0.176255584, -0.0507553145, 0.0465276837, 0.101288795, 0.0988561213, 0.26927191, 0.0359455496, -0.0644713417, -0.111713909, -0.0275543593, 0.0756363198, 0.129606321, -0.0822765008, -0.0942883864, 0.19877547, 0.19598493, 0.215467617, 0.291533828, 0.00361102726, 0.124397606, -0.0280649215, 0.168855429, -0.112812266, 0.122410379, 0.0934093297, -0.148264557, -0.19147487, 0.206352189, -0.0994248465, 0.0225330386, 0.0747373477, 0.255917758, 0.0614369214, 0.0724327862, -0.163247064, 0.122555465, -0.0454005823, 0.0308880359, -0.0578934774, 0.150650114, -0.149725288, 0.0518169105, -0.0274477303, -0.0175606608, -0.0310429484, -0.0695917085, 0.0271570683, -0.0377356112, -0.0874331668, -0.159476444, 0.0832052976, -0.120977715, 0.056534633, 0.119316041, -0.0385935158, 0.155146539, 0.0712380558, -0.100473084, 0.0589886606, -0.106654853, 0.130597323, -0.052939482, 0.0062623471, 0.105926424, 0.132178992, -0.0180872381, -0.103644699, -0.0419721752, -0.101392165, 0.100607246, 0.0282868296, 0.0239832699, 0.0741458237, 0.142718792, 0.036145851, 0.0679779053, 0.0737555027, -0.0777623132, -0.118951581, 0.152075291, -0.077001296, -0.0121540725, -0.162707806, -0.0802720636, -0.000443041325, -0.137032732, 0.125278503, -0.0793484524, 0.0357272327, 0.154186189, -0.146461859, 0.120278478, 0.0228909701, 0.0579886436, 0.119533151, 0.109961629, 0.0650678426, 0.0944842398, -0.0540032163, -0.00230793655, -0.0306214094, -0.0839392766, -0.101581298, -0.0297169536, 0.00261315703, -0.0793418586, 0.0962284505, 0.0747976154, -0.0490718186, -0.0460839123, -0.121211097, -0.0941298455, 0.147601575, -0.00747478008, -0.0966355428, 0.0673684478, 0.0190058649, 0.0783318132, 0.155542791, 0.154795766, 0.115915358, -0.0469682291, 0.0349576324, 0.0622119457, -0.0650975406, -0.129059151, -0.147409394, -0.0998990089, -0.0230246037, -0.0337439477, -0.0809858665, -0.158101678, -0.0520249605, 0.155415684, -0.121042997, 0.149232894, 0.0681352764, -0.0599856302, -0.120198473, -0.102902919, -0.108941555, 0.0707386434, -0.163428396, 0.129345238, -0.0824232548, -0.0146582872, 0.0550943017, 0.0509623587, -0.098253876, -0.101240456, 0.0781475902, -0.129406273, -0.134796083, 0.154310763, -0.0798555985, 0.154313385, 0.0380191356, 0.0932592154, 0.0412110835, -0.0763610452, 0.0198271275, -0.141942278, 0.163606405, -0.115325183, -0.146009341, 0.0275302231, -0.122357205, 0.115435362, 0.0795787424, 0.132455558, -0.0191496909, -0.0176981688, -0.128091753, -0.0139716119, -0.0840594992, 0.0725945234, -0.0903724134, 0.0669592768, -0.142521769, 0.0478438437, 0.0334864557, -0.112349331, 0.0355492234, -0.0227393359, -0.144553527, -0.0324503332, 0.16084832, 0.14594382, -0.160798505, -0.00560747087, 0.0450707823, -0.0263125449, 0.0697827488, -0.0987388939, -0.0254066885, 0.0437710583, -0.122737065, -0.0671603531, 0.0593396127, -0.105872646, -0.112519696, -0.00898827612, 0.106537521, -0.07144963, 0.129475683, 0.0547391474, -0.152269349, -0.0508661717, 0.00455754995, -0.000966608524, 0.120649546, 0.13629204, -0.147438228, -0.0119368136, -0.0535460189, 0.0359031707, -0.0802643374, -0.136192709, 0.108641565, -0.0409720466, 0.143817961, 0.0494245589, -0.104909658, 0.0250150412];
    CONSTANT bias_1 : ARRAY[0..95] OF REAL := [-0.00675970502, -0.136126995, 0, -0.122499049, 0.242127135, 0, -0.0310927685, 0.207573012, 0.0948098674, 0, 0.115450546, 0.258484989, -0.00888741482, -0.00828406774, 0.119643688, 0.127291426, -0.129898831, -0.0517314821, 0.245927826, -0.0048302412, 0.133843109, 0, -0.0133913904, -0.0135692973, 0.0960704908, 0.291111261, 0.133287236, -0.122080714, 0, -0.00517006498, -0.226739645, 0.187288508, 0, 0, 0.136925355, -0.00909534469, 0.298944861, 0.226344824, -0.121498398, 0.234410852, -0.125201017, -0.00906701386, 0.297800422, 0, -0.0485578477, 0, 0, 0.132167235, -0.105923273, 0.202280939, 0, -0.00390069163, -0.00429093977, -0.13896066, -0.118062675, 0.211628303, 0, -0.119156256, 0.132621035, 0, -0.00772260362, 0.282757133, 0.248255253, -0.135500908, -0.159288019, 0, 0, 0, 0.222187474, 0.203655556, -0.0318242013, -0.0157510564, -0.185170233, -0.0148093309, 0.114873521, -0.012113723, 0, 0, -0.0339766107, 0.127130404, 0.239730254, 0.00635725306, 0.101751298, -0.00261538732, 0, -0.126262948, 0, -0.0100879008, 0, 0, -0.201107219, -0.109117478, -0.125762165, -0.1518161, -0.0896416381, 0.276514798];
    CONSTANT weights_2 : ARRAY[0..287] OF REAL := [-0.086540468, 0.172771111, -0.220383257, -0.552691996, 0.0318835452, 0.612700164, -0.0329583585, -0.0454194695, 0.227657318, -0.476521522, 0.193516552, 0.416927308, 0.360883504, 0.35479334, -0.725205362, 0.0127351284, 0.00659608841, -0.077765286, 0.0985900313, 0.120690353, 0.105450228, 0.508144796, 0.130406424, -1.01746202, 0.904253662, -1.11978483, -0.232323259, 0.181972265, 0.00731435418, -0.0696650892, 1.03260088, -1.09293258, -0.287332207, 0.370921373, 0.321434826, -0.712032735, -0.0679141358, 0.179906562, -0.124551736, 0.192289323, -0.140516713, 0.0810432881, 0.856259704, -1.07160294, -0.223457828, 0.807030499, -0.976367593, -0.307652324, -0.786935031, -0.107092589, 0.150858521, -0.624960959, 0.36329934, 0.532729268, 0.384019405, 0.46479398, -0.802043259, 0.187860116, -0.136551112, 0.0211512949, 0.720803916, -0.827788591, -0.298880219, -0.202536553, 0.173984587, 0.185747623, -0.184981599, 0.0150071271, 0.00353488303, 0.0683722198, 0.187118113, 0.237856477, 1.01755667, -1.10523689, -0.268671334, 0.240274504, 0.30826062, -0.654990911, 0.872478366, -1.05786157, -0.229688749, -0.66336894, 0.0199285392, 0.532636046, -0.0841914713, 0.0642075539, 0.0174617469, -0.0364442356, 0.188555226, -0.242369831, 0.00474316673, -0.759811342, 0.954901636, 0.593428373, 0.096972242, -1.04332292, -0.205035418, 0.18625772, 0.209811807, 0.172150373, 0.0444886386, -0.186326519, 0.902395904, -1.12277734, -0.0967059359, -0.0028087846, 0.141072839, 0.130949974, 0.330060393, 0.323049426, -0.685176551, 0.492645383, 0.322297305, -0.804180861, -0.752909601, -0.107810475, 0.338000387, 0.220442653, 0.451399148, -0.57051903, -0.757164657, -0.126809373, 0.439987898, 0.0298772864, 0.00199659704, 0.166657642, 0.229579955, 0.268833876, -0.694251597, -0.0976240188, 0.0951045454, 0.2128084, -0.488305151, 0.345968217, 0.402587503, 0.0220696926, 0.122957081, 0.138620675, -0.146714658, 0.128199548, 0.0768355131, 0.988235116, -0.820175171, -0.0243866928, -0.564573824, 0.0925929025, 0.436609149, 0.605118215, 0.151139334, -1.10266984, 0.227359504, 0.0128947198, 0.0949031711, 0.120222516, 0.206790701, -0.00842625648, 0.120845072, 0.212780789, 0.12719503, -0.755692124, -0.150177613, 0.340954095, -0.853432715, -0.333076835, 0.391219765, 0.48939836, -0.116058439, -1.27640653, 0.0483904779, 0.217980474, -0.00876715779, -0.644433141, 0.0299610049, 0.399048507, 0.929591358, -0.906723499, -0.0457304083, 0.0974808037, -0.178352863, -0.0875617117, -0.169119462, -0.014128576, 0.133027628, 0.469002575, 0.474750727, -0.581674278, 0.372726113, 0.190089732, -0.973690569, -0.53365171, 0.140256211, 0.40247342, -0.113590144, -1.07570827, 0.916958451, -0.124050736, 0.0386698842, 0.104596823, 0.0975920856, -0.122577384, -0.230316952, 0.0917100608, -0.204680085, -0.157175794, 0.0664396286, 0.443755388, -0.550633371, 0.524068952, 0.155129775, -1.07333207, -0.0423594192, 0.0332752727, 0.193382502, -0.147190854, 0.123858854, -0.18527922, -0.251415074, -1.22913897, 0.845771313, -0.110015817, 0.065641731, 0.0683446452, 0.979607761, -0.910373867, -0.153985277, -0.0826165602, 0.125199199, 0.105670959, 0.127799779, -0.173133329, -0.0312328637, 0.147351772, 0.183071434, -0.226357937, -0.664937735, 0.321295112, 0.338666469, 1.03204453, -0.964660764, -0.207029104, 0.53012073, 0.460012823, -0.891147494, -0.551259696, 0.262762219, 0.241604507, 0.96495378, -0.912866771, -0.143412411, -0.645358205, 0.383842945, 0.425131768, -0.0753789395, -0.00826120377, 0.0299984515, -0.784333527, -0.1359182, 0.4243536, 0.178426176, -0.175408095, -0.077928111, -0.240787193, -0.203756183, 0.0390834771, -0.0964978486, -0.143233955, -0.104287267, 0.22191146, -0.0092907697, 0.138567775, -0.176785797, -0.841094136, 0.893011391, -0.736852944, 0.00464549148, 0.51239562, -0.529248655, 0.0516002066, 0.706514895, -0.518120229, 0.0655920431, 0.586107075, -0.604757965, 0.123719975, 0.379719675, 0.365877658, 0.503408611, -0.481252313];
    CONSTANT bias_2 : ARRAY[0..2] OF REAL := [0.0345217623, 0.145207137, -0.191580176];
END_VAR
